// TIA Portal V17 export
// export: Created 2025-03-05T08:01:27.0836463Z, ExportSetting WithDefaults, DisplayName Totally Integrated Automation Portal, DisplayVersion V17 Update 8, DisplayName TIA Portal Openness, DisplayVersion V17 Update 8, DisplayName TIA Portal Version Control Interface, DisplayVersion V17, DisplayName SINAMICS Startdrive Advanced, DisplayVersion V17 SP2, DisplayName SINAMICS Startdrive G110M, G120, G120C, G120D, G120P, G115D, DisplayVersion V17 SP2, DisplayName SINAMICS Startdrive G130, G150, S120, S150, SINAMICS MV, S210, DisplayVersion V17 SP2, DisplayName STEP 7 Professional, DisplayVersion V17 Update 8, DisplayName SINUMERIK ONE STEP 7 Toolbox, DisplayVersion V17 Update 12, DisplayName SINUMERIK 840D sl STEP 7 Toolbox, DisplayVersion V17 Update 12, DisplayName STEP 7 Safety, DisplayVersion V17 Update 6, DisplayName WinCC Advanced, DisplayVersion V17 Update 8
FUNCTION "FC16011_METHOD_CALLS_U01_STA3_MEAS" : Void   // FC16011, LAD
{ S7_Optimized_Access := 'TRUE' }
VERSION : 0.1
// stored: AutoNumber false, IsIECCheckEnabled false, SetENOAutomatically false, UDAEnableTagReadback false
   VAR_TEMP
      AUX_WSTRING_PART_ID_STA3 : WString;
      AUX_WCHARS : Array[0..63] of WChar;
      index : Int;
      ALARM_AUX : Bool;
   END_VAR
   VAR_TEMP   // added for the SCL form of the ladder/FBD networks
      _w1 : Bool;
      _w2 : Bool;
      _w3 : Bool;
      _s5time1 : S5Time;
      _w4 : Bool;
   END_VAR
BEGIN

REGION Network 1 (SCL): TRANSFORM TO WCHARS
   FOR #index := 0 TO 63 DO
       #AUX_WCHARS[#index] := CHAR_TO_WCHAR("DB8000_PART_STATUS".UNIT_01.STATION_3.PART_A.PART_ID[#index]);
   END_FOR;
END_REGION

REGION Network 2: TRANSFORM TO WSTRING
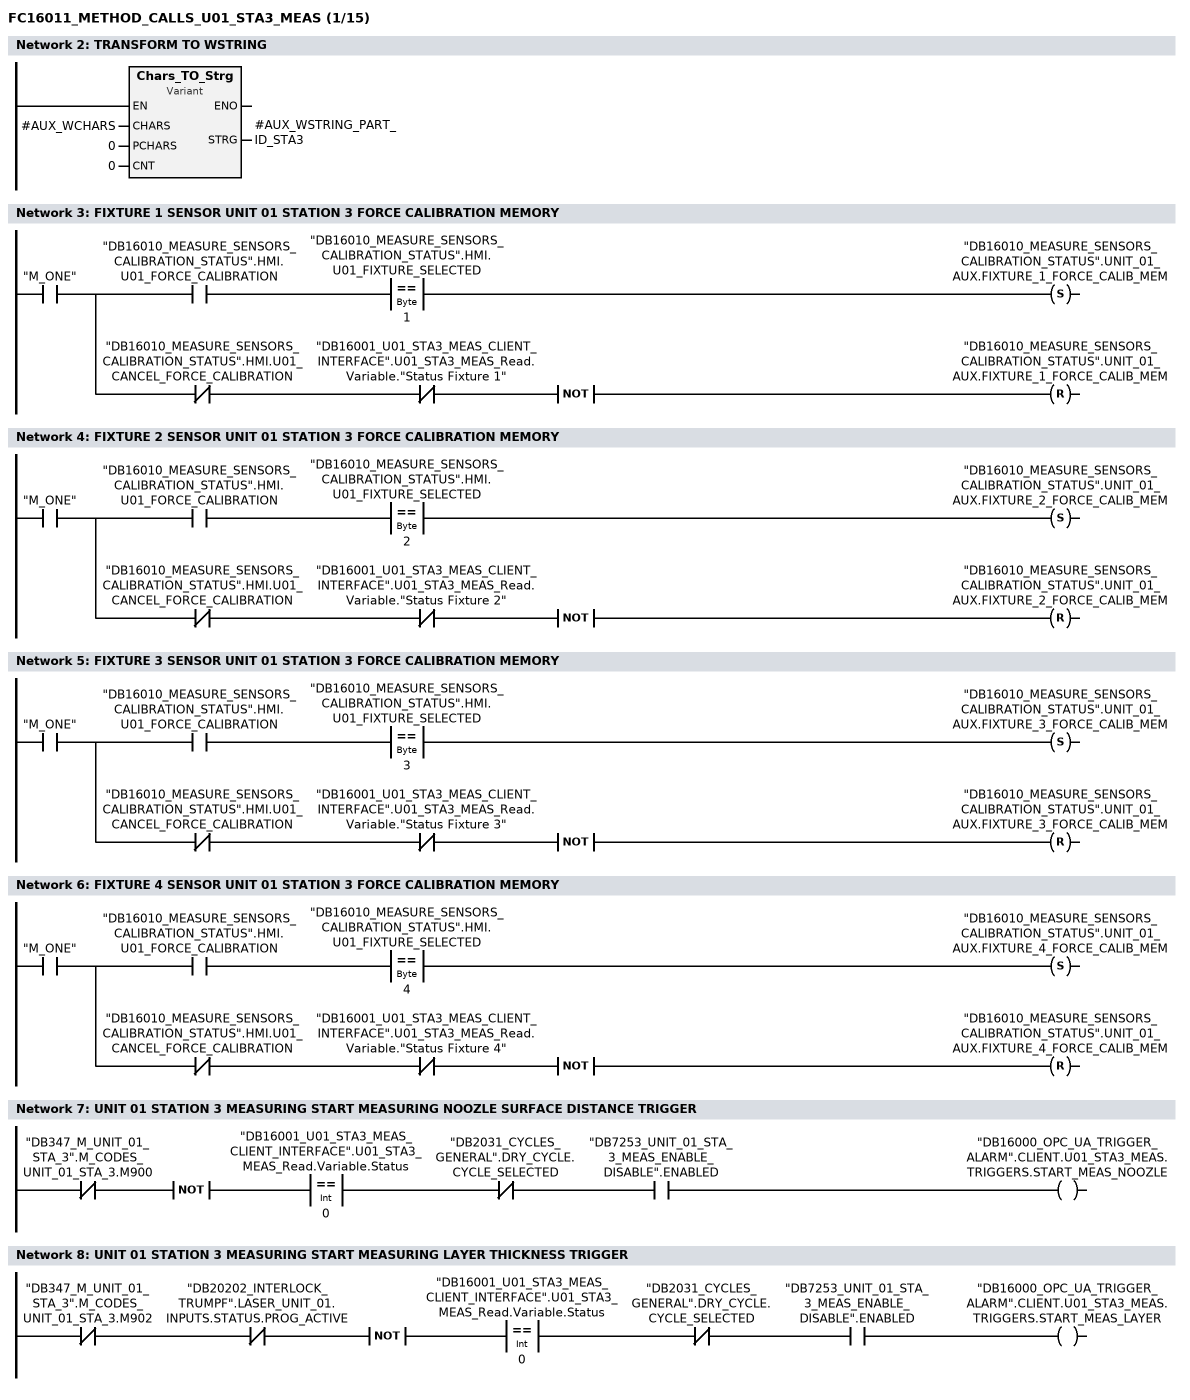
   RUNG wire#powerrail
      { S7_Templates := "[ptr_type := Variant, str_type := WString]" } Chars_TO_Strg(Chars := #AUX_WCHARS, pChars := 0, Cnt := 0, Strg => #AUX_WSTRING_PART_ID_STA3)
   END_RUNG
   // the same network as SCL:
   Chars_TO_Strg(Chars := #AUX_WCHARS, pChars := 0, Cnt := 0, Strg => #AUX_WSTRING_PART_ID_STA3);
END_REGION

REGION Network 3: FIXTURE 1 SENSOR UNIT 01 STATION 3 FORCE CALIBRATION MEMORY
   RUNG wire#powerrail
      Contact( "M_ONE" )
      wire#w1
      Contact( "DB16010_MEASURE_SENSORS_CALIBRATION_STATUS".HMI.U01_FORCE_CALIBRATION )
      { S7_Templates := "SrcType := Byte" } EQ_Contact(in1 := "DB16010_MEASURE_SENSORS_CALIBRATION_STATUS".HMI.U01_FIXTURE_SELECTED, in2 := 1)
      S_Coil( "DB16010_MEASURE_SENSORS_CALIBRATION_STATUS".UNIT_01_AUX.FIXTURE_1_FORCE_CALIB_MEM )
   END_RUNG
   RUNG wire#w1
      I_Contact( "DB16010_MEASURE_SENSORS_CALIBRATION_STATUS".HMI.U01_CANCEL_FORCE_CALIBRATION )
      I_Contact( "DB16001_U01_STA3_MEAS_CLIENT_INTERFACE".U01_STA3_MEAS_Read.Variable."Status Fixture 1" )
      Not()
      R_Coil( "DB16010_MEASURE_SENSORS_CALIBRATION_STATUS".UNIT_01_AUX.FIXTURE_1_FORCE_CALIB_MEM )
   END_RUNG
   // the same network as SCL:
   IF "M_ONE" AND "DB16010_MEASURE_SENSORS_CALIBRATION_STATUS".HMI.U01_FORCE_CALIBRATION AND ("DB16010_MEASURE_SENSORS_CALIBRATION_STATUS".HMI.U01_FIXTURE_SELECTED = 1) THEN
       "DB16010_MEASURE_SENSORS_CALIBRATION_STATUS".UNIT_01_AUX.FIXTURE_1_FORCE_CALIB_MEM := TRUE;
   END_IF;
   IF NOT ("M_ONE" AND NOT "DB16010_MEASURE_SENSORS_CALIBRATION_STATUS".HMI.U01_CANCEL_FORCE_CALIBRATION AND NOT "DB16001_U01_STA3_MEAS_CLIENT_INTERFACE".U01_STA3_MEAS_Read.Variable."Status Fixture 1") THEN
       "DB16010_MEASURE_SENSORS_CALIBRATION_STATUS".UNIT_01_AUX.FIXTURE_1_FORCE_CALIB_MEM := FALSE;
   END_IF;
END_REGION

REGION Network 4: FIXTURE 2 SENSOR UNIT 01 STATION 3 FORCE CALIBRATION MEMORY
   RUNG wire#powerrail
      Contact( "M_ONE" )
      wire#w1
      Contact( "DB16010_MEASURE_SENSORS_CALIBRATION_STATUS".HMI.U01_FORCE_CALIBRATION )
      { S7_Templates := "SrcType := Byte" } EQ_Contact(in1 := "DB16010_MEASURE_SENSORS_CALIBRATION_STATUS".HMI.U01_FIXTURE_SELECTED, in2 := 2)
      S_Coil( "DB16010_MEASURE_SENSORS_CALIBRATION_STATUS".UNIT_01_AUX.FIXTURE_2_FORCE_CALIB_MEM )
   END_RUNG
   RUNG wire#w1
      I_Contact( "DB16010_MEASURE_SENSORS_CALIBRATION_STATUS".HMI.U01_CANCEL_FORCE_CALIBRATION )
      I_Contact( "DB16001_U01_STA3_MEAS_CLIENT_INTERFACE".U01_STA3_MEAS_Read.Variable."Status Fixture 2" )
      Not()
      R_Coil( "DB16010_MEASURE_SENSORS_CALIBRATION_STATUS".UNIT_01_AUX.FIXTURE_2_FORCE_CALIB_MEM )
   END_RUNG
   // the same network as SCL:
   IF "M_ONE" AND "DB16010_MEASURE_SENSORS_CALIBRATION_STATUS".HMI.U01_FORCE_CALIBRATION AND ("DB16010_MEASURE_SENSORS_CALIBRATION_STATUS".HMI.U01_FIXTURE_SELECTED = 2) THEN
       "DB16010_MEASURE_SENSORS_CALIBRATION_STATUS".UNIT_01_AUX.FIXTURE_2_FORCE_CALIB_MEM := TRUE;
   END_IF;
   IF NOT ("M_ONE" AND NOT "DB16010_MEASURE_SENSORS_CALIBRATION_STATUS".HMI.U01_CANCEL_FORCE_CALIBRATION AND NOT "DB16001_U01_STA3_MEAS_CLIENT_INTERFACE".U01_STA3_MEAS_Read.Variable."Status Fixture 2") THEN
       "DB16010_MEASURE_SENSORS_CALIBRATION_STATUS".UNIT_01_AUX.FIXTURE_2_FORCE_CALIB_MEM := FALSE;
   END_IF;
END_REGION

REGION Network 5: FIXTURE 3 SENSOR UNIT 01 STATION 3 FORCE CALIBRATION MEMORY
   RUNG wire#powerrail
      Contact( "M_ONE" )
      wire#w1
      Contact( "DB16010_MEASURE_SENSORS_CALIBRATION_STATUS".HMI.U01_FORCE_CALIBRATION )
      { S7_Templates := "SrcType := Byte" } EQ_Contact(in1 := "DB16010_MEASURE_SENSORS_CALIBRATION_STATUS".HMI.U01_FIXTURE_SELECTED, in2 := 3)
      S_Coil( "DB16010_MEASURE_SENSORS_CALIBRATION_STATUS".UNIT_01_AUX.FIXTURE_3_FORCE_CALIB_MEM )
   END_RUNG
   RUNG wire#w1
      I_Contact( "DB16010_MEASURE_SENSORS_CALIBRATION_STATUS".HMI.U01_CANCEL_FORCE_CALIBRATION )
      I_Contact( "DB16001_U01_STA3_MEAS_CLIENT_INTERFACE".U01_STA3_MEAS_Read.Variable."Status Fixture 3" )
      Not()
      R_Coil( "DB16010_MEASURE_SENSORS_CALIBRATION_STATUS".UNIT_01_AUX.FIXTURE_3_FORCE_CALIB_MEM )
   END_RUNG
   // the same network as SCL:
   IF "M_ONE" AND "DB16010_MEASURE_SENSORS_CALIBRATION_STATUS".HMI.U01_FORCE_CALIBRATION AND ("DB16010_MEASURE_SENSORS_CALIBRATION_STATUS".HMI.U01_FIXTURE_SELECTED = 3) THEN
       "DB16010_MEASURE_SENSORS_CALIBRATION_STATUS".UNIT_01_AUX.FIXTURE_3_FORCE_CALIB_MEM := TRUE;
   END_IF;
   IF NOT ("M_ONE" AND NOT "DB16010_MEASURE_SENSORS_CALIBRATION_STATUS".HMI.U01_CANCEL_FORCE_CALIBRATION AND NOT "DB16001_U01_STA3_MEAS_CLIENT_INTERFACE".U01_STA3_MEAS_Read.Variable."Status Fixture 3") THEN
       "DB16010_MEASURE_SENSORS_CALIBRATION_STATUS".UNIT_01_AUX.FIXTURE_3_FORCE_CALIB_MEM := FALSE;
   END_IF;
END_REGION

REGION Network 6: FIXTURE 4 SENSOR UNIT 01 STATION 3 FORCE CALIBRATION MEMORY
   RUNG wire#powerrail
      Contact( "M_ONE" )
      wire#w1
      Contact( "DB16010_MEASURE_SENSORS_CALIBRATION_STATUS".HMI.U01_FORCE_CALIBRATION )
      { S7_Templates := "SrcType := Byte" } EQ_Contact(in1 := "DB16010_MEASURE_SENSORS_CALIBRATION_STATUS".HMI.U01_FIXTURE_SELECTED, in2 := 4)
      S_Coil( "DB16010_MEASURE_SENSORS_CALIBRATION_STATUS".UNIT_01_AUX.FIXTURE_4_FORCE_CALIB_MEM )
   END_RUNG
   RUNG wire#w1
      I_Contact( "DB16010_MEASURE_SENSORS_CALIBRATION_STATUS".HMI.U01_CANCEL_FORCE_CALIBRATION )
      I_Contact( "DB16001_U01_STA3_MEAS_CLIENT_INTERFACE".U01_STA3_MEAS_Read.Variable."Status Fixture 4" )
      Not()
      R_Coil( "DB16010_MEASURE_SENSORS_CALIBRATION_STATUS".UNIT_01_AUX.FIXTURE_4_FORCE_CALIB_MEM )
   END_RUNG
   // the same network as SCL:
   IF "M_ONE" AND "DB16010_MEASURE_SENSORS_CALIBRATION_STATUS".HMI.U01_FORCE_CALIBRATION AND ("DB16010_MEASURE_SENSORS_CALIBRATION_STATUS".HMI.U01_FIXTURE_SELECTED = 4) THEN
       "DB16010_MEASURE_SENSORS_CALIBRATION_STATUS".UNIT_01_AUX.FIXTURE_4_FORCE_CALIB_MEM := TRUE;
   END_IF;
   IF NOT ("M_ONE" AND NOT "DB16010_MEASURE_SENSORS_CALIBRATION_STATUS".HMI.U01_CANCEL_FORCE_CALIBRATION AND NOT "DB16001_U01_STA3_MEAS_CLIENT_INTERFACE".U01_STA3_MEAS_Read.Variable."Status Fixture 4") THEN
       "DB16010_MEASURE_SENSORS_CALIBRATION_STATUS".UNIT_01_AUX.FIXTURE_4_FORCE_CALIB_MEM := FALSE;
   END_IF;
END_REGION

REGION Network 7: UNIT 01 STATION 3 MEASURING START MEASURING NOOZLE SURFACE DISTANCE TRIGGER
   RUNG wire#powerrail
      I_Contact( "DB347_M_UNIT_01_STA_3".M_CODES_UNIT_01_STA_3.M900 )
      Not()
      { S7_Templates := "SrcType := Int" } EQ_Contact(in1 := "DB16001_U01_STA3_MEAS_CLIENT_INTERFACE".U01_STA3_MEAS_Read.Variable.Status, in2 := 0)
      I_Contact( "DB2031_CYCLES_GENERAL".DRY_CYCLE.CYCLE_SELECTED )
      Contact( "DB7253_UNIT_01_STA_3_MEAS_ENABLE_DISABLE".ENABLED )
      Coil( "DB16000_OPC_UA_TRIGGER_ALARM".CLIENT.U01_STA3_MEAS.TRIGGERS.START_MEAS_NOOZLE )
   END_RUNG
   // the same network as SCL:
   "DB16000_OPC_UA_TRIGGER_ALARM".CLIENT.U01_STA3_MEAS.TRIGGERS.START_MEAS_NOOZLE := NOT (NOT "DB347_M_UNIT_01_STA_3".M_CODES_UNIT_01_STA_3.M900) AND ("DB16001_U01_STA3_MEAS_CLIENT_INTERFACE".U01_STA3_MEAS_Read.Variable.Status = 0) AND NOT "DB2031_CYCLES_GENERAL".DRY_CYCLE.CYCLE_SELECTED AND "DB7253_UNIT_01_STA_3_MEAS_ENABLE_DISABLE".ENABLED;
END_REGION

REGION Network 8: UNIT 01 STATION 3 MEASURING START MEASURING LAYER THICKNESS TRIGGER
   RUNG wire#powerrail
      I_Contact( "DB347_M_UNIT_01_STA_3".M_CODES_UNIT_01_STA_3.M902 )
      I_Contact( "DB20202_INTERLOCK_TRUMPF".LASER_UNIT_01.INPUTS.STATUS.PROG_ACTIVE )
      Not()
      { S7_Templates := "SrcType := Int" } EQ_Contact(in1 := "DB16001_U01_STA3_MEAS_CLIENT_INTERFACE".U01_STA3_MEAS_Read.Variable.Status, in2 := 0)
      I_Contact( "DB2031_CYCLES_GENERAL".DRY_CYCLE.CYCLE_SELECTED )
      Contact( "DB7253_UNIT_01_STA_3_MEAS_ENABLE_DISABLE".ENABLED )
      Coil( "DB16000_OPC_UA_TRIGGER_ALARM".CLIENT.U01_STA3_MEAS.TRIGGERS.START_MEAS_LAYER )
   END_RUNG
   // the same network as SCL:
   "DB16000_OPC_UA_TRIGGER_ALARM".CLIENT.U01_STA3_MEAS.TRIGGERS.START_MEAS_LAYER := NOT (NOT "DB347_M_UNIT_01_STA_3".M_CODES_UNIT_01_STA_3.M902 AND NOT "DB20202_INTERLOCK_TRUMPF".LASER_UNIT_01.INPUTS.STATUS.PROG_ACTIVE) AND ("DB16001_U01_STA3_MEAS_CLIENT_INTERFACE".U01_STA3_MEAS_Read.Variable.Status = 0) AND NOT "DB2031_CYCLES_GENERAL".DRY_CYCLE.CYCLE_SELECTED AND "DB7253_UNIT_01_STA_3_MEAS_ENABLE_DISABLE".ENABLED;
END_REGION

REGION Network 9: UNIT 01 STATION 3 MEASURING STOP MEASURING LAYER THICKNESS TRIGGER
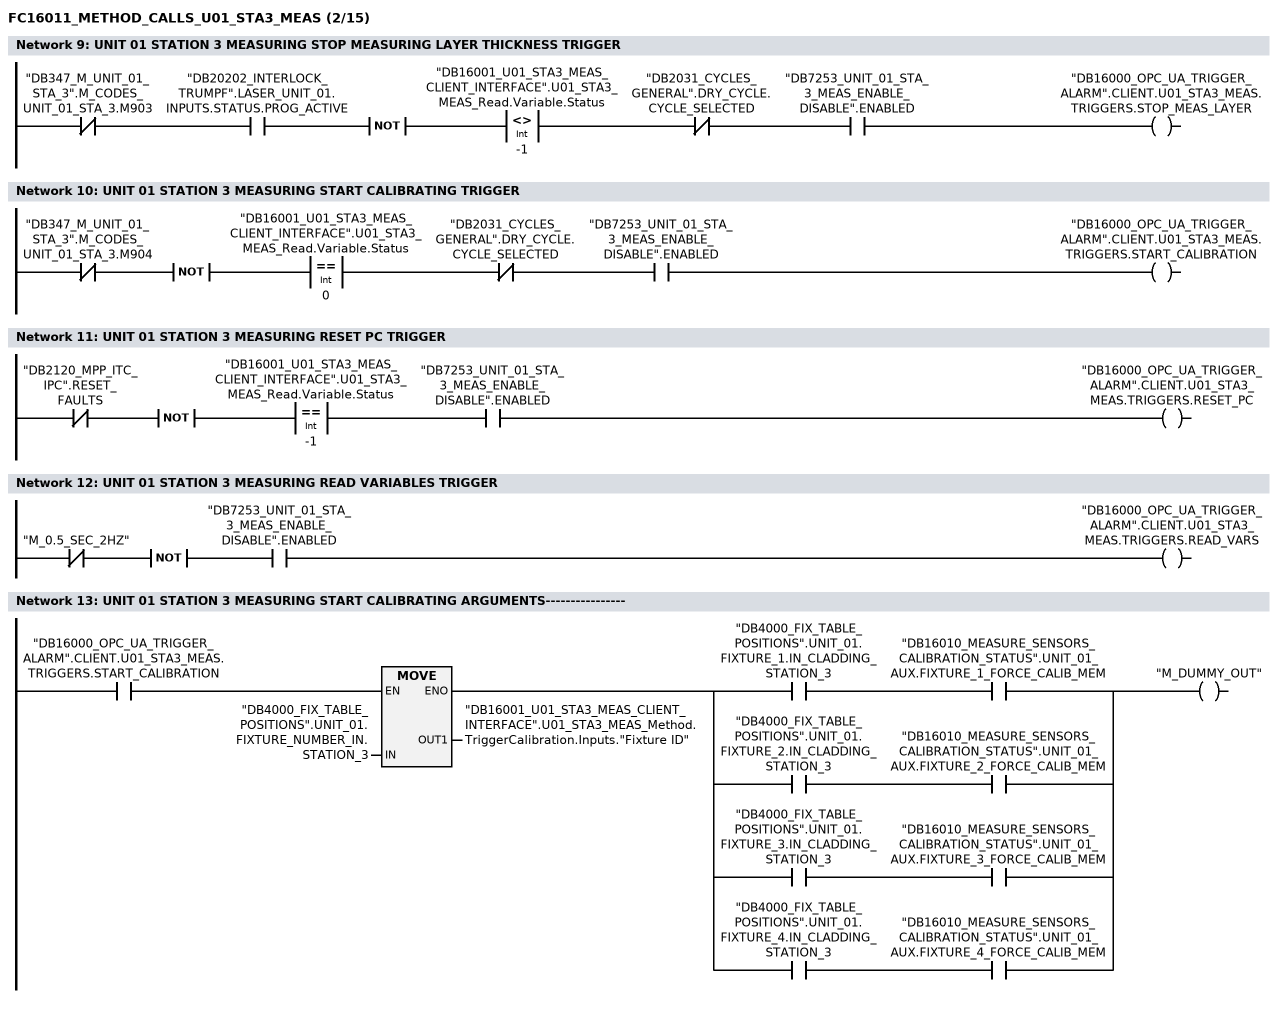
   RUNG wire#powerrail
      I_Contact( "DB347_M_UNIT_01_STA_3".M_CODES_UNIT_01_STA_3.M903 )
      Contact( "DB20202_INTERLOCK_TRUMPF".LASER_UNIT_01.INPUTS.STATUS.PROG_ACTIVE )
      Not()
      { S7_Templates := "SrcType := Int" } NE_Contact(in1 := "DB16001_U01_STA3_MEAS_CLIENT_INTERFACE".U01_STA3_MEAS_Read.Variable.Status, in2 := -1)
      I_Contact( "DB2031_CYCLES_GENERAL".DRY_CYCLE.CYCLE_SELECTED )
      Contact( "DB7253_UNIT_01_STA_3_MEAS_ENABLE_DISABLE".ENABLED )
      Coil( "DB16000_OPC_UA_TRIGGER_ALARM".CLIENT.U01_STA3_MEAS.TRIGGERS.STOP_MEAS_LAYER )
   END_RUNG
   // the same network as SCL:
   "DB16000_OPC_UA_TRIGGER_ALARM".CLIENT.U01_STA3_MEAS.TRIGGERS.STOP_MEAS_LAYER := NOT (NOT "DB347_M_UNIT_01_STA_3".M_CODES_UNIT_01_STA_3.M903 AND "DB20202_INTERLOCK_TRUMPF".LASER_UNIT_01.INPUTS.STATUS.PROG_ACTIVE) AND ("DB16001_U01_STA3_MEAS_CLIENT_INTERFACE".U01_STA3_MEAS_Read.Variable.Status <> (-1)) AND NOT "DB2031_CYCLES_GENERAL".DRY_CYCLE.CYCLE_SELECTED AND "DB7253_UNIT_01_STA_3_MEAS_ENABLE_DISABLE".ENABLED;
END_REGION

REGION Network 10: UNIT 01 STATION 3 MEASURING START CALIBRATING TRIGGER
   RUNG wire#powerrail
      I_Contact( "DB347_M_UNIT_01_STA_3".M_CODES_UNIT_01_STA_3.M904 )
      Not()
      { S7_Templates := "SrcType := Int" } EQ_Contact(in1 := "DB16001_U01_STA3_MEAS_CLIENT_INTERFACE".U01_STA3_MEAS_Read.Variable.Status, in2 := 0)
      I_Contact( "DB2031_CYCLES_GENERAL".DRY_CYCLE.CYCLE_SELECTED )
      Contact( "DB7253_UNIT_01_STA_3_MEAS_ENABLE_DISABLE".ENABLED )
      Coil( "DB16000_OPC_UA_TRIGGER_ALARM".CLIENT.U01_STA3_MEAS.TRIGGERS.START_CALIBRATION )
   END_RUNG
   // the same network as SCL:
   "DB16000_OPC_UA_TRIGGER_ALARM".CLIENT.U01_STA3_MEAS.TRIGGERS.START_CALIBRATION := NOT (NOT "DB347_M_UNIT_01_STA_3".M_CODES_UNIT_01_STA_3.M904) AND ("DB16001_U01_STA3_MEAS_CLIENT_INTERFACE".U01_STA3_MEAS_Read.Variable.Status = 0) AND NOT "DB2031_CYCLES_GENERAL".DRY_CYCLE.CYCLE_SELECTED AND "DB7253_UNIT_01_STA_3_MEAS_ENABLE_DISABLE".ENABLED;
END_REGION

REGION Network 11: UNIT 01 STATION 3 MEASURING RESET PC TRIGGER
   RUNG wire#powerrail
      I_Contact( "DB2120_MPP_ITC_IPC".RESET_FAULTS )
      Not()
      { S7_Templates := "SrcType := Int" } EQ_Contact(in1 := "DB16001_U01_STA3_MEAS_CLIENT_INTERFACE".U01_STA3_MEAS_Read.Variable.Status, in2 := -1)
      Contact( "DB7253_UNIT_01_STA_3_MEAS_ENABLE_DISABLE".ENABLED )
      Coil( "DB16000_OPC_UA_TRIGGER_ALARM".CLIENT.U01_STA3_MEAS.TRIGGERS.RESET_PC )
   END_RUNG
   // the same network as SCL:
   "DB16000_OPC_UA_TRIGGER_ALARM".CLIENT.U01_STA3_MEAS.TRIGGERS.RESET_PC := NOT (NOT "DB2120_MPP_ITC_IPC".RESET_FAULTS) AND ("DB16001_U01_STA3_MEAS_CLIENT_INTERFACE".U01_STA3_MEAS_Read.Variable.Status = (-1)) AND "DB7253_UNIT_01_STA_3_MEAS_ENABLE_DISABLE".ENABLED;
END_REGION

REGION Network 12: UNIT 01 STATION 3 MEASURING READ VARIABLES TRIGGER
   RUNG wire#powerrail
      I_Contact( "M_0.5_SEC_2HZ" )
      Not()
      Contact( "DB7253_UNIT_01_STA_3_MEAS_ENABLE_DISABLE".ENABLED )
      Coil( "DB16000_OPC_UA_TRIGGER_ALARM".CLIENT.U01_STA3_MEAS.TRIGGERS.READ_VARS )
   END_RUNG
   // the same network as SCL:
   "DB16000_OPC_UA_TRIGGER_ALARM".CLIENT.U01_STA3_MEAS.TRIGGERS.READ_VARS := NOT (NOT "M_0.5_SEC_2HZ") AND "DB7253_UNIT_01_STA_3_MEAS_ENABLE_DISABLE".ENABLED;
END_REGION

REGION Network 13: UNIT 01 STATION 3 MEASURING START CALIBRATING ARGUMENTS----------------
   RUNG wire#powerrail
      Contact( "DB16000_OPC_UA_TRIGGER_ALARM".CLIENT.U01_STA3_MEAS.TRIGGERS.START_CALIBRATION )
      Move(in := "DB4000_FIX_TABLE_POSITIONS".UNIT_01.FIXTURE_NUMBER_IN.STATION_3, out1 => "DB16001_U01_STA3_MEAS_CLIENT_INTERFACE".U01_STA3_MEAS_Method.TriggerCalibration.Inputs."Fixture ID")
      wire#w1
      Contact( "DB4000_FIX_TABLE_POSITIONS".UNIT_01.FIXTURE_1.IN_CLADDING_STATION_3 )
      Contact( "DB16010_MEASURE_SENSORS_CALIBRATION_STATUS".UNIT_01_AUX.FIXTURE_1_FORCE_CALIB_MEM )
      wire#w2
      Coil( "M_DUMMY_OUT" )
   END_RUNG
   RUNG wire#w1
      Contact( "DB4000_FIX_TABLE_POSITIONS".UNIT_01.FIXTURE_2.IN_CLADDING_STATION_3 )
      Contact( "DB16010_MEASURE_SENSORS_CALIBRATION_STATUS".UNIT_01_AUX.FIXTURE_2_FORCE_CALIB_MEM )
   END_RUNG wire#w2
   RUNG wire#w1
      Contact( "DB4000_FIX_TABLE_POSITIONS".UNIT_01.FIXTURE_3.IN_CLADDING_STATION_3 )
      Contact( "DB16010_MEASURE_SENSORS_CALIBRATION_STATUS".UNIT_01_AUX.FIXTURE_3_FORCE_CALIB_MEM )
   END_RUNG wire#w2
   RUNG wire#w1
      Contact( "DB4000_FIX_TABLE_POSITIONS".UNIT_01.FIXTURE_4.IN_CLADDING_STATION_3 )
      Contact( "DB16010_MEASURE_SENSORS_CALIBRATION_STATUS".UNIT_01_AUX.FIXTURE_4_FORCE_CALIB_MEM )
   END_RUNG wire#w2
   // the same network as SCL:
   IF "DB16000_OPC_UA_TRIGGER_ALARM".CLIENT.U01_STA3_MEAS.TRIGGERS.START_CALIBRATION THEN
       "DB16001_U01_STA3_MEAS_CLIENT_INTERFACE".U01_STA3_MEAS_Method.TriggerCalibration.Inputs."Fixture ID" := "DB4000_FIX_TABLE_POSITIONS".UNIT_01.FIXTURE_NUMBER_IN.STATION_3;
   END_IF;
   "M_DUMMY_OUT" := "DB16000_OPC_UA_TRIGGER_ALARM".CLIENT.U01_STA3_MEAS.TRIGGERS.START_CALIBRATION AND (("DB4000_FIX_TABLE_POSITIONS".UNIT_01.FIXTURE_1.IN_CLADDING_STATION_3 AND "DB16010_MEASURE_SENSORS_CALIBRATION_STATUS".UNIT_01_AUX.FIXTURE_1_FORCE_CALIB_MEM) OR ("DB4000_FIX_TABLE_POSITIONS".UNIT_01.FIXTURE_2.IN_CLADDING_STATION_3 AND "DB16010_MEASURE_SENSORS_CALIBRATION_STATUS".UNIT_01_AUX.FIXTURE_2_FORCE_CALIB_MEM) OR ("DB4000_FIX_TABLE_POSITIONS".UNIT_01.FIXTURE_3.IN_CLADDING_STATION_3 AND "DB16010_MEASURE_SENSORS_CALIBRATION_STATUS".UNIT_01_AUX.FIXTURE_3_FORCE_CALIB_MEM) OR ("DB4000_FIX_TABLE_POSITIONS".UNIT_01.FIXTURE_4.IN_CLADDING_STATION_3 AND "DB16010_MEASURE_SENSORS_CALIBRATION_STATUS".UNIT_01_AUX.FIXTURE_4_FORCE_CALIB_MEM));
END_REGION

REGION Network 14: UNIT 01 STATION 3 MEASURING START MEASURING NOOZLE SURFACE DISTANCE TRIGGER CALL
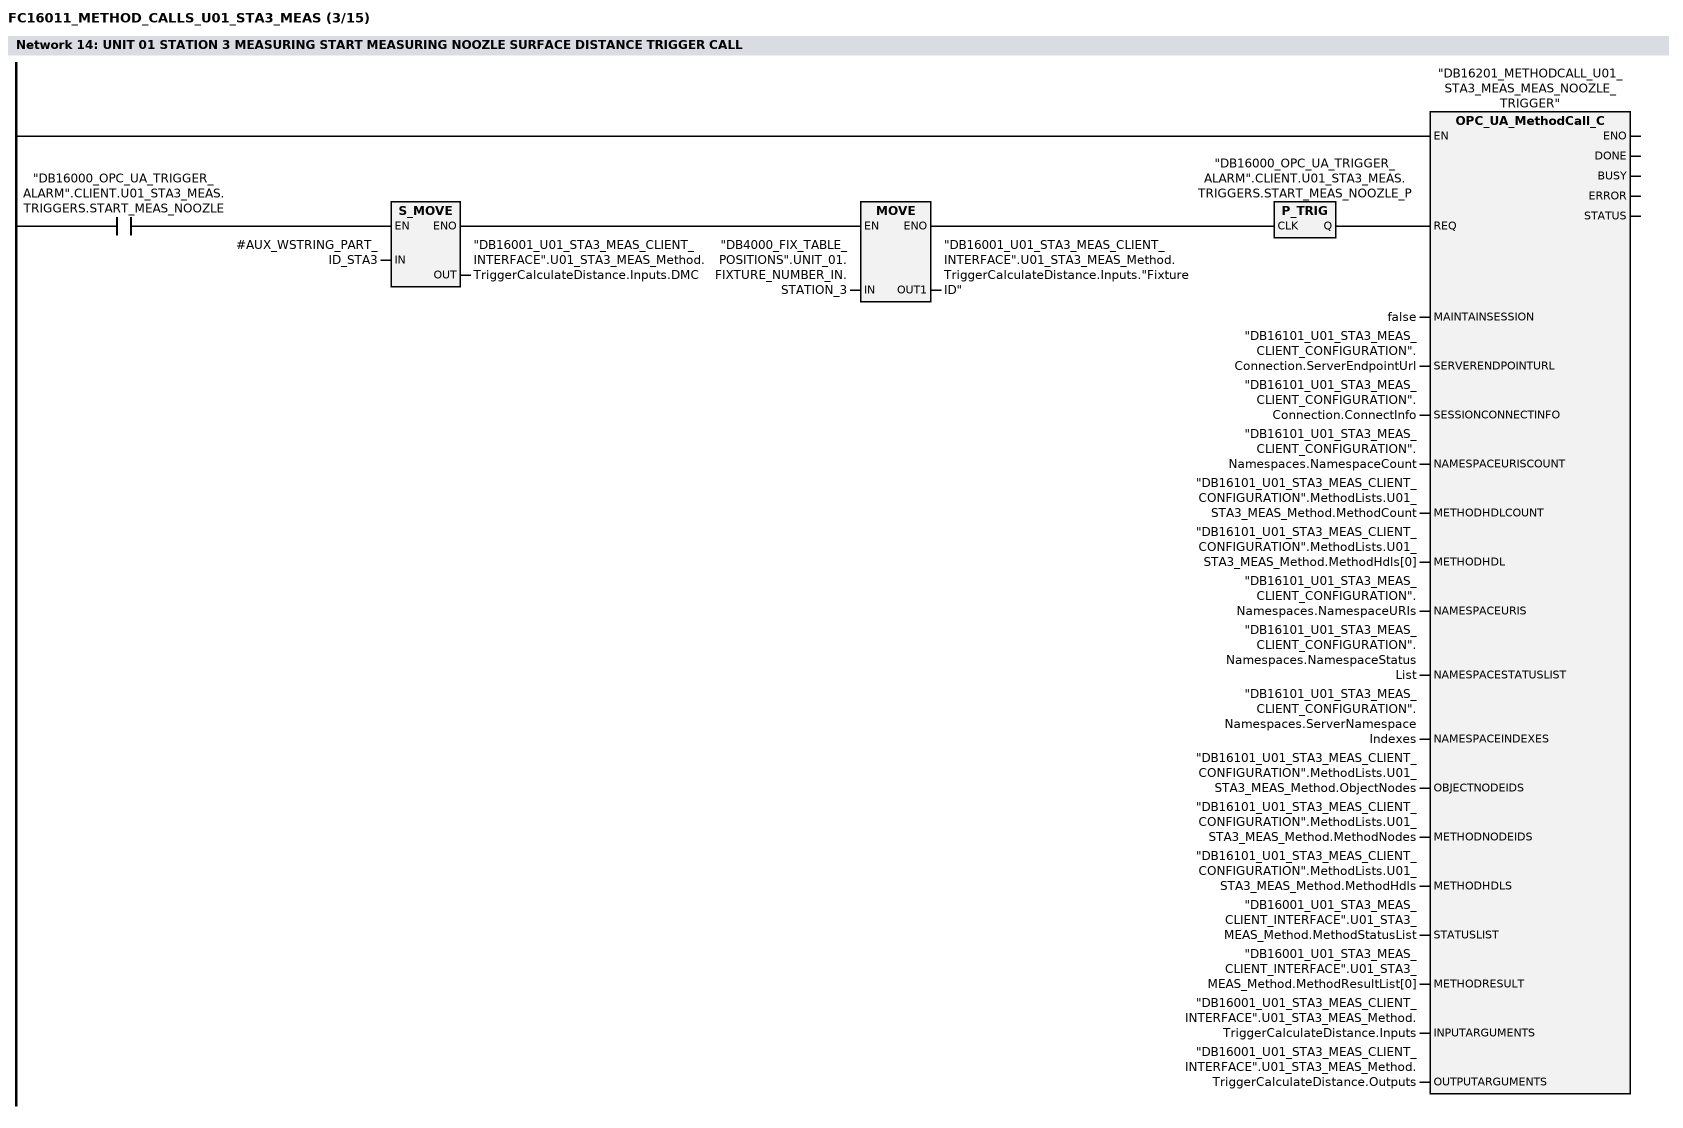
   RUNG wire#powerrail
      "DB16201_METHODCALL_U01_STA3_MEAS_MEAS_NOOZLE_TRIGGER".OPC_UA_MethodCall_C(REQ := wire#w1, MaintainSession := false, ServerEndpointUrl := "DB16101_U01_STA3_MEAS_CLIENT_CONFIGURATION".Connection.ServerEndpointUrl, SessionConnectInfo := "DB16101_U01_STA3_MEAS_CLIENT_CONFIGURATION".Connection.ConnectInfo, NamespaceUrisCount := "DB16101_U01_STA3_MEAS_CLIENT_CONFIGURATION".Namespaces.NamespaceCount, MethodHdlCount := "DB16101_U01_STA3_MEAS_CLIENT_CONFIGURATION".MethodLists.U01_STA3_MEAS_Method.MethodCount, MethodHdl := "DB16101_U01_STA3_MEAS_CLIENT_CONFIGURATION".MethodLists.U01_STA3_MEAS_Method.MethodHdls[0], NamespaceUris := "DB16101_U01_STA3_MEAS_CLIENT_CONFIGURATION".Namespaces.NamespaceURIs, NamespaceStatusList := "DB16101_U01_STA3_MEAS_CLIENT_CONFIGURATION".Namespaces.NamespaceStatusList, NamespaceIndexes := "DB16101_U01_STA3_MEAS_CLIENT_CONFIGURATION".Namespaces.ServerNamespaceIndexes, ObjectNodeIDs := "DB16101_U01_STA3_MEAS_CLIENT_CONFIGURATION".MethodLists.U01_STA3_MEAS_Method.ObjectNodes, MethodNodeIDs := "DB16101_U01_STA3_MEAS_CLIENT_CONFIGURATION".MethodLists.U01_STA3_MEAS_Method.MethodNodes, MethodHdls := "DB16101_U01_STA3_MEAS_CLIENT_CONFIGURATION".MethodLists.U01_STA3_MEAS_Method.MethodHdls, StatusList := "DB16001_U01_STA3_MEAS_CLIENT_INTERFACE".U01_STA3_MEAS_Method.MethodStatusList, MethodResult := "DB16001_U01_STA3_MEAS_CLIENT_INTERFACE".U01_STA3_MEAS_Method.MethodResultList[0], InputArguments := "DB16001_U01_STA3_MEAS_CLIENT_INTERFACE".U01_STA3_MEAS_Method.TriggerCalculateDistance.Inputs, OutputArguments := "DB16001_U01_STA3_MEAS_CLIENT_INTERFACE".U01_STA3_MEAS_Method.TriggerCalculateDistance.Outputs, Done =>, Busy =>, Error =>, Status =>)
   END_RUNG
   RUNG wire#powerrail
      Contact( "DB16000_OPC_UA_TRIGGER_ALARM".CLIENT.U01_STA3_MEAS.TRIGGERS.START_MEAS_NOOZLE )
      S_Move(in := #AUX_WSTRING_PART_ID_STA3, out => "DB16001_U01_STA3_MEAS_CLIENT_INTERFACE".U01_STA3_MEAS_Method.TriggerCalculateDistance.Inputs.DMC)
      Move(in := "DB4000_FIX_TABLE_POSITIONS".UNIT_01.FIXTURE_NUMBER_IN.STATION_3, out1 => "DB16001_U01_STA3_MEAS_CLIENT_INTERFACE".U01_STA3_MEAS_Method.TriggerCalculateDistance.Inputs."Fixture ID")
      P_Trig( "DB16000_OPC_UA_TRIGGER_ALARM".CLIENT.U01_STA3_MEAS.TRIGGERS.START_MEAS_NOOZLE_P )
   END_RUNG wire#w1
   // the same network as SCL:
   IF "DB16000_OPC_UA_TRIGGER_ALARM".CLIENT.U01_STA3_MEAS.TRIGGERS.START_MEAS_NOOZLE THEN
       "DB16001_U01_STA3_MEAS_CLIENT_INTERFACE".U01_STA3_MEAS_Method.TriggerCalculateDistance.Inputs.DMC := #AUX_WSTRING_PART_ID_STA3;
       "DB16001_U01_STA3_MEAS_CLIENT_INTERFACE".U01_STA3_MEAS_Method.TriggerCalculateDistance.Inputs."Fixture ID" := "DB4000_FIX_TABLE_POSITIONS".UNIT_01.FIXTURE_NUMBER_IN.STATION_3;
   END_IF;
   #_w1 := "DB16000_OPC_UA_TRIGGER_ALARM".CLIENT.U01_STA3_MEAS.TRIGGERS.START_MEAS_NOOZLE AND NOT "DB16000_OPC_UA_TRIGGER_ALARM".CLIENT.U01_STA3_MEAS.TRIGGERS.START_MEAS_NOOZLE_P;   // rising edge
   "DB16000_OPC_UA_TRIGGER_ALARM".CLIENT.U01_STA3_MEAS.TRIGGERS.START_MEAS_NOOZLE_P := "DB16000_OPC_UA_TRIGGER_ALARM".CLIENT.U01_STA3_MEAS.TRIGGERS.START_MEAS_NOOZLE;
   "DB16201_METHODCALL_U01_STA3_MEAS_MEAS_NOOZLE_TRIGGER"(REQ := #_w1,   // OPC_UA_MethodCall_C
                           MaintainSession := false,
                           ServerEndpointUrl := "DB16101_U01_STA3_MEAS_CLIENT_CONFIGURATION".Connection.ServerEndpointUrl,
                           SessionConnectInfo := "DB16101_U01_STA3_MEAS_CLIENT_CONFIGURATION".Connection.ConnectInfo,
                           NamespaceUrisCount := "DB16101_U01_STA3_MEAS_CLIENT_CONFIGURATION".Namespaces.NamespaceCount,
                           MethodHdlCount := "DB16101_U01_STA3_MEAS_CLIENT_CONFIGURATION".MethodLists.U01_STA3_MEAS_Method.MethodCount,
                           MethodHdl := "DB16101_U01_STA3_MEAS_CLIENT_CONFIGURATION".MethodLists.U01_STA3_MEAS_Method.MethodHdls[0],
                           NamespaceUris := "DB16101_U01_STA3_MEAS_CLIENT_CONFIGURATION".Namespaces.NamespaceURIs,
                           NamespaceStatusList := "DB16101_U01_STA3_MEAS_CLIENT_CONFIGURATION".Namespaces.NamespaceStatusList,
                           NamespaceIndexes := "DB16101_U01_STA3_MEAS_CLIENT_CONFIGURATION".Namespaces.ServerNamespaceIndexes,
                           ObjectNodeIDs := "DB16101_U01_STA3_MEAS_CLIENT_CONFIGURATION".MethodLists.U01_STA3_MEAS_Method.ObjectNodes,
                           MethodNodeIDs := "DB16101_U01_STA3_MEAS_CLIENT_CONFIGURATION".MethodLists.U01_STA3_MEAS_Method.MethodNodes,
                           MethodHdls := "DB16101_U01_STA3_MEAS_CLIENT_CONFIGURATION".MethodLists.U01_STA3_MEAS_Method.MethodHdls,
                           StatusList := "DB16001_U01_STA3_MEAS_CLIENT_INTERFACE".U01_STA3_MEAS_Method.MethodStatusList,
                           MethodResult := "DB16001_U01_STA3_MEAS_CLIENT_INTERFACE".U01_STA3_MEAS_Method.MethodResultList[0],
                           InputArguments := "DB16001_U01_STA3_MEAS_CLIENT_INTERFACE".U01_STA3_MEAS_Method.TriggerCalculateDistance.Inputs,
                           OutputArguments := "DB16001_U01_STA3_MEAS_CLIENT_INTERFACE".U01_STA3_MEAS_Method.TriggerCalculateDistance.Outputs);
END_REGION

REGION Network 15: UNIT 01 STATION 3 MEASURING START MEASURING LAYER THICKNESS TRIGGER CALL
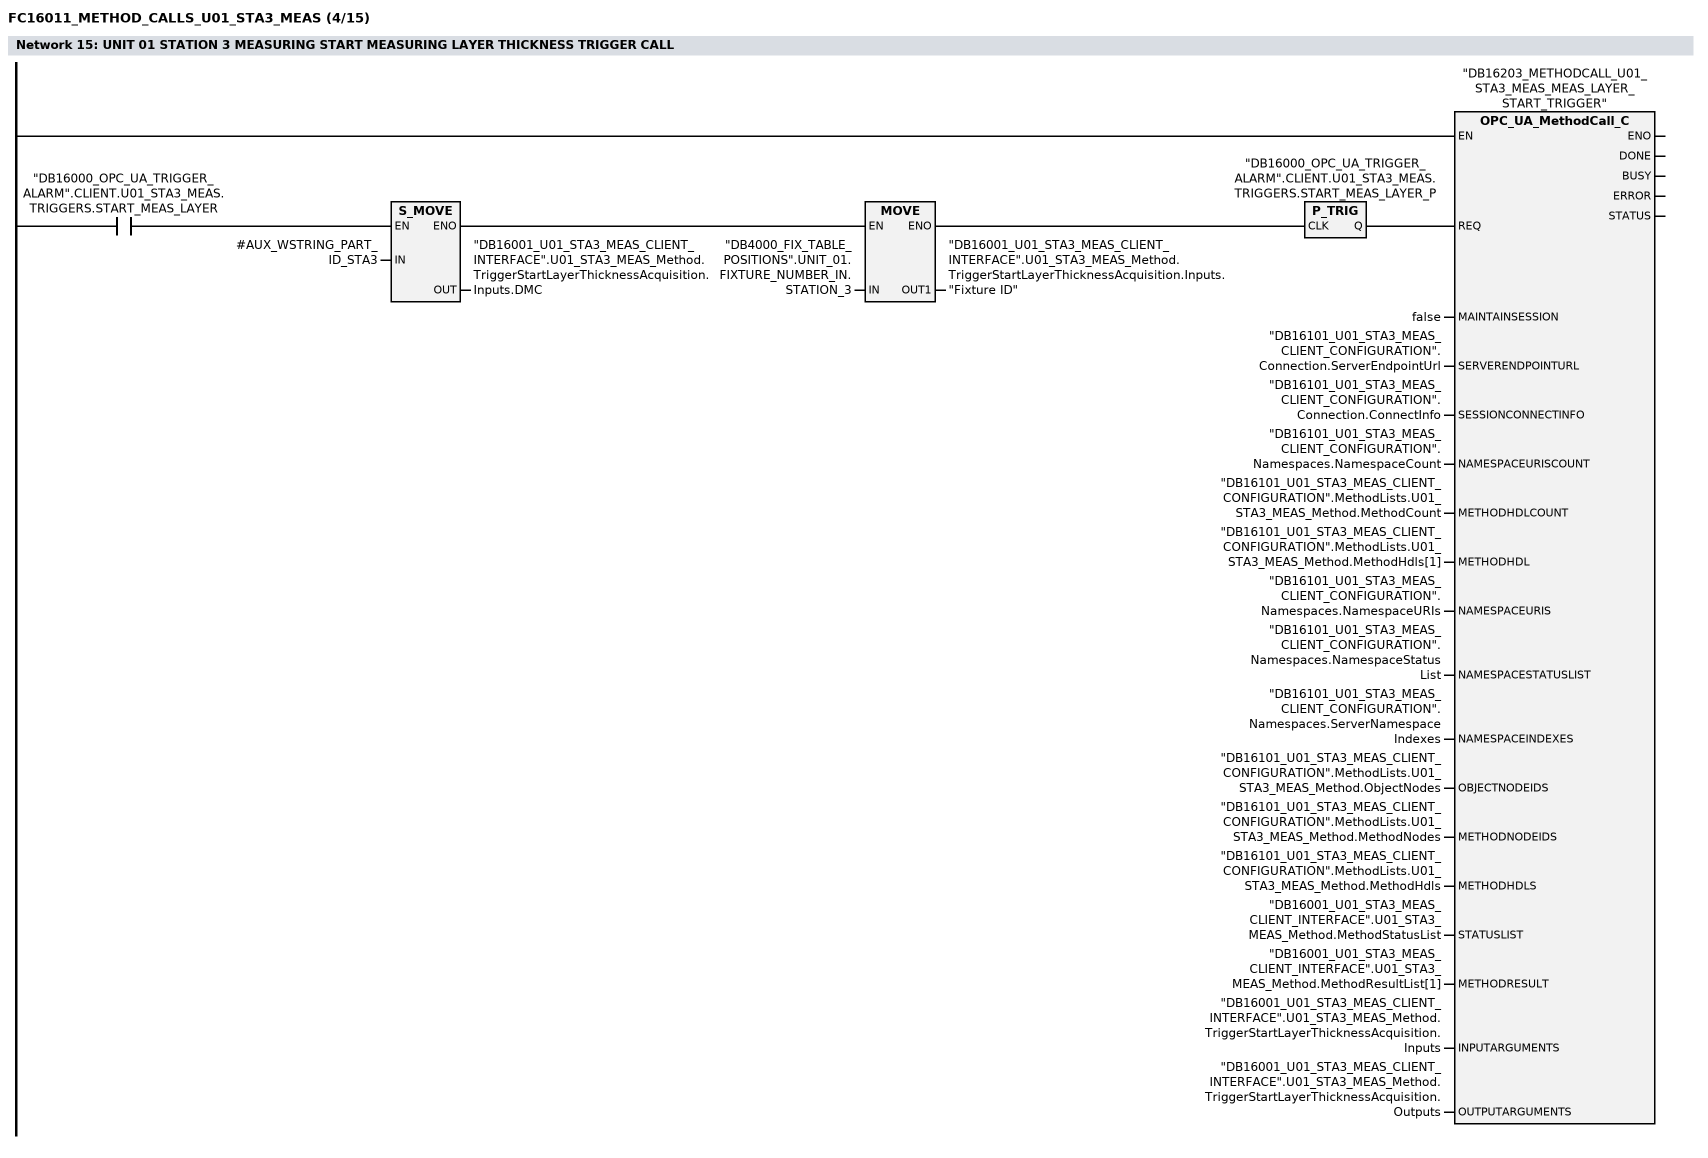
   RUNG wire#powerrail
      "DB16203_METHODCALL_U01_STA3_MEAS_MEAS_LAYER_START_TRIGGER".OPC_UA_MethodCall_C(REQ := wire#w1, MaintainSession := false, ServerEndpointUrl := "DB16101_U01_STA3_MEAS_CLIENT_CONFIGURATION".Connection.ServerEndpointUrl, SessionConnectInfo := "DB16101_U01_STA3_MEAS_CLIENT_CONFIGURATION".Connection.ConnectInfo, NamespaceUrisCount := "DB16101_U01_STA3_MEAS_CLIENT_CONFIGURATION".Namespaces.NamespaceCount, MethodHdlCount := "DB16101_U01_STA3_MEAS_CLIENT_CONFIGURATION".MethodLists.U01_STA3_MEAS_Method.MethodCount, MethodHdl := "DB16101_U01_STA3_MEAS_CLIENT_CONFIGURATION".MethodLists.U01_STA3_MEAS_Method.MethodHdls[1], NamespaceUris := "DB16101_U01_STA3_MEAS_CLIENT_CONFIGURATION".Namespaces.NamespaceURIs, NamespaceStatusList := "DB16101_U01_STA3_MEAS_CLIENT_CONFIGURATION".Namespaces.NamespaceStatusList, NamespaceIndexes := "DB16101_U01_STA3_MEAS_CLIENT_CONFIGURATION".Namespaces.ServerNamespaceIndexes, ObjectNodeIDs := "DB16101_U01_STA3_MEAS_CLIENT_CONFIGURATION".MethodLists.U01_STA3_MEAS_Method.ObjectNodes, MethodNodeIDs := "DB16101_U01_STA3_MEAS_CLIENT_CONFIGURATION".MethodLists.U01_STA3_MEAS_Method.MethodNodes, MethodHdls := "DB16101_U01_STA3_MEAS_CLIENT_CONFIGURATION".MethodLists.U01_STA3_MEAS_Method.MethodHdls, StatusList := "DB16001_U01_STA3_MEAS_CLIENT_INTERFACE".U01_STA3_MEAS_Method.MethodStatusList, MethodResult := "DB16001_U01_STA3_MEAS_CLIENT_INTERFACE".U01_STA3_MEAS_Method.MethodResultList[1], InputArguments := "DB16001_U01_STA3_MEAS_CLIENT_INTERFACE".U01_STA3_MEAS_Method.TriggerStartLayerThicknessAcquisition.Inputs, OutputArguments := "DB16001_U01_STA3_MEAS_CLIENT_INTERFACE".U01_STA3_MEAS_Method.TriggerStartLayerThicknessAcquisition.Outputs, Done =>, Busy =>, Error =>, Status =>)
   END_RUNG
   RUNG wire#powerrail
      Contact( "DB16000_OPC_UA_TRIGGER_ALARM".CLIENT.U01_STA3_MEAS.TRIGGERS.START_MEAS_LAYER )
      S_Move(in := #AUX_WSTRING_PART_ID_STA3, out => "DB16001_U01_STA3_MEAS_CLIENT_INTERFACE".U01_STA3_MEAS_Method.TriggerStartLayerThicknessAcquisition.Inputs.DMC)
      Move(in := "DB4000_FIX_TABLE_POSITIONS".UNIT_01.FIXTURE_NUMBER_IN.STATION_3, out1 => "DB16001_U01_STA3_MEAS_CLIENT_INTERFACE".U01_STA3_MEAS_Method.TriggerStartLayerThicknessAcquisition.Inputs."Fixture ID")
      P_Trig( "DB16000_OPC_UA_TRIGGER_ALARM".CLIENT.U01_STA3_MEAS.TRIGGERS.START_MEAS_LAYER_P )
   END_RUNG wire#w1
   // the same network as SCL:
   IF "DB16000_OPC_UA_TRIGGER_ALARM".CLIENT.U01_STA3_MEAS.TRIGGERS.START_MEAS_LAYER THEN
       "DB16001_U01_STA3_MEAS_CLIENT_INTERFACE".U01_STA3_MEAS_Method.TriggerStartLayerThicknessAcquisition.Inputs.DMC := #AUX_WSTRING_PART_ID_STA3;
       "DB16001_U01_STA3_MEAS_CLIENT_INTERFACE".U01_STA3_MEAS_Method.TriggerStartLayerThicknessAcquisition.Inputs."Fixture ID" := "DB4000_FIX_TABLE_POSITIONS".UNIT_01.FIXTURE_NUMBER_IN.STATION_3;
   END_IF;
   #_w1 := "DB16000_OPC_UA_TRIGGER_ALARM".CLIENT.U01_STA3_MEAS.TRIGGERS.START_MEAS_LAYER AND NOT "DB16000_OPC_UA_TRIGGER_ALARM".CLIENT.U01_STA3_MEAS.TRIGGERS.START_MEAS_LAYER_P;   // rising edge
   "DB16000_OPC_UA_TRIGGER_ALARM".CLIENT.U01_STA3_MEAS.TRIGGERS.START_MEAS_LAYER_P := "DB16000_OPC_UA_TRIGGER_ALARM".CLIENT.U01_STA3_MEAS.TRIGGERS.START_MEAS_LAYER;
   "DB16203_METHODCALL_U01_STA3_MEAS_MEAS_LAYER_START_TRIGGER"(REQ := #_w1,   // OPC_UA_MethodCall_C
                           MaintainSession := false,
                           ServerEndpointUrl := "DB16101_U01_STA3_MEAS_CLIENT_CONFIGURATION".Connection.ServerEndpointUrl,
                           SessionConnectInfo := "DB16101_U01_STA3_MEAS_CLIENT_CONFIGURATION".Connection.ConnectInfo,
                           NamespaceUrisCount := "DB16101_U01_STA3_MEAS_CLIENT_CONFIGURATION".Namespaces.NamespaceCount,
                           MethodHdlCount := "DB16101_U01_STA3_MEAS_CLIENT_CONFIGURATION".MethodLists.U01_STA3_MEAS_Method.MethodCount,
                           MethodHdl := "DB16101_U01_STA3_MEAS_CLIENT_CONFIGURATION".MethodLists.U01_STA3_MEAS_Method.MethodHdls[1],
                           NamespaceUris := "DB16101_U01_STA3_MEAS_CLIENT_CONFIGURATION".Namespaces.NamespaceURIs,
                           NamespaceStatusList := "DB16101_U01_STA3_MEAS_CLIENT_CONFIGURATION".Namespaces.NamespaceStatusList,
                           NamespaceIndexes := "DB16101_U01_STA3_MEAS_CLIENT_CONFIGURATION".Namespaces.ServerNamespaceIndexes,
                           ObjectNodeIDs := "DB16101_U01_STA3_MEAS_CLIENT_CONFIGURATION".MethodLists.U01_STA3_MEAS_Method.ObjectNodes,
                           MethodNodeIDs := "DB16101_U01_STA3_MEAS_CLIENT_CONFIGURATION".MethodLists.U01_STA3_MEAS_Method.MethodNodes,
                           MethodHdls := "DB16101_U01_STA3_MEAS_CLIENT_CONFIGURATION".MethodLists.U01_STA3_MEAS_Method.MethodHdls,
                           StatusList := "DB16001_U01_STA3_MEAS_CLIENT_INTERFACE".U01_STA3_MEAS_Method.MethodStatusList,
                           MethodResult := "DB16001_U01_STA3_MEAS_CLIENT_INTERFACE".U01_STA3_MEAS_Method.MethodResultList[1],
                           InputArguments := "DB16001_U01_STA3_MEAS_CLIENT_INTERFACE".U01_STA3_MEAS_Method.TriggerStartLayerThicknessAcquisition.Inputs,
                           OutputArguments := "DB16001_U01_STA3_MEAS_CLIENT_INTERFACE".U01_STA3_MEAS_Method.TriggerStartLayerThicknessAcquisition.Outputs);
END_REGION

REGION Network 16: UNIT 01 STATION 3 MEASURING STOP MEASURING LAYER THICKNESS TRIGGER CALL
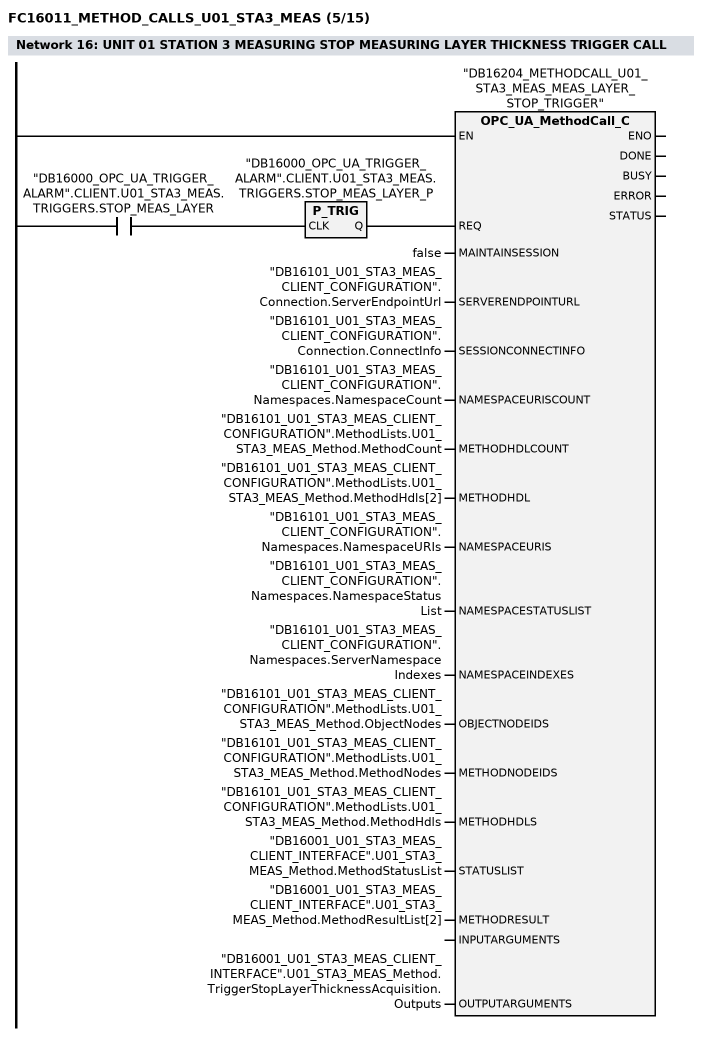
   RUNG wire#powerrail
      "DB16204_METHODCALL_U01_STA3_MEAS_MEAS_LAYER_STOP_TRIGGER".OPC_UA_MethodCall_C(REQ := wire#w1, MaintainSession := false, ServerEndpointUrl := "DB16101_U01_STA3_MEAS_CLIENT_CONFIGURATION".Connection.ServerEndpointUrl, SessionConnectInfo := "DB16101_U01_STA3_MEAS_CLIENT_CONFIGURATION".Connection.ConnectInfo, NamespaceUrisCount := "DB16101_U01_STA3_MEAS_CLIENT_CONFIGURATION".Namespaces.NamespaceCount, MethodHdlCount := "DB16101_U01_STA3_MEAS_CLIENT_CONFIGURATION".MethodLists.U01_STA3_MEAS_Method.MethodCount, MethodHdl := "DB16101_U01_STA3_MEAS_CLIENT_CONFIGURATION".MethodLists.U01_STA3_MEAS_Method.MethodHdls[2], NamespaceUris := "DB16101_U01_STA3_MEAS_CLIENT_CONFIGURATION".Namespaces.NamespaceURIs, NamespaceStatusList := "DB16101_U01_STA3_MEAS_CLIENT_CONFIGURATION".Namespaces.NamespaceStatusList, NamespaceIndexes := "DB16101_U01_STA3_MEAS_CLIENT_CONFIGURATION".Namespaces.ServerNamespaceIndexes, ObjectNodeIDs := "DB16101_U01_STA3_MEAS_CLIENT_CONFIGURATION".MethodLists.U01_STA3_MEAS_Method.ObjectNodes, MethodNodeIDs := "DB16101_U01_STA3_MEAS_CLIENT_CONFIGURATION".MethodLists.U01_STA3_MEAS_Method.MethodNodes, MethodHdls := "DB16101_U01_STA3_MEAS_CLIENT_CONFIGURATION".MethodLists.U01_STA3_MEAS_Method.MethodHdls, StatusList := "DB16001_U01_STA3_MEAS_CLIENT_INTERFACE".U01_STA3_MEAS_Method.MethodStatusList, MethodResult := "DB16001_U01_STA3_MEAS_CLIENT_INTERFACE".U01_STA3_MEAS_Method.MethodResultList[2], InputArguments :=, OutputArguments := "DB16001_U01_STA3_MEAS_CLIENT_INTERFACE".U01_STA3_MEAS_Method.TriggerStopLayerThicknessAcquisition.Outputs, Done =>, Busy =>, Error =>, Status =>)
   END_RUNG
   RUNG wire#powerrail
      Contact( "DB16000_OPC_UA_TRIGGER_ALARM".CLIENT.U01_STA3_MEAS.TRIGGERS.STOP_MEAS_LAYER )
      P_Trig( "DB16000_OPC_UA_TRIGGER_ALARM".CLIENT.U01_STA3_MEAS.TRIGGERS.STOP_MEAS_LAYER_P )
   END_RUNG wire#w1
   // the same network as SCL:
   #_w1 := "DB16000_OPC_UA_TRIGGER_ALARM".CLIENT.U01_STA3_MEAS.TRIGGERS.STOP_MEAS_LAYER AND NOT "DB16000_OPC_UA_TRIGGER_ALARM".CLIENT.U01_STA3_MEAS.TRIGGERS.STOP_MEAS_LAYER_P;   // rising edge
   "DB16000_OPC_UA_TRIGGER_ALARM".CLIENT.U01_STA3_MEAS.TRIGGERS.STOP_MEAS_LAYER_P := "DB16000_OPC_UA_TRIGGER_ALARM".CLIENT.U01_STA3_MEAS.TRIGGERS.STOP_MEAS_LAYER;
   "DB16204_METHODCALL_U01_STA3_MEAS_MEAS_LAYER_STOP_TRIGGER"(REQ := #_w1,   // OPC_UA_MethodCall_C
                           MaintainSession := false,
                           ServerEndpointUrl := "DB16101_U01_STA3_MEAS_CLIENT_CONFIGURATION".Connection.ServerEndpointUrl,
                           SessionConnectInfo := "DB16101_U01_STA3_MEAS_CLIENT_CONFIGURATION".Connection.ConnectInfo,
                           NamespaceUrisCount := "DB16101_U01_STA3_MEAS_CLIENT_CONFIGURATION".Namespaces.NamespaceCount,
                           MethodHdlCount := "DB16101_U01_STA3_MEAS_CLIENT_CONFIGURATION".MethodLists.U01_STA3_MEAS_Method.MethodCount,
                           MethodHdl := "DB16101_U01_STA3_MEAS_CLIENT_CONFIGURATION".MethodLists.U01_STA3_MEAS_Method.MethodHdls[2],
                           NamespaceUris := "DB16101_U01_STA3_MEAS_CLIENT_CONFIGURATION".Namespaces.NamespaceURIs,
                           NamespaceStatusList := "DB16101_U01_STA3_MEAS_CLIENT_CONFIGURATION".Namespaces.NamespaceStatusList,
                           NamespaceIndexes := "DB16101_U01_STA3_MEAS_CLIENT_CONFIGURATION".Namespaces.ServerNamespaceIndexes,
                           ObjectNodeIDs := "DB16101_U01_STA3_MEAS_CLIENT_CONFIGURATION".MethodLists.U01_STA3_MEAS_Method.ObjectNodes,
                           MethodNodeIDs := "DB16101_U01_STA3_MEAS_CLIENT_CONFIGURATION".MethodLists.U01_STA3_MEAS_Method.MethodNodes,
                           MethodHdls := "DB16101_U01_STA3_MEAS_CLIENT_CONFIGURATION".MethodLists.U01_STA3_MEAS_Method.MethodHdls,
                           StatusList := "DB16001_U01_STA3_MEAS_CLIENT_INTERFACE".U01_STA3_MEAS_Method.MethodStatusList,
                           MethodResult := "DB16001_U01_STA3_MEAS_CLIENT_INTERFACE".U01_STA3_MEAS_Method.MethodResultList[2],
                           OutputArguments := "DB16001_U01_STA3_MEAS_CLIENT_INTERFACE".U01_STA3_MEAS_Method.TriggerStopLayerThicknessAcquisition.Outputs);
END_REGION

REGION Network 17: UNIT 01 STATION 3 MEASURING START CALIBRATING TRIGGER CALL
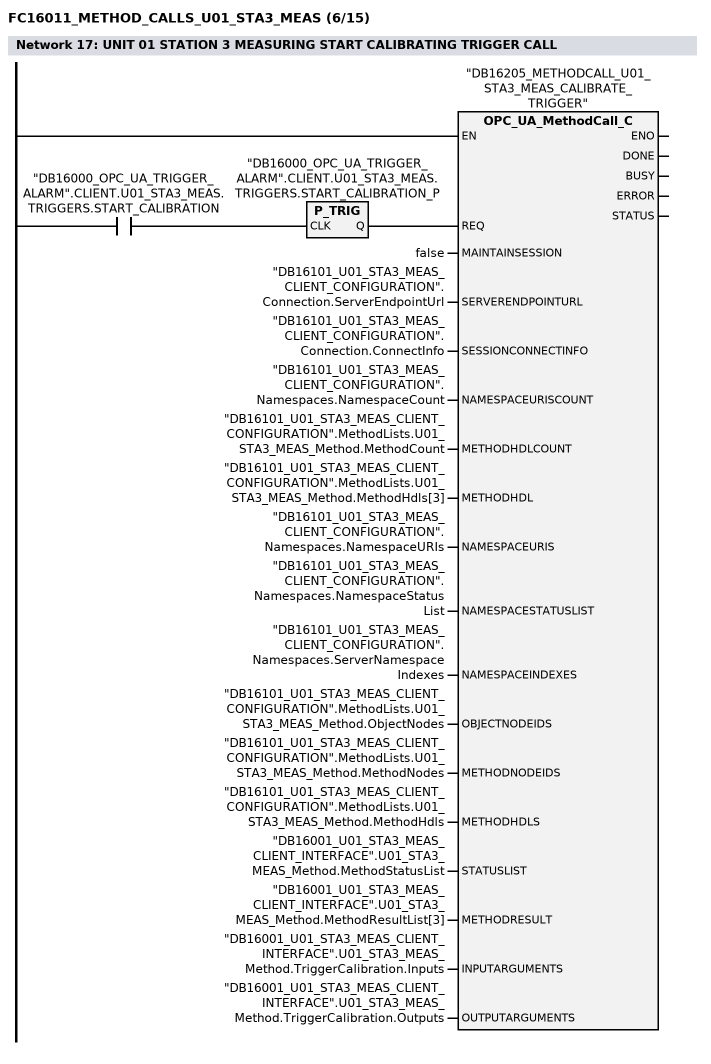
   RUNG wire#powerrail
      "DB16205_METHODCALL_U01_STA3_MEAS_CALIBRATE_TRIGGER".OPC_UA_MethodCall_C(REQ := wire#w1, MaintainSession := false, ServerEndpointUrl := "DB16101_U01_STA3_MEAS_CLIENT_CONFIGURATION".Connection.ServerEndpointUrl, SessionConnectInfo := "DB16101_U01_STA3_MEAS_CLIENT_CONFIGURATION".Connection.ConnectInfo, NamespaceUrisCount := "DB16101_U01_STA3_MEAS_CLIENT_CONFIGURATION".Namespaces.NamespaceCount, MethodHdlCount := "DB16101_U01_STA3_MEAS_CLIENT_CONFIGURATION".MethodLists.U01_STA3_MEAS_Method.MethodCount, MethodHdl := "DB16101_U01_STA3_MEAS_CLIENT_CONFIGURATION".MethodLists.U01_STA3_MEAS_Method.MethodHdls[3], NamespaceUris := "DB16101_U01_STA3_MEAS_CLIENT_CONFIGURATION".Namespaces.NamespaceURIs, NamespaceStatusList := "DB16101_U01_STA3_MEAS_CLIENT_CONFIGURATION".Namespaces.NamespaceStatusList, NamespaceIndexes := "DB16101_U01_STA3_MEAS_CLIENT_CONFIGURATION".Namespaces.ServerNamespaceIndexes, ObjectNodeIDs := "DB16101_U01_STA3_MEAS_CLIENT_CONFIGURATION".MethodLists.U01_STA3_MEAS_Method.ObjectNodes, MethodNodeIDs := "DB16101_U01_STA3_MEAS_CLIENT_CONFIGURATION".MethodLists.U01_STA3_MEAS_Method.MethodNodes, MethodHdls := "DB16101_U01_STA3_MEAS_CLIENT_CONFIGURATION".MethodLists.U01_STA3_MEAS_Method.MethodHdls, StatusList := "DB16001_U01_STA3_MEAS_CLIENT_INTERFACE".U01_STA3_MEAS_Method.MethodStatusList, MethodResult := "DB16001_U01_STA3_MEAS_CLIENT_INTERFACE".U01_STA3_MEAS_Method.MethodResultList[3], InputArguments := "DB16001_U01_STA3_MEAS_CLIENT_INTERFACE".U01_STA3_MEAS_Method.TriggerCalibration.Inputs, OutputArguments := "DB16001_U01_STA3_MEAS_CLIENT_INTERFACE".U01_STA3_MEAS_Method.TriggerCalibration.Outputs, Done =>, Busy =>, Error =>, Status =>)
   END_RUNG
   RUNG wire#powerrail
      Contact( "DB16000_OPC_UA_TRIGGER_ALARM".CLIENT.U01_STA3_MEAS.TRIGGERS.START_CALIBRATION )
      P_Trig( "DB16000_OPC_UA_TRIGGER_ALARM".CLIENT.U01_STA3_MEAS.TRIGGERS.START_CALIBRATION_P )
   END_RUNG wire#w1
   // the same network as SCL:
   #_w1 := "DB16000_OPC_UA_TRIGGER_ALARM".CLIENT.U01_STA3_MEAS.TRIGGERS.START_CALIBRATION AND NOT "DB16000_OPC_UA_TRIGGER_ALARM".CLIENT.U01_STA3_MEAS.TRIGGERS.START_CALIBRATION_P;   // rising edge
   "DB16000_OPC_UA_TRIGGER_ALARM".CLIENT.U01_STA3_MEAS.TRIGGERS.START_CALIBRATION_P := "DB16000_OPC_UA_TRIGGER_ALARM".CLIENT.U01_STA3_MEAS.TRIGGERS.START_CALIBRATION;
   "DB16205_METHODCALL_U01_STA3_MEAS_CALIBRATE_TRIGGER"(REQ := #_w1,   // OPC_UA_MethodCall_C
                           MaintainSession := false,
                           ServerEndpointUrl := "DB16101_U01_STA3_MEAS_CLIENT_CONFIGURATION".Connection.ServerEndpointUrl,
                           SessionConnectInfo := "DB16101_U01_STA3_MEAS_CLIENT_CONFIGURATION".Connection.ConnectInfo,
                           NamespaceUrisCount := "DB16101_U01_STA3_MEAS_CLIENT_CONFIGURATION".Namespaces.NamespaceCount,
                           MethodHdlCount := "DB16101_U01_STA3_MEAS_CLIENT_CONFIGURATION".MethodLists.U01_STA3_MEAS_Method.MethodCount,
                           MethodHdl := "DB16101_U01_STA3_MEAS_CLIENT_CONFIGURATION".MethodLists.U01_STA3_MEAS_Method.MethodHdls[3],
                           NamespaceUris := "DB16101_U01_STA3_MEAS_CLIENT_CONFIGURATION".Namespaces.NamespaceURIs,
                           NamespaceStatusList := "DB16101_U01_STA3_MEAS_CLIENT_CONFIGURATION".Namespaces.NamespaceStatusList,
                           NamespaceIndexes := "DB16101_U01_STA3_MEAS_CLIENT_CONFIGURATION".Namespaces.ServerNamespaceIndexes,
                           ObjectNodeIDs := "DB16101_U01_STA3_MEAS_CLIENT_CONFIGURATION".MethodLists.U01_STA3_MEAS_Method.ObjectNodes,
                           MethodNodeIDs := "DB16101_U01_STA3_MEAS_CLIENT_CONFIGURATION".MethodLists.U01_STA3_MEAS_Method.MethodNodes,
                           MethodHdls := "DB16101_U01_STA3_MEAS_CLIENT_CONFIGURATION".MethodLists.U01_STA3_MEAS_Method.MethodHdls,
                           StatusList := "DB16001_U01_STA3_MEAS_CLIENT_INTERFACE".U01_STA3_MEAS_Method.MethodStatusList,
                           MethodResult := "DB16001_U01_STA3_MEAS_CLIENT_INTERFACE".U01_STA3_MEAS_Method.MethodResultList[3],
                           InputArguments := "DB16001_U01_STA3_MEAS_CLIENT_INTERFACE".U01_STA3_MEAS_Method.TriggerCalibration.Inputs,
                           OutputArguments := "DB16001_U01_STA3_MEAS_CLIENT_INTERFACE".U01_STA3_MEAS_Method.TriggerCalibration.Outputs);
END_REGION

REGION Network 18: UNIT 01 STATION 3 MEASURING RESET PC TRIGGER CALL
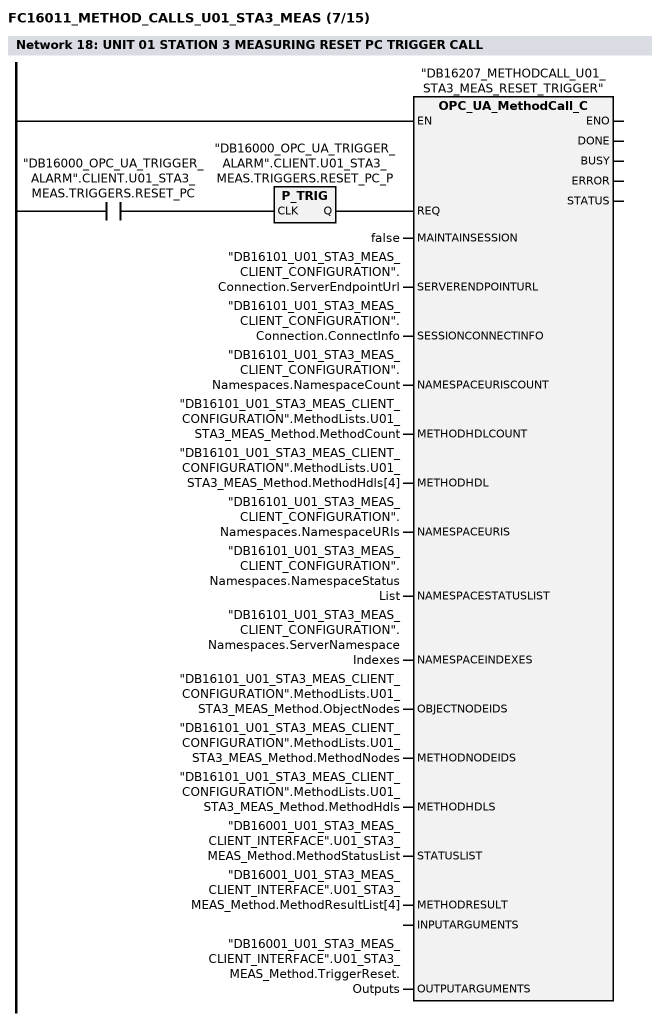
   RUNG wire#powerrail
      "DB16207_METHODCALL_U01_STA3_MEAS_RESET_TRIGGER".OPC_UA_MethodCall_C(REQ := wire#w1, MaintainSession := false, ServerEndpointUrl := "DB16101_U01_STA3_MEAS_CLIENT_CONFIGURATION".Connection.ServerEndpointUrl, SessionConnectInfo := "DB16101_U01_STA3_MEAS_CLIENT_CONFIGURATION".Connection.ConnectInfo, NamespaceUrisCount := "DB16101_U01_STA3_MEAS_CLIENT_CONFIGURATION".Namespaces.NamespaceCount, MethodHdlCount := "DB16101_U01_STA3_MEAS_CLIENT_CONFIGURATION".MethodLists.U01_STA3_MEAS_Method.MethodCount, MethodHdl := "DB16101_U01_STA3_MEAS_CLIENT_CONFIGURATION".MethodLists.U01_STA3_MEAS_Method.MethodHdls[4], NamespaceUris := "DB16101_U01_STA3_MEAS_CLIENT_CONFIGURATION".Namespaces.NamespaceURIs, NamespaceStatusList := "DB16101_U01_STA3_MEAS_CLIENT_CONFIGURATION".Namespaces.NamespaceStatusList, NamespaceIndexes := "DB16101_U01_STA3_MEAS_CLIENT_CONFIGURATION".Namespaces.ServerNamespaceIndexes, ObjectNodeIDs := "DB16101_U01_STA3_MEAS_CLIENT_CONFIGURATION".MethodLists.U01_STA3_MEAS_Method.ObjectNodes, MethodNodeIDs := "DB16101_U01_STA3_MEAS_CLIENT_CONFIGURATION".MethodLists.U01_STA3_MEAS_Method.MethodNodes, MethodHdls := "DB16101_U01_STA3_MEAS_CLIENT_CONFIGURATION".MethodLists.U01_STA3_MEAS_Method.MethodHdls, StatusList := "DB16001_U01_STA3_MEAS_CLIENT_INTERFACE".U01_STA3_MEAS_Method.MethodStatusList, MethodResult := "DB16001_U01_STA3_MEAS_CLIENT_INTERFACE".U01_STA3_MEAS_Method.MethodResultList[4], InputArguments :=, OutputArguments := "DB16001_U01_STA3_MEAS_CLIENT_INTERFACE".U01_STA3_MEAS_Method.TriggerReset.Outputs, Done =>, Busy =>, Error =>, Status =>)
   END_RUNG
   RUNG wire#powerrail
      Contact( "DB16000_OPC_UA_TRIGGER_ALARM".CLIENT.U01_STA3_MEAS.TRIGGERS.RESET_PC )
      P_Trig( "DB16000_OPC_UA_TRIGGER_ALARM".CLIENT.U01_STA3_MEAS.TRIGGERS.RESET_PC_P )
   END_RUNG wire#w1
   // the same network as SCL:
   #_w1 := "DB16000_OPC_UA_TRIGGER_ALARM".CLIENT.U01_STA3_MEAS.TRIGGERS.RESET_PC AND NOT "DB16000_OPC_UA_TRIGGER_ALARM".CLIENT.U01_STA3_MEAS.TRIGGERS.RESET_PC_P;   // rising edge
   "DB16000_OPC_UA_TRIGGER_ALARM".CLIENT.U01_STA3_MEAS.TRIGGERS.RESET_PC_P := "DB16000_OPC_UA_TRIGGER_ALARM".CLIENT.U01_STA3_MEAS.TRIGGERS.RESET_PC;
   "DB16207_METHODCALL_U01_STA3_MEAS_RESET_TRIGGER"(REQ := #_w1,   // OPC_UA_MethodCall_C
                           MaintainSession := false,
                           ServerEndpointUrl := "DB16101_U01_STA3_MEAS_CLIENT_CONFIGURATION".Connection.ServerEndpointUrl,
                           SessionConnectInfo := "DB16101_U01_STA3_MEAS_CLIENT_CONFIGURATION".Connection.ConnectInfo,
                           NamespaceUrisCount := "DB16101_U01_STA3_MEAS_CLIENT_CONFIGURATION".Namespaces.NamespaceCount,
                           MethodHdlCount := "DB16101_U01_STA3_MEAS_CLIENT_CONFIGURATION".MethodLists.U01_STA3_MEAS_Method.MethodCount,
                           MethodHdl := "DB16101_U01_STA3_MEAS_CLIENT_CONFIGURATION".MethodLists.U01_STA3_MEAS_Method.MethodHdls[4],
                           NamespaceUris := "DB16101_U01_STA3_MEAS_CLIENT_CONFIGURATION".Namespaces.NamespaceURIs,
                           NamespaceStatusList := "DB16101_U01_STA3_MEAS_CLIENT_CONFIGURATION".Namespaces.NamespaceStatusList,
                           NamespaceIndexes := "DB16101_U01_STA3_MEAS_CLIENT_CONFIGURATION".Namespaces.ServerNamespaceIndexes,
                           ObjectNodeIDs := "DB16101_U01_STA3_MEAS_CLIENT_CONFIGURATION".MethodLists.U01_STA3_MEAS_Method.ObjectNodes,
                           MethodNodeIDs := "DB16101_U01_STA3_MEAS_CLIENT_CONFIGURATION".MethodLists.U01_STA3_MEAS_Method.MethodNodes,
                           MethodHdls := "DB16101_U01_STA3_MEAS_CLIENT_CONFIGURATION".MethodLists.U01_STA3_MEAS_Method.MethodHdls,
                           StatusList := "DB16001_U01_STA3_MEAS_CLIENT_INTERFACE".U01_STA3_MEAS_Method.MethodStatusList,
                           MethodResult := "DB16001_U01_STA3_MEAS_CLIENT_INTERFACE".U01_STA3_MEAS_Method.MethodResultList[4],
                           OutputArguments := "DB16001_U01_STA3_MEAS_CLIENT_INTERFACE".U01_STA3_MEAS_Method.TriggerReset.Outputs);
END_REGION

REGION Network 19: UNIT 01 STATION 3 MEASURING READ VARIABLES TRIGGER CALL
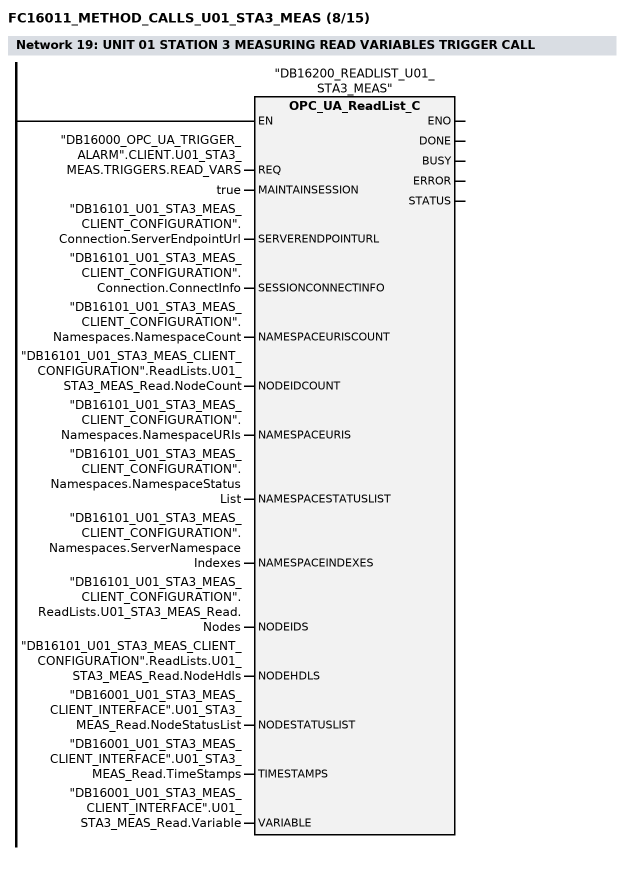
   RUNG wire#powerrail
      "DB16200_READLIST_U01_STA3_MEAS".OPC_UA_ReadList_C(REQ := "DB16000_OPC_UA_TRIGGER_ALARM".CLIENT.U01_STA3_MEAS.TRIGGERS.READ_VARS, MaintainSession := true, ServerEndpointUrl := "DB16101_U01_STA3_MEAS_CLIENT_CONFIGURATION".Connection.ServerEndpointUrl, SessionConnectInfo := "DB16101_U01_STA3_MEAS_CLIENT_CONFIGURATION".Connection.ConnectInfo, NamespaceUrisCount := "DB16101_U01_STA3_MEAS_CLIENT_CONFIGURATION".Namespaces.NamespaceCount, NodeIDCount := "DB16101_U01_STA3_MEAS_CLIENT_CONFIGURATION".ReadLists.U01_STA3_MEAS_Read.NodeCount, NamespaceUris := "DB16101_U01_STA3_MEAS_CLIENT_CONFIGURATION".Namespaces.NamespaceURIs, NamespaceStatusList := "DB16101_U01_STA3_MEAS_CLIENT_CONFIGURATION".Namespaces.NamespaceStatusList, NamespaceIndexes := "DB16101_U01_STA3_MEAS_CLIENT_CONFIGURATION".Namespaces.ServerNamespaceIndexes, NodeIDs := "DB16101_U01_STA3_MEAS_CLIENT_CONFIGURATION".ReadLists.U01_STA3_MEAS_Read.Nodes, NodeHdls := "DB16101_U01_STA3_MEAS_CLIENT_CONFIGURATION".ReadLists.U01_STA3_MEAS_Read.NodeHdls, NodeStatusList := "DB16001_U01_STA3_MEAS_CLIENT_INTERFACE".U01_STA3_MEAS_Read.NodeStatusList, Timestamps := "DB16001_U01_STA3_MEAS_CLIENT_INTERFACE".U01_STA3_MEAS_Read.TimeStamps, Variable := "DB16001_U01_STA3_MEAS_CLIENT_INTERFACE".U01_STA3_MEAS_Read.Variable, Done =>, Busy =>, Error =>, Status =>)
   END_RUNG
   // the same network as SCL:
   "DB16200_READLIST_U01_STA3_MEAS"(REQ := "DB16000_OPC_UA_TRIGGER_ALARM".CLIENT.U01_STA3_MEAS.TRIGGERS.READ_VARS,   // OPC_UA_ReadList_C
                           MaintainSession := true,
                           ServerEndpointUrl := "DB16101_U01_STA3_MEAS_CLIENT_CONFIGURATION".Connection.ServerEndpointUrl,
                           SessionConnectInfo := "DB16101_U01_STA3_MEAS_CLIENT_CONFIGURATION".Connection.ConnectInfo,
                           NamespaceUrisCount := "DB16101_U01_STA3_MEAS_CLIENT_CONFIGURATION".Namespaces.NamespaceCount,
                           NodeIDCount := "DB16101_U01_STA3_MEAS_CLIENT_CONFIGURATION".ReadLists.U01_STA3_MEAS_Read.NodeCount,
                           NamespaceUris := "DB16101_U01_STA3_MEAS_CLIENT_CONFIGURATION".Namespaces.NamespaceURIs,
                           NamespaceStatusList := "DB16101_U01_STA3_MEAS_CLIENT_CONFIGURATION".Namespaces.NamespaceStatusList,
                           NamespaceIndexes := "DB16101_U01_STA3_MEAS_CLIENT_CONFIGURATION".Namespaces.ServerNamespaceIndexes,
                           NodeIDs := "DB16101_U01_STA3_MEAS_CLIENT_CONFIGURATION".ReadLists.U01_STA3_MEAS_Read.Nodes,
                           NodeHdls := "DB16101_U01_STA3_MEAS_CLIENT_CONFIGURATION".ReadLists.U01_STA3_MEAS_Read.NodeHdls,
                           NodeStatusList := "DB16001_U01_STA3_MEAS_CLIENT_INTERFACE".U01_STA3_MEAS_Read.NodeStatusList,
                           Timestamps := "DB16001_U01_STA3_MEAS_CLIENT_INTERFACE".U01_STA3_MEAS_Read.TimeStamps,
                           Variable := "DB16001_U01_STA3_MEAS_CLIENT_INTERFACE".U01_STA3_MEAS_Read.Variable);
END_REGION

REGION Network 20: UNIT 01 NOOZLE SURFACE DISTANCE UPDATE
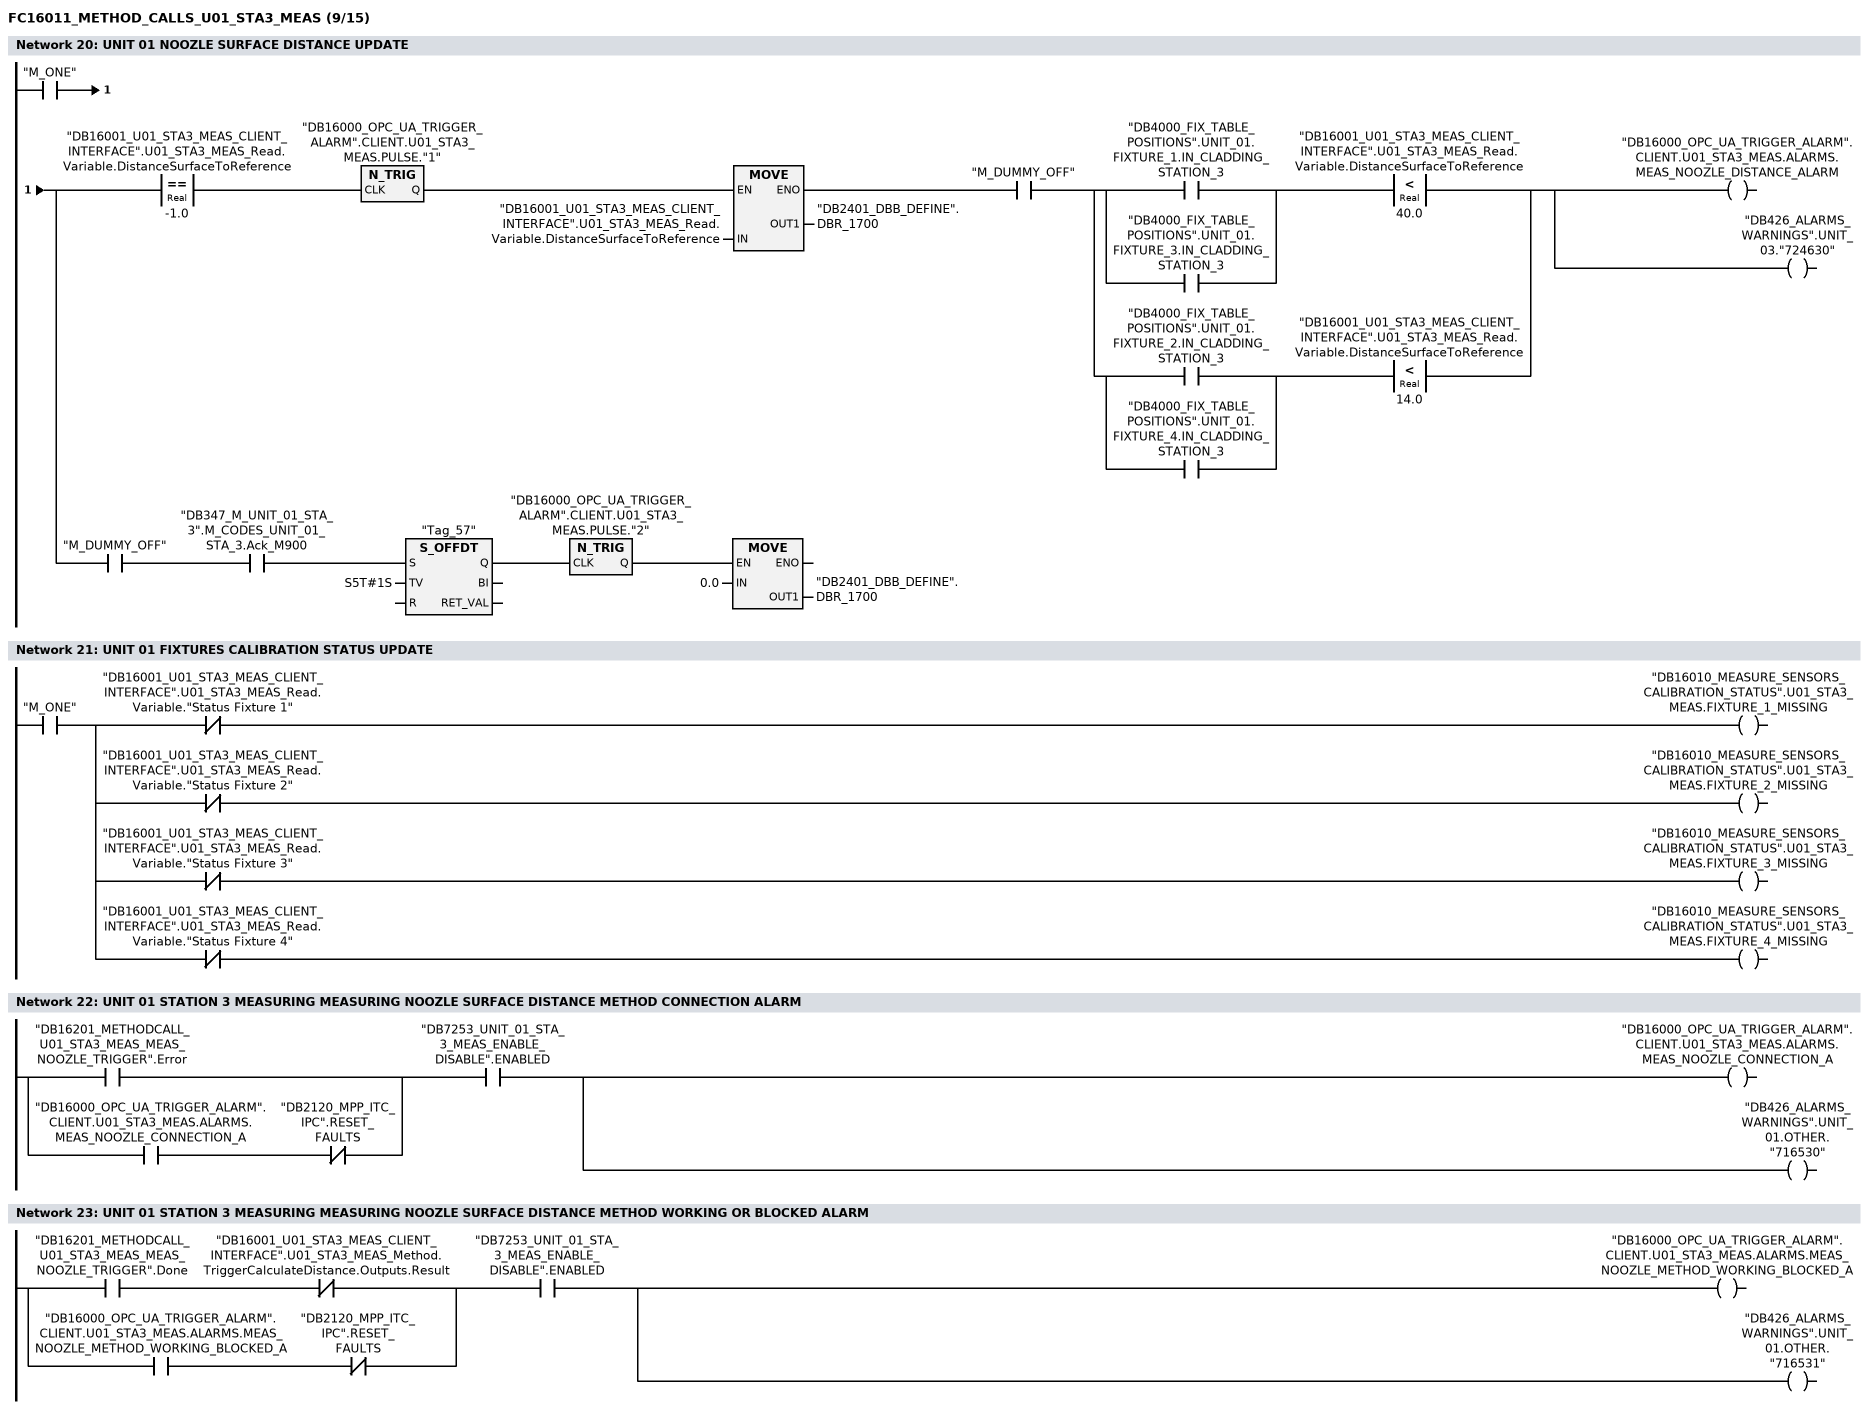
   RUNG wire#powerrail
      Contact( "M_ONE" )
      wire#w1
      { S7_Templates := "SrcType := Real" } EQ_Contact(in1 := "DB16001_U01_STA3_MEAS_CLIENT_INTERFACE".U01_STA3_MEAS_Read.Variable.DistanceSurfaceToReference, in2 := -1.0)
      N_Trig( "DB16000_OPC_UA_TRIGGER_ALARM".CLIENT.U01_STA3_MEAS.PULSE."1" )
      Move(in := "DB16001_U01_STA3_MEAS_CLIENT_INTERFACE".U01_STA3_MEAS_Read.Variable.DistanceSurfaceToReference, out1 => "DB2401_DBB_DEFINE".DBR_1700)
      Contact( "M_DUMMY_OFF" )
      wire#w2
      Contact( "DB4000_FIX_TABLE_POSITIONS".UNIT_01.FIXTURE_1.IN_CLADDING_STATION_3 )
      wire#w3
      { S7_Templates := "SrcType := Real" } LT_Contact(in1 := "DB16001_U01_STA3_MEAS_CLIENT_INTERFACE".U01_STA3_MEAS_Read.Variable.DistanceSurfaceToReference, in2 := 40.0)
      wire#w4
      Coil( "DB16000_OPC_UA_TRIGGER_ALARM".CLIENT.U01_STA3_MEAS.ALARMS.MEAS_NOOZLE_DISTANCE_ALARM )
   END_RUNG
   RUNG wire#w2
      Contact( "DB4000_FIX_TABLE_POSITIONS".UNIT_01.FIXTURE_3.IN_CLADDING_STATION_3 )
   END_RUNG wire#w3
   RUNG wire#w2
      Contact( "DB4000_FIX_TABLE_POSITIONS".UNIT_01.FIXTURE_2.IN_CLADDING_STATION_3 )
      wire#w5
      { S7_Templates := "SrcType := Real" } LT_Contact(in1 := "DB16001_U01_STA3_MEAS_CLIENT_INTERFACE".U01_STA3_MEAS_Read.Variable.DistanceSurfaceToReference, in2 := 14.0)
   END_RUNG wire#w4
   RUNG wire#w2
      Contact( "DB4000_FIX_TABLE_POSITIONS".UNIT_01.FIXTURE_4.IN_CLADDING_STATION_3 )
   END_RUNG wire#w5
   RUNG wire#w4
      Coil( "DB426_ALARMS_WARNINGS".UNIT_03."724630" )
   END_RUNG
   RUNG wire#w1
      Contact( "M_DUMMY_OFF" )
      Contact( "DB347_M_UNIT_01_STA_3".M_CODES_UNIT_01_STA_3.Ack_M900 )
      S_OFFDT(T_NO := "Tag_57", TV := S5T#1S, R :=, BI =>, RET_VAL =>)
      N_Trig( "DB16000_OPC_UA_TRIGGER_ALARM".CLIENT.U01_STA3_MEAS.PULSE."2" )
      Move(in := 0.0, out1 => "DB2401_DBB_DEFINE".DBR_1700)
   END_RUNG
   // the same network as SCL:
   #_w1 := "M_ONE" AND ("DB16001_U01_STA3_MEAS_CLIENT_INTERFACE".U01_STA3_MEAS_Read.Variable.DistanceSurfaceToReference = (-1.0));
   #_w2 := NOT #_w1 AND "DB16000_OPC_UA_TRIGGER_ALARM".CLIENT.U01_STA3_MEAS.PULSE."1";   // falling edge
   "DB16000_OPC_UA_TRIGGER_ALARM".CLIENT.U01_STA3_MEAS.PULSE."1" := #_w1;
   IF #_w2 THEN
       "DB2401_DBB_DEFINE".DBR_1700 := "DB16001_U01_STA3_MEAS_CLIENT_INTERFACE".U01_STA3_MEAS_Read.Variable.DistanceSurfaceToReference;
   END_IF;
   "DB16000_OPC_UA_TRIGGER_ALARM".CLIENT.U01_STA3_MEAS.ALARMS.MEAS_NOOZLE_DISTANCE_ALARM := #_w2 AND "M_DUMMY_OFF" AND ((("DB4000_FIX_TABLE_POSITIONS".UNIT_01.FIXTURE_1.IN_CLADDING_STATION_3 OR "DB4000_FIX_TABLE_POSITIONS".UNIT_01.FIXTURE_3.IN_CLADDING_STATION_3) AND ("DB16001_U01_STA3_MEAS_CLIENT_INTERFACE".U01_STA3_MEAS_Read.Variable.DistanceSurfaceToReference < 40.0)) OR (("DB4000_FIX_TABLE_POSITIONS".UNIT_01.FIXTURE_2.IN_CLADDING_STATION_3 OR "DB4000_FIX_TABLE_POSITIONS".UNIT_01.FIXTURE_4.IN_CLADDING_STATION_3) AND ("DB16001_U01_STA3_MEAS_CLIENT_INTERFACE".U01_STA3_MEAS_Read.Variable.DistanceSurfaceToReference < 14.0)));
   "DB426_ALARMS_WARNINGS".UNIT_03."724630" := "DB16000_OPC_UA_TRIGGER_ALARM".CLIENT.U01_STA3_MEAS.ALARMS.MEAS_NOOZLE_DISTANCE_ALARM;
   #_s5time1 := S_OFFDT(T_NO := "Tag_57",
                        S := "M_ONE" AND "M_DUMMY_OFF" AND "DB347_M_UNIT_01_STA_3".M_CODES_UNIT_01_STA_3.Ack_M900,
                        TV := S5T#1S,
                        Q => #_w3);
   #_w4 := NOT #_w3 AND "DB16000_OPC_UA_TRIGGER_ALARM".CLIENT.U01_STA3_MEAS.PULSE."2";   // falling edge
   "DB16000_OPC_UA_TRIGGER_ALARM".CLIENT.U01_STA3_MEAS.PULSE."2" := #_w3;
   IF #_w4 THEN "DB2401_DBB_DEFINE".DBR_1700 := 0.0; END_IF;
END_REGION

REGION Network 21: UNIT 01 FIXTURES CALIBRATION STATUS UPDATE
   RUNG wire#powerrail
      Contact( "M_ONE" )
      wire#w1
      I_Contact( "DB16001_U01_STA3_MEAS_CLIENT_INTERFACE".U01_STA3_MEAS_Read.Variable."Status Fixture 1" )
      Coil( "DB16010_MEASURE_SENSORS_CALIBRATION_STATUS".U01_STA3_MEAS.FIXTURE_1_MISSING )
   END_RUNG
   RUNG wire#w1
      I_Contact( "DB16001_U01_STA3_MEAS_CLIENT_INTERFACE".U01_STA3_MEAS_Read.Variable."Status Fixture 2" )
      Coil( "DB16010_MEASURE_SENSORS_CALIBRATION_STATUS".U01_STA3_MEAS.FIXTURE_2_MISSING )
   END_RUNG
   RUNG wire#w1
      I_Contact( "DB16001_U01_STA3_MEAS_CLIENT_INTERFACE".U01_STA3_MEAS_Read.Variable."Status Fixture 3" )
      Coil( "DB16010_MEASURE_SENSORS_CALIBRATION_STATUS".U01_STA3_MEAS.FIXTURE_3_MISSING )
   END_RUNG
   RUNG wire#w1
      I_Contact( "DB16001_U01_STA3_MEAS_CLIENT_INTERFACE".U01_STA3_MEAS_Read.Variable."Status Fixture 4" )
      Coil( "DB16010_MEASURE_SENSORS_CALIBRATION_STATUS".U01_STA3_MEAS.FIXTURE_4_MISSING )
   END_RUNG
   // the same network as SCL:
   "DB16010_MEASURE_SENSORS_CALIBRATION_STATUS".U01_STA3_MEAS.FIXTURE_1_MISSING := "M_ONE" AND NOT "DB16001_U01_STA3_MEAS_CLIENT_INTERFACE".U01_STA3_MEAS_Read.Variable."Status Fixture 1";
   "DB16010_MEASURE_SENSORS_CALIBRATION_STATUS".U01_STA3_MEAS.FIXTURE_2_MISSING := "M_ONE" AND NOT "DB16001_U01_STA3_MEAS_CLIENT_INTERFACE".U01_STA3_MEAS_Read.Variable."Status Fixture 2";
   "DB16010_MEASURE_SENSORS_CALIBRATION_STATUS".U01_STA3_MEAS.FIXTURE_3_MISSING := "M_ONE" AND NOT "DB16001_U01_STA3_MEAS_CLIENT_INTERFACE".U01_STA3_MEAS_Read.Variable."Status Fixture 3";
   "DB16010_MEASURE_SENSORS_CALIBRATION_STATUS".U01_STA3_MEAS.FIXTURE_4_MISSING := "M_ONE" AND NOT "DB16001_U01_STA3_MEAS_CLIENT_INTERFACE".U01_STA3_MEAS_Read.Variable."Status Fixture 4";
END_REGION

REGION Network 22: UNIT 01 STATION 3 MEASURING MEASURING NOOZLE SURFACE DISTANCE METHOD CONNECTION ALARM
   RUNG wire#powerrail
      Contact( "DB16201_METHODCALL_U01_STA3_MEAS_MEAS_NOOZLE_TRIGGER".Error )
      wire#w1
      Contact( "DB7253_UNIT_01_STA_3_MEAS_ENABLE_DISABLE".ENABLED )
      wire#w2
      Coil( "DB16000_OPC_UA_TRIGGER_ALARM".CLIENT.U01_STA3_MEAS.ALARMS.MEAS_NOOZLE_CONNECTION_A )
   END_RUNG
   RUNG wire#powerrail
      Contact( "DB16000_OPC_UA_TRIGGER_ALARM".CLIENT.U01_STA3_MEAS.ALARMS.MEAS_NOOZLE_CONNECTION_A )
      I_Contact( "DB2120_MPP_ITC_IPC".RESET_FAULTS )
   END_RUNG wire#w1
   RUNG wire#w2
      Coil( "DB426_ALARMS_WARNINGS".UNIT_01.OTHER."716530" )
   END_RUNG
   // the same network as SCL:
   "DB16000_OPC_UA_TRIGGER_ALARM".CLIENT.U01_STA3_MEAS.ALARMS.MEAS_NOOZLE_CONNECTION_A := ("DB16201_METHODCALL_U01_STA3_MEAS_MEAS_NOOZLE_TRIGGER".Error OR ("DB16000_OPC_UA_TRIGGER_ALARM".CLIENT.U01_STA3_MEAS.ALARMS.MEAS_NOOZLE_CONNECTION_A AND NOT "DB2120_MPP_ITC_IPC".RESET_FAULTS)) AND "DB7253_UNIT_01_STA_3_MEAS_ENABLE_DISABLE".ENABLED;
   "DB426_ALARMS_WARNINGS".UNIT_01.OTHER."716530" := "DB16000_OPC_UA_TRIGGER_ALARM".CLIENT.U01_STA3_MEAS.ALARMS.MEAS_NOOZLE_CONNECTION_A;
END_REGION

REGION Network 23: UNIT 01 STATION 3 MEASURING MEASURING NOOZLE SURFACE DISTANCE METHOD WORKING OR BLOCKED ALARM
   RUNG wire#powerrail
      Contact( "DB16201_METHODCALL_U01_STA3_MEAS_MEAS_NOOZLE_TRIGGER".Done )
      I_Contact( "DB16001_U01_STA3_MEAS_CLIENT_INTERFACE".U01_STA3_MEAS_Method.TriggerCalculateDistance.Outputs.Result )
      wire#w1
      Contact( "DB7253_UNIT_01_STA_3_MEAS_ENABLE_DISABLE".ENABLED )
      wire#w2
      Coil( "DB16000_OPC_UA_TRIGGER_ALARM".CLIENT.U01_STA3_MEAS.ALARMS.MEAS_NOOZLE_METHOD_WORKING_BLOCKED_A )
   END_RUNG
   RUNG wire#powerrail
      Contact( "DB16000_OPC_UA_TRIGGER_ALARM".CLIENT.U01_STA3_MEAS.ALARMS.MEAS_NOOZLE_METHOD_WORKING_BLOCKED_A )
      I_Contact( "DB2120_MPP_ITC_IPC".RESET_FAULTS )
   END_RUNG wire#w1
   RUNG wire#w2
      Coil( "DB426_ALARMS_WARNINGS".UNIT_01.OTHER."716531" )
   END_RUNG
   // the same network as SCL:
   "DB16000_OPC_UA_TRIGGER_ALARM".CLIENT.U01_STA3_MEAS.ALARMS.MEAS_NOOZLE_METHOD_WORKING_BLOCKED_A := (("DB16201_METHODCALL_U01_STA3_MEAS_MEAS_NOOZLE_TRIGGER".Done AND NOT "DB16001_U01_STA3_MEAS_CLIENT_INTERFACE".U01_STA3_MEAS_Method.TriggerCalculateDistance.Outputs.Result) OR ("DB16000_OPC_UA_TRIGGER_ALARM".CLIENT.U01_STA3_MEAS.ALARMS.MEAS_NOOZLE_METHOD_WORKING_BLOCKED_A AND NOT "DB2120_MPP_ITC_IPC".RESET_FAULTS)) AND "DB7253_UNIT_01_STA_3_MEAS_ENABLE_DISABLE".ENABLED;
   "DB426_ALARMS_WARNINGS".UNIT_01.OTHER."716531" := "DB16000_OPC_UA_TRIGGER_ALARM".CLIENT.U01_STA3_MEAS.ALARMS.MEAS_NOOZLE_METHOD_WORKING_BLOCKED_A;
END_REGION

REGION Network 24: UNIT 01 STATION 3 MEASURING START MEASURING LAYER THICKNESS METHOD CONNECTION ALARM
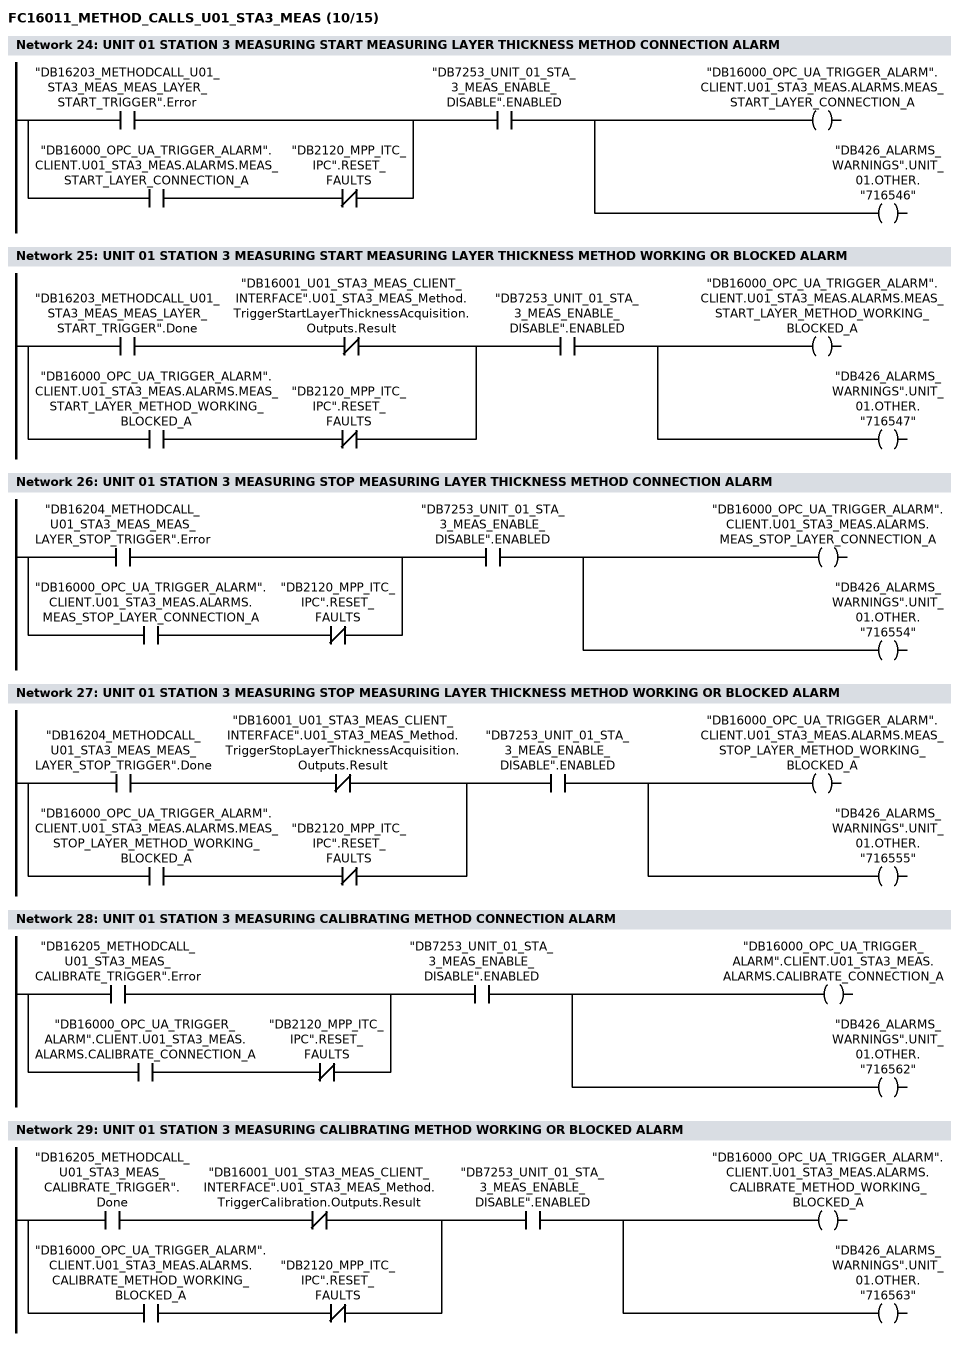
   RUNG wire#powerrail
      Contact( "DB16203_METHODCALL_U01_STA3_MEAS_MEAS_LAYER_START_TRIGGER".Error )
      wire#w1
      Contact( "DB7253_UNIT_01_STA_3_MEAS_ENABLE_DISABLE".ENABLED )
      wire#w2
      Coil( "DB16000_OPC_UA_TRIGGER_ALARM".CLIENT.U01_STA3_MEAS.ALARMS.MEAS_START_LAYER_CONNECTION_A )
   END_RUNG
   RUNG wire#powerrail
      Contact( "DB16000_OPC_UA_TRIGGER_ALARM".CLIENT.U01_STA3_MEAS.ALARMS.MEAS_START_LAYER_CONNECTION_A )
      I_Contact( "DB2120_MPP_ITC_IPC".RESET_FAULTS )
   END_RUNG wire#w1
   RUNG wire#w2
      Coil( "DB426_ALARMS_WARNINGS".UNIT_01.OTHER."716546" )
   END_RUNG
   // the same network as SCL:
   "DB16000_OPC_UA_TRIGGER_ALARM".CLIENT.U01_STA3_MEAS.ALARMS.MEAS_START_LAYER_CONNECTION_A := ("DB16203_METHODCALL_U01_STA3_MEAS_MEAS_LAYER_START_TRIGGER".Error OR ("DB16000_OPC_UA_TRIGGER_ALARM".CLIENT.U01_STA3_MEAS.ALARMS.MEAS_START_LAYER_CONNECTION_A AND NOT "DB2120_MPP_ITC_IPC".RESET_FAULTS)) AND "DB7253_UNIT_01_STA_3_MEAS_ENABLE_DISABLE".ENABLED;
   "DB426_ALARMS_WARNINGS".UNIT_01.OTHER."716546" := "DB16000_OPC_UA_TRIGGER_ALARM".CLIENT.U01_STA3_MEAS.ALARMS.MEAS_START_LAYER_CONNECTION_A;
END_REGION

REGION Network 25: UNIT 01 STATION 3 MEASURING START MEASURING LAYER THICKNESS METHOD WORKING OR BLOCKED ALARM
   RUNG wire#powerrail
      Contact( "DB16203_METHODCALL_U01_STA3_MEAS_MEAS_LAYER_START_TRIGGER".Done )
      I_Contact( "DB16001_U01_STA3_MEAS_CLIENT_INTERFACE".U01_STA3_MEAS_Method.TriggerStartLayerThicknessAcquisition.Outputs.Result )
      wire#w1
      Contact( "DB7253_UNIT_01_STA_3_MEAS_ENABLE_DISABLE".ENABLED )
      wire#w2
      Coil( "DB16000_OPC_UA_TRIGGER_ALARM".CLIENT.U01_STA3_MEAS.ALARMS.MEAS_START_LAYER_METHOD_WORKING_BLOCKED_A )
   END_RUNG
   RUNG wire#powerrail
      Contact( "DB16000_OPC_UA_TRIGGER_ALARM".CLIENT.U01_STA3_MEAS.ALARMS.MEAS_START_LAYER_METHOD_WORKING_BLOCKED_A )
      I_Contact( "DB2120_MPP_ITC_IPC".RESET_FAULTS )
   END_RUNG wire#w1
   RUNG wire#w2
      Coil( "DB426_ALARMS_WARNINGS".UNIT_01.OTHER."716547" )
   END_RUNG
   // the same network as SCL:
   "DB16000_OPC_UA_TRIGGER_ALARM".CLIENT.U01_STA3_MEAS.ALARMS.MEAS_START_LAYER_METHOD_WORKING_BLOCKED_A := (("DB16203_METHODCALL_U01_STA3_MEAS_MEAS_LAYER_START_TRIGGER".Done AND NOT "DB16001_U01_STA3_MEAS_CLIENT_INTERFACE".U01_STA3_MEAS_Method.TriggerStartLayerThicknessAcquisition.Outputs.Result) OR ("DB16000_OPC_UA_TRIGGER_ALARM".CLIENT.U01_STA3_MEAS.ALARMS.MEAS_START_LAYER_METHOD_WORKING_BLOCKED_A AND NOT "DB2120_MPP_ITC_IPC".RESET_FAULTS)) AND "DB7253_UNIT_01_STA_3_MEAS_ENABLE_DISABLE".ENABLED;
   "DB426_ALARMS_WARNINGS".UNIT_01.OTHER."716547" := "DB16000_OPC_UA_TRIGGER_ALARM".CLIENT.U01_STA3_MEAS.ALARMS.MEAS_START_LAYER_METHOD_WORKING_BLOCKED_A;
END_REGION

REGION Network 26: UNIT 01 STATION 3 MEASURING STOP MEASURING LAYER THICKNESS METHOD CONNECTION ALARM
   RUNG wire#powerrail
      Contact( "DB16204_METHODCALL_U01_STA3_MEAS_MEAS_LAYER_STOP_TRIGGER".Error )
      wire#w1
      Contact( "DB7253_UNIT_01_STA_3_MEAS_ENABLE_DISABLE".ENABLED )
      wire#w2
      Coil( "DB16000_OPC_UA_TRIGGER_ALARM".CLIENT.U01_STA3_MEAS.ALARMS.MEAS_STOP_LAYER_CONNECTION_A )
   END_RUNG
   RUNG wire#powerrail
      Contact( "DB16000_OPC_UA_TRIGGER_ALARM".CLIENT.U01_STA3_MEAS.ALARMS.MEAS_STOP_LAYER_CONNECTION_A )
      I_Contact( "DB2120_MPP_ITC_IPC".RESET_FAULTS )
   END_RUNG wire#w1
   RUNG wire#w2
      Coil( "DB426_ALARMS_WARNINGS".UNIT_01.OTHER."716554" )
   END_RUNG
   // the same network as SCL:
   "DB16000_OPC_UA_TRIGGER_ALARM".CLIENT.U01_STA3_MEAS.ALARMS.MEAS_STOP_LAYER_CONNECTION_A := ("DB16204_METHODCALL_U01_STA3_MEAS_MEAS_LAYER_STOP_TRIGGER".Error OR ("DB16000_OPC_UA_TRIGGER_ALARM".CLIENT.U01_STA3_MEAS.ALARMS.MEAS_STOP_LAYER_CONNECTION_A AND NOT "DB2120_MPP_ITC_IPC".RESET_FAULTS)) AND "DB7253_UNIT_01_STA_3_MEAS_ENABLE_DISABLE".ENABLED;
   "DB426_ALARMS_WARNINGS".UNIT_01.OTHER."716554" := "DB16000_OPC_UA_TRIGGER_ALARM".CLIENT.U01_STA3_MEAS.ALARMS.MEAS_STOP_LAYER_CONNECTION_A;
END_REGION

REGION Network 27: UNIT 01 STATION 3 MEASURING STOP MEASURING LAYER THICKNESS METHOD WORKING OR BLOCKED ALARM
   RUNG wire#powerrail
      Contact( "DB16204_METHODCALL_U01_STA3_MEAS_MEAS_LAYER_STOP_TRIGGER".Done )
      I_Contact( "DB16001_U01_STA3_MEAS_CLIENT_INTERFACE".U01_STA3_MEAS_Method.TriggerStopLayerThicknessAcquisition.Outputs.Result )
      wire#w1
      Contact( "DB7253_UNIT_01_STA_3_MEAS_ENABLE_DISABLE".ENABLED )
      wire#w2
      Coil( "DB16000_OPC_UA_TRIGGER_ALARM".CLIENT.U01_STA3_MEAS.ALARMS.MEAS_STOP_LAYER_METHOD_WORKING_BLOCKED_A )
   END_RUNG
   RUNG wire#powerrail
      Contact( "DB16000_OPC_UA_TRIGGER_ALARM".CLIENT.U01_STA3_MEAS.ALARMS.MEAS_STOP_LAYER_METHOD_WORKING_BLOCKED_A )
      I_Contact( "DB2120_MPP_ITC_IPC".RESET_FAULTS )
   END_RUNG wire#w1
   RUNG wire#w2
      Coil( "DB426_ALARMS_WARNINGS".UNIT_01.OTHER."716555" )
   END_RUNG
   // the same network as SCL:
   "DB16000_OPC_UA_TRIGGER_ALARM".CLIENT.U01_STA3_MEAS.ALARMS.MEAS_STOP_LAYER_METHOD_WORKING_BLOCKED_A := (("DB16204_METHODCALL_U01_STA3_MEAS_MEAS_LAYER_STOP_TRIGGER".Done AND NOT "DB16001_U01_STA3_MEAS_CLIENT_INTERFACE".U01_STA3_MEAS_Method.TriggerStopLayerThicknessAcquisition.Outputs.Result) OR ("DB16000_OPC_UA_TRIGGER_ALARM".CLIENT.U01_STA3_MEAS.ALARMS.MEAS_STOP_LAYER_METHOD_WORKING_BLOCKED_A AND NOT "DB2120_MPP_ITC_IPC".RESET_FAULTS)) AND "DB7253_UNIT_01_STA_3_MEAS_ENABLE_DISABLE".ENABLED;
   "DB426_ALARMS_WARNINGS".UNIT_01.OTHER."716555" := "DB16000_OPC_UA_TRIGGER_ALARM".CLIENT.U01_STA3_MEAS.ALARMS.MEAS_STOP_LAYER_METHOD_WORKING_BLOCKED_A;
END_REGION

REGION Network 28: UNIT 01 STATION 3 MEASURING CALIBRATING METHOD CONNECTION ALARM
   RUNG wire#powerrail
      Contact( "DB16205_METHODCALL_U01_STA3_MEAS_CALIBRATE_TRIGGER".Error )
      wire#w1
      Contact( "DB7253_UNIT_01_STA_3_MEAS_ENABLE_DISABLE".ENABLED )
      wire#w2
      Coil( "DB16000_OPC_UA_TRIGGER_ALARM".CLIENT.U01_STA3_MEAS.ALARMS.CALIBRATE_CONNECTION_A )
   END_RUNG
   RUNG wire#powerrail
      Contact( "DB16000_OPC_UA_TRIGGER_ALARM".CLIENT.U01_STA3_MEAS.ALARMS.CALIBRATE_CONNECTION_A )
      I_Contact( "DB2120_MPP_ITC_IPC".RESET_FAULTS )
   END_RUNG wire#w1
   RUNG wire#w2
      Coil( "DB426_ALARMS_WARNINGS".UNIT_01.OTHER."716562" )
   END_RUNG
   // the same network as SCL:
   "DB16000_OPC_UA_TRIGGER_ALARM".CLIENT.U01_STA3_MEAS.ALARMS.CALIBRATE_CONNECTION_A := ("DB16205_METHODCALL_U01_STA3_MEAS_CALIBRATE_TRIGGER".Error OR ("DB16000_OPC_UA_TRIGGER_ALARM".CLIENT.U01_STA3_MEAS.ALARMS.CALIBRATE_CONNECTION_A AND NOT "DB2120_MPP_ITC_IPC".RESET_FAULTS)) AND "DB7253_UNIT_01_STA_3_MEAS_ENABLE_DISABLE".ENABLED;
   "DB426_ALARMS_WARNINGS".UNIT_01.OTHER."716562" := "DB16000_OPC_UA_TRIGGER_ALARM".CLIENT.U01_STA3_MEAS.ALARMS.CALIBRATE_CONNECTION_A;
END_REGION

REGION Network 29: UNIT 01 STATION 3 MEASURING CALIBRATING METHOD WORKING OR BLOCKED ALARM
   RUNG wire#powerrail
      Contact( "DB16205_METHODCALL_U01_STA3_MEAS_CALIBRATE_TRIGGER".Done )
      I_Contact( "DB16001_U01_STA3_MEAS_CLIENT_INTERFACE".U01_STA3_MEAS_Method.TriggerCalibration.Outputs.Result )
      wire#w1
      Contact( "DB7253_UNIT_01_STA_3_MEAS_ENABLE_DISABLE".ENABLED )
      wire#w2
      Coil( "DB16000_OPC_UA_TRIGGER_ALARM".CLIENT.U01_STA3_MEAS.ALARMS.CALIBRATE_METHOD_WORKING_BLOCKED_A )
   END_RUNG
   RUNG wire#powerrail
      Contact( "DB16000_OPC_UA_TRIGGER_ALARM".CLIENT.U01_STA3_MEAS.ALARMS.CALIBRATE_METHOD_WORKING_BLOCKED_A )
      I_Contact( "DB2120_MPP_ITC_IPC".RESET_FAULTS )
   END_RUNG wire#w1
   RUNG wire#w2
      Coil( "DB426_ALARMS_WARNINGS".UNIT_01.OTHER."716563" )
   END_RUNG
   // the same network as SCL:
   "DB16000_OPC_UA_TRIGGER_ALARM".CLIENT.U01_STA3_MEAS.ALARMS.CALIBRATE_METHOD_WORKING_BLOCKED_A := (("DB16205_METHODCALL_U01_STA3_MEAS_CALIBRATE_TRIGGER".Done AND NOT "DB16001_U01_STA3_MEAS_CLIENT_INTERFACE".U01_STA3_MEAS_Method.TriggerCalibration.Outputs.Result) OR ("DB16000_OPC_UA_TRIGGER_ALARM".CLIENT.U01_STA3_MEAS.ALARMS.CALIBRATE_METHOD_WORKING_BLOCKED_A AND NOT "DB2120_MPP_ITC_IPC".RESET_FAULTS)) AND "DB7253_UNIT_01_STA_3_MEAS_ENABLE_DISABLE".ENABLED;
   "DB426_ALARMS_WARNINGS".UNIT_01.OTHER."716563" := "DB16000_OPC_UA_TRIGGER_ALARM".CLIENT.U01_STA3_MEAS.ALARMS.CALIBRATE_METHOD_WORKING_BLOCKED_A;
END_REGION

REGION Network 30: UNIT 01 STATION 3 MEASURING RESET METHOD CONNECTION ALARM
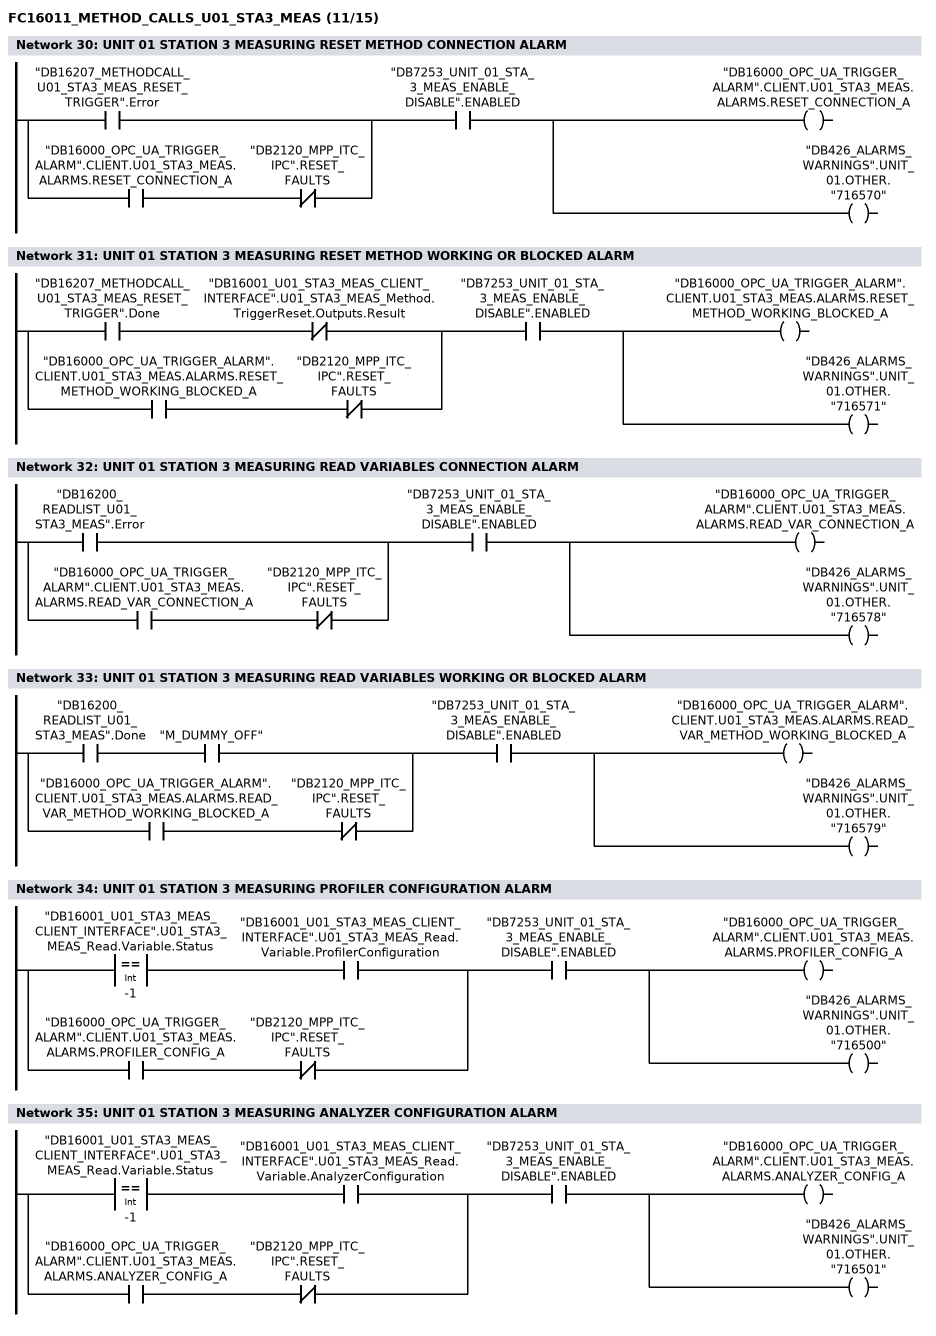
   RUNG wire#powerrail
      Contact( "DB16207_METHODCALL_U01_STA3_MEAS_RESET_TRIGGER".Error )
      wire#w1
      Contact( "DB7253_UNIT_01_STA_3_MEAS_ENABLE_DISABLE".ENABLED )
      wire#w2
      Coil( "DB16000_OPC_UA_TRIGGER_ALARM".CLIENT.U01_STA3_MEAS.ALARMS.RESET_CONNECTION_A )
   END_RUNG
   RUNG wire#powerrail
      Contact( "DB16000_OPC_UA_TRIGGER_ALARM".CLIENT.U01_STA3_MEAS.ALARMS.RESET_CONNECTION_A )
      I_Contact( "DB2120_MPP_ITC_IPC".RESET_FAULTS )
   END_RUNG wire#w1
   RUNG wire#w2
      Coil( "DB426_ALARMS_WARNINGS".UNIT_01.OTHER."716570" )
   END_RUNG
   // the same network as SCL:
   "DB16000_OPC_UA_TRIGGER_ALARM".CLIENT.U01_STA3_MEAS.ALARMS.RESET_CONNECTION_A := ("DB16207_METHODCALL_U01_STA3_MEAS_RESET_TRIGGER".Error OR ("DB16000_OPC_UA_TRIGGER_ALARM".CLIENT.U01_STA3_MEAS.ALARMS.RESET_CONNECTION_A AND NOT "DB2120_MPP_ITC_IPC".RESET_FAULTS)) AND "DB7253_UNIT_01_STA_3_MEAS_ENABLE_DISABLE".ENABLED;
   "DB426_ALARMS_WARNINGS".UNIT_01.OTHER."716570" := "DB16000_OPC_UA_TRIGGER_ALARM".CLIENT.U01_STA3_MEAS.ALARMS.RESET_CONNECTION_A;
END_REGION

REGION Network 31: UNIT 01 STATION 3 MEASURING RESET METHOD WORKING OR BLOCKED ALARM
   RUNG wire#powerrail
      Contact( "DB16207_METHODCALL_U01_STA3_MEAS_RESET_TRIGGER".Done )
      I_Contact( "DB16001_U01_STA3_MEAS_CLIENT_INTERFACE".U01_STA3_MEAS_Method.TriggerReset.Outputs.Result )
      wire#w1
      Contact( "DB7253_UNIT_01_STA_3_MEAS_ENABLE_DISABLE".ENABLED )
      wire#w2
      Coil( "DB16000_OPC_UA_TRIGGER_ALARM".CLIENT.U01_STA3_MEAS.ALARMS.RESET_METHOD_WORKING_BLOCKED_A )
   END_RUNG
   RUNG wire#powerrail
      Contact( "DB16000_OPC_UA_TRIGGER_ALARM".CLIENT.U01_STA3_MEAS.ALARMS.RESET_METHOD_WORKING_BLOCKED_A )
      I_Contact( "DB2120_MPP_ITC_IPC".RESET_FAULTS )
   END_RUNG wire#w1
   RUNG wire#w2
      Coil( "DB426_ALARMS_WARNINGS".UNIT_01.OTHER."716571" )
   END_RUNG
   // the same network as SCL:
   "DB16000_OPC_UA_TRIGGER_ALARM".CLIENT.U01_STA3_MEAS.ALARMS.RESET_METHOD_WORKING_BLOCKED_A := (("DB16207_METHODCALL_U01_STA3_MEAS_RESET_TRIGGER".Done AND NOT "DB16001_U01_STA3_MEAS_CLIENT_INTERFACE".U01_STA3_MEAS_Method.TriggerReset.Outputs.Result) OR ("DB16000_OPC_UA_TRIGGER_ALARM".CLIENT.U01_STA3_MEAS.ALARMS.RESET_METHOD_WORKING_BLOCKED_A AND NOT "DB2120_MPP_ITC_IPC".RESET_FAULTS)) AND "DB7253_UNIT_01_STA_3_MEAS_ENABLE_DISABLE".ENABLED;
   "DB426_ALARMS_WARNINGS".UNIT_01.OTHER."716571" := "DB16000_OPC_UA_TRIGGER_ALARM".CLIENT.U01_STA3_MEAS.ALARMS.RESET_METHOD_WORKING_BLOCKED_A;
END_REGION

REGION Network 32: UNIT 01 STATION 3 MEASURING READ VARIABLES CONNECTION ALARM
   RUNG wire#powerrail
      Contact( "DB16200_READLIST_U01_STA3_MEAS".Error )
      wire#w1
      Contact( "DB7253_UNIT_01_STA_3_MEAS_ENABLE_DISABLE".ENABLED )
      wire#w2
      Coil( "DB16000_OPC_UA_TRIGGER_ALARM".CLIENT.U01_STA3_MEAS.ALARMS.READ_VAR_CONNECTION_A )
   END_RUNG
   RUNG wire#powerrail
      Contact( "DB16000_OPC_UA_TRIGGER_ALARM".CLIENT.U01_STA3_MEAS.ALARMS.READ_VAR_CONNECTION_A )
      I_Contact( "DB2120_MPP_ITC_IPC".RESET_FAULTS )
   END_RUNG wire#w1
   RUNG wire#w2
      Coil( "DB426_ALARMS_WARNINGS".UNIT_01.OTHER."716578" )
   END_RUNG
   // the same network as SCL:
   "DB16000_OPC_UA_TRIGGER_ALARM".CLIENT.U01_STA3_MEAS.ALARMS.READ_VAR_CONNECTION_A := ("DB16200_READLIST_U01_STA3_MEAS".Error OR ("DB16000_OPC_UA_TRIGGER_ALARM".CLIENT.U01_STA3_MEAS.ALARMS.READ_VAR_CONNECTION_A AND NOT "DB2120_MPP_ITC_IPC".RESET_FAULTS)) AND "DB7253_UNIT_01_STA_3_MEAS_ENABLE_DISABLE".ENABLED;
   "DB426_ALARMS_WARNINGS".UNIT_01.OTHER."716578" := "DB16000_OPC_UA_TRIGGER_ALARM".CLIENT.U01_STA3_MEAS.ALARMS.READ_VAR_CONNECTION_A;
END_REGION

REGION Network 33: UNIT 01 STATION 3 MEASURING READ VARIABLES WORKING OR BLOCKED ALARM
   RUNG wire#powerrail
      Contact( "DB16200_READLIST_U01_STA3_MEAS".Done )
      Contact( "M_DUMMY_OFF" )
      wire#w1
      Contact( "DB7253_UNIT_01_STA_3_MEAS_ENABLE_DISABLE".ENABLED )
      wire#w2
      Coil( "DB16000_OPC_UA_TRIGGER_ALARM".CLIENT.U01_STA3_MEAS.ALARMS.READ_VAR_METHOD_WORKING_BLOCKED_A )
   END_RUNG
   RUNG wire#powerrail
      Contact( "DB16000_OPC_UA_TRIGGER_ALARM".CLIENT.U01_STA3_MEAS.ALARMS.READ_VAR_METHOD_WORKING_BLOCKED_A )
      I_Contact( "DB2120_MPP_ITC_IPC".RESET_FAULTS )
   END_RUNG wire#w1
   RUNG wire#w2
      Coil( "DB426_ALARMS_WARNINGS".UNIT_01.OTHER."716579" )
   END_RUNG
   // the same network as SCL:
   "DB16000_OPC_UA_TRIGGER_ALARM".CLIENT.U01_STA3_MEAS.ALARMS.READ_VAR_METHOD_WORKING_BLOCKED_A := (("DB16200_READLIST_U01_STA3_MEAS".Done AND "M_DUMMY_OFF") OR ("DB16000_OPC_UA_TRIGGER_ALARM".CLIENT.U01_STA3_MEAS.ALARMS.READ_VAR_METHOD_WORKING_BLOCKED_A AND NOT "DB2120_MPP_ITC_IPC".RESET_FAULTS)) AND "DB7253_UNIT_01_STA_3_MEAS_ENABLE_DISABLE".ENABLED;
   "DB426_ALARMS_WARNINGS".UNIT_01.OTHER."716579" := "DB16000_OPC_UA_TRIGGER_ALARM".CLIENT.U01_STA3_MEAS.ALARMS.READ_VAR_METHOD_WORKING_BLOCKED_A;
END_REGION

REGION Network 34: UNIT 01 STATION 3 MEASURING PROFILER CONFIGURATION ALARM
   RUNG wire#powerrail
      { S7_Templates := "SrcType := Int" } EQ_Contact(in1 := "DB16001_U01_STA3_MEAS_CLIENT_INTERFACE".U01_STA3_MEAS_Read.Variable.Status, in2 := -1)
      Contact( "DB16001_U01_STA3_MEAS_CLIENT_INTERFACE".U01_STA3_MEAS_Read.Variable.ProfilerConfiguration )
      wire#w1
      Contact( "DB7253_UNIT_01_STA_3_MEAS_ENABLE_DISABLE".ENABLED )
      wire#w2
      Coil( "DB16000_OPC_UA_TRIGGER_ALARM".CLIENT.U01_STA3_MEAS.ALARMS.PROFILER_CONFIG_A )
   END_RUNG
   RUNG wire#powerrail
      Contact( "DB16000_OPC_UA_TRIGGER_ALARM".CLIENT.U01_STA3_MEAS.ALARMS.PROFILER_CONFIG_A )
      I_Contact( "DB2120_MPP_ITC_IPC".RESET_FAULTS )
   END_RUNG wire#w1
   RUNG wire#w2
      Coil( "DB426_ALARMS_WARNINGS".UNIT_01.OTHER."716500" )
   END_RUNG
   // the same network as SCL:
   "DB16000_OPC_UA_TRIGGER_ALARM".CLIENT.U01_STA3_MEAS.ALARMS.PROFILER_CONFIG_A := ((("DB16001_U01_STA3_MEAS_CLIENT_INTERFACE".U01_STA3_MEAS_Read.Variable.Status = (-1)) AND "DB16001_U01_STA3_MEAS_CLIENT_INTERFACE".U01_STA3_MEAS_Read.Variable.ProfilerConfiguration) OR ("DB16000_OPC_UA_TRIGGER_ALARM".CLIENT.U01_STA3_MEAS.ALARMS.PROFILER_CONFIG_A AND NOT "DB2120_MPP_ITC_IPC".RESET_FAULTS)) AND "DB7253_UNIT_01_STA_3_MEAS_ENABLE_DISABLE".ENABLED;
   "DB426_ALARMS_WARNINGS".UNIT_01.OTHER."716500" := "DB16000_OPC_UA_TRIGGER_ALARM".CLIENT.U01_STA3_MEAS.ALARMS.PROFILER_CONFIG_A;
END_REGION

REGION Network 35: UNIT 01 STATION 3 MEASURING ANALYZER CONFIGURATION ALARM
   RUNG wire#powerrail
      { S7_Templates := "SrcType := Int" } EQ_Contact(in1 := "DB16001_U01_STA3_MEAS_CLIENT_INTERFACE".U01_STA3_MEAS_Read.Variable.Status, in2 := -1)
      Contact( "DB16001_U01_STA3_MEAS_CLIENT_INTERFACE".U01_STA3_MEAS_Read.Variable.AnalyzerConfiguration )
      wire#w1
      Contact( "DB7253_UNIT_01_STA_3_MEAS_ENABLE_DISABLE".ENABLED )
      wire#w2
      Coil( "DB16000_OPC_UA_TRIGGER_ALARM".CLIENT.U01_STA3_MEAS.ALARMS.ANALYZER_CONFIG_A )
   END_RUNG
   RUNG wire#powerrail
      Contact( "DB16000_OPC_UA_TRIGGER_ALARM".CLIENT.U01_STA3_MEAS.ALARMS.ANALYZER_CONFIG_A )
      I_Contact( "DB2120_MPP_ITC_IPC".RESET_FAULTS )
   END_RUNG wire#w1
   RUNG wire#w2
      Coil( "DB426_ALARMS_WARNINGS".UNIT_01.OTHER."716501" )
   END_RUNG
   // the same network as SCL:
   "DB16000_OPC_UA_TRIGGER_ALARM".CLIENT.U01_STA3_MEAS.ALARMS.ANALYZER_CONFIG_A := ((("DB16001_U01_STA3_MEAS_CLIENT_INTERFACE".U01_STA3_MEAS_Read.Variable.Status = (-1)) AND "DB16001_U01_STA3_MEAS_CLIENT_INTERFACE".U01_STA3_MEAS_Read.Variable.AnalyzerConfiguration) OR ("DB16000_OPC_UA_TRIGGER_ALARM".CLIENT.U01_STA3_MEAS.ALARMS.ANALYZER_CONFIG_A AND NOT "DB2120_MPP_ITC_IPC".RESET_FAULTS)) AND "DB7253_UNIT_01_STA_3_MEAS_ENABLE_DISABLE".ENABLED;
   "DB426_ALARMS_WARNINGS".UNIT_01.OTHER."716501" := "DB16000_OPC_UA_TRIGGER_ALARM".CLIENT.U01_STA3_MEAS.ALARMS.ANALYZER_CONFIG_A;
END_REGION

REGION Network 36: UNIT 01 STATION 3 MEASURING DMC STRUCTURE ALARM
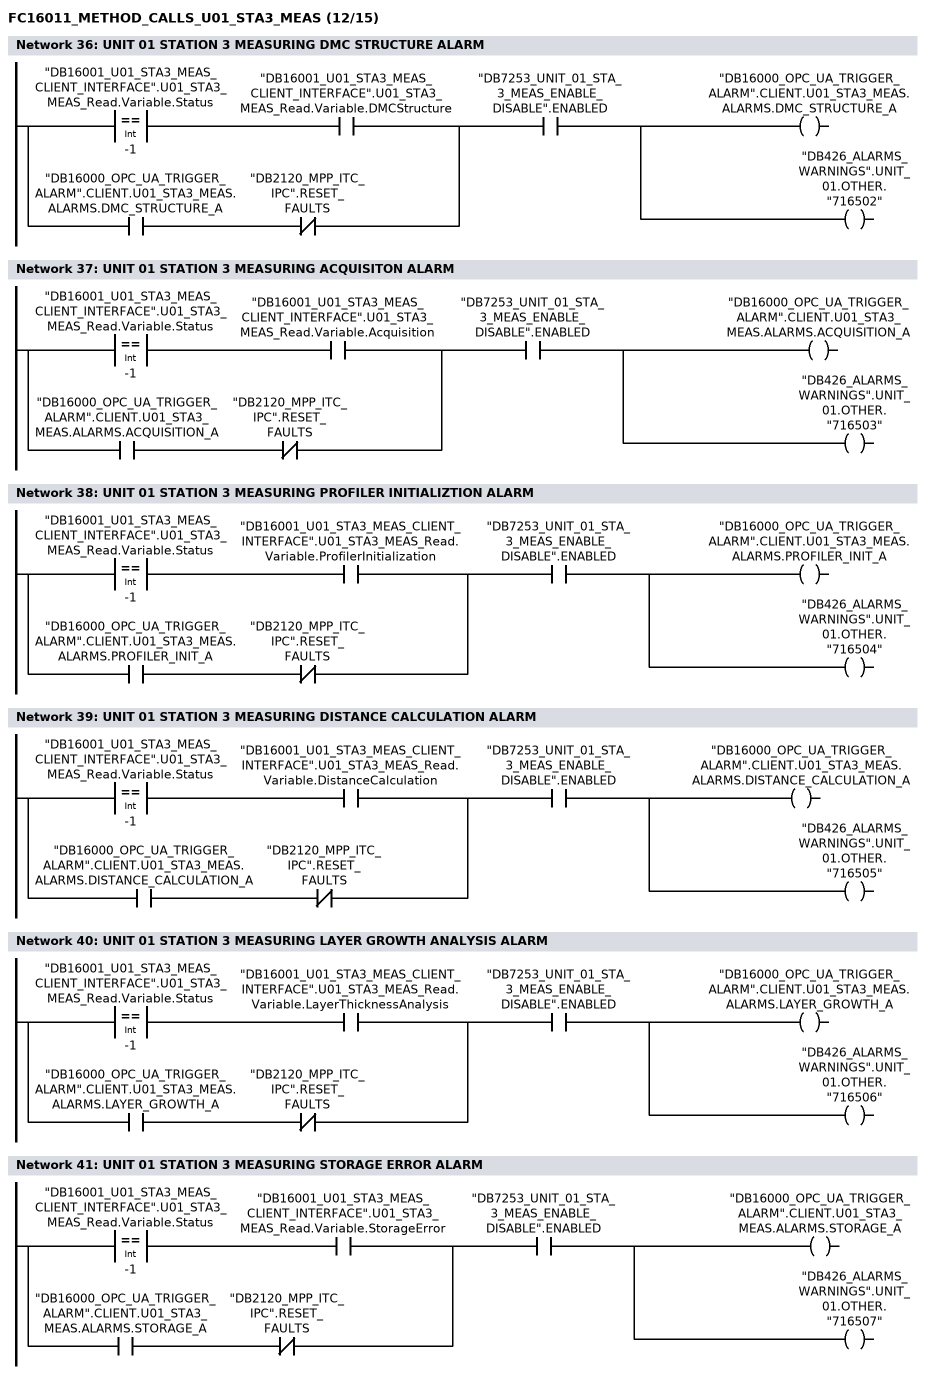
   RUNG wire#powerrail
      { S7_Templates := "SrcType := Int" } EQ_Contact(in1 := "DB16001_U01_STA3_MEAS_CLIENT_INTERFACE".U01_STA3_MEAS_Read.Variable.Status, in2 := -1)
      Contact( "DB16001_U01_STA3_MEAS_CLIENT_INTERFACE".U01_STA3_MEAS_Read.Variable.DMCStructure )
      wire#w1
      Contact( "DB7253_UNIT_01_STA_3_MEAS_ENABLE_DISABLE".ENABLED )
      wire#w2
      Coil( "DB16000_OPC_UA_TRIGGER_ALARM".CLIENT.U01_STA3_MEAS.ALARMS.DMC_STRUCTURE_A )
   END_RUNG
   RUNG wire#powerrail
      Contact( "DB16000_OPC_UA_TRIGGER_ALARM".CLIENT.U01_STA3_MEAS.ALARMS.DMC_STRUCTURE_A )
      I_Contact( "DB2120_MPP_ITC_IPC".RESET_FAULTS )
   END_RUNG wire#w1
   RUNG wire#w2
      Coil( "DB426_ALARMS_WARNINGS".UNIT_01.OTHER."716502" )
   END_RUNG
   // the same network as SCL:
   "DB16000_OPC_UA_TRIGGER_ALARM".CLIENT.U01_STA3_MEAS.ALARMS.DMC_STRUCTURE_A := ((("DB16001_U01_STA3_MEAS_CLIENT_INTERFACE".U01_STA3_MEAS_Read.Variable.Status = (-1)) AND "DB16001_U01_STA3_MEAS_CLIENT_INTERFACE".U01_STA3_MEAS_Read.Variable.DMCStructure) OR ("DB16000_OPC_UA_TRIGGER_ALARM".CLIENT.U01_STA3_MEAS.ALARMS.DMC_STRUCTURE_A AND NOT "DB2120_MPP_ITC_IPC".RESET_FAULTS)) AND "DB7253_UNIT_01_STA_3_MEAS_ENABLE_DISABLE".ENABLED;
   "DB426_ALARMS_WARNINGS".UNIT_01.OTHER."716502" := "DB16000_OPC_UA_TRIGGER_ALARM".CLIENT.U01_STA3_MEAS.ALARMS.DMC_STRUCTURE_A;
END_REGION

REGION Network 37: UNIT 01 STATION 3 MEASURING ACQUISITON ALARM
   RUNG wire#powerrail
      { S7_Templates := "SrcType := Int" } EQ_Contact(in1 := "DB16001_U01_STA3_MEAS_CLIENT_INTERFACE".U01_STA3_MEAS_Read.Variable.Status, in2 := -1)
      Contact( "DB16001_U01_STA3_MEAS_CLIENT_INTERFACE".U01_STA3_MEAS_Read.Variable.Acquisition )
      wire#w1
      Contact( "DB7253_UNIT_01_STA_3_MEAS_ENABLE_DISABLE".ENABLED )
      wire#w2
      Coil( "DB16000_OPC_UA_TRIGGER_ALARM".CLIENT.U01_STA3_MEAS.ALARMS.ACQUISITION_A )
   END_RUNG
   RUNG wire#powerrail
      Contact( "DB16000_OPC_UA_TRIGGER_ALARM".CLIENT.U01_STA3_MEAS.ALARMS.ACQUISITION_A )
      I_Contact( "DB2120_MPP_ITC_IPC".RESET_FAULTS )
   END_RUNG wire#w1
   RUNG wire#w2
      Coil( "DB426_ALARMS_WARNINGS".UNIT_01.OTHER."716503" )
   END_RUNG
   // the same network as SCL:
   "DB16000_OPC_UA_TRIGGER_ALARM".CLIENT.U01_STA3_MEAS.ALARMS.ACQUISITION_A := ((("DB16001_U01_STA3_MEAS_CLIENT_INTERFACE".U01_STA3_MEAS_Read.Variable.Status = (-1)) AND "DB16001_U01_STA3_MEAS_CLIENT_INTERFACE".U01_STA3_MEAS_Read.Variable.Acquisition) OR ("DB16000_OPC_UA_TRIGGER_ALARM".CLIENT.U01_STA3_MEAS.ALARMS.ACQUISITION_A AND NOT "DB2120_MPP_ITC_IPC".RESET_FAULTS)) AND "DB7253_UNIT_01_STA_3_MEAS_ENABLE_DISABLE".ENABLED;
   "DB426_ALARMS_WARNINGS".UNIT_01.OTHER."716503" := "DB16000_OPC_UA_TRIGGER_ALARM".CLIENT.U01_STA3_MEAS.ALARMS.ACQUISITION_A;
END_REGION

REGION Network 38: UNIT 01 STATION 3 MEASURING PROFILER INITIALIZTION ALARM
   RUNG wire#powerrail
      { S7_Templates := "SrcType := Int" } EQ_Contact(in1 := "DB16001_U01_STA3_MEAS_CLIENT_INTERFACE".U01_STA3_MEAS_Read.Variable.Status, in2 := -1)
      Contact( "DB16001_U01_STA3_MEAS_CLIENT_INTERFACE".U01_STA3_MEAS_Read.Variable.ProfilerInitialization )
      wire#w1
      Contact( "DB7253_UNIT_01_STA_3_MEAS_ENABLE_DISABLE".ENABLED )
      wire#w2
      Coil( "DB16000_OPC_UA_TRIGGER_ALARM".CLIENT.U01_STA3_MEAS.ALARMS.PROFILER_INIT_A )
   END_RUNG
   RUNG wire#powerrail
      Contact( "DB16000_OPC_UA_TRIGGER_ALARM".CLIENT.U01_STA3_MEAS.ALARMS.PROFILER_INIT_A )
      I_Contact( "DB2120_MPP_ITC_IPC".RESET_FAULTS )
   END_RUNG wire#w1
   RUNG wire#w2
      Coil( "DB426_ALARMS_WARNINGS".UNIT_01.OTHER."716504" )
   END_RUNG
   // the same network as SCL:
   "DB16000_OPC_UA_TRIGGER_ALARM".CLIENT.U01_STA3_MEAS.ALARMS.PROFILER_INIT_A := ((("DB16001_U01_STA3_MEAS_CLIENT_INTERFACE".U01_STA3_MEAS_Read.Variable.Status = (-1)) AND "DB16001_U01_STA3_MEAS_CLIENT_INTERFACE".U01_STA3_MEAS_Read.Variable.ProfilerInitialization) OR ("DB16000_OPC_UA_TRIGGER_ALARM".CLIENT.U01_STA3_MEAS.ALARMS.PROFILER_INIT_A AND NOT "DB2120_MPP_ITC_IPC".RESET_FAULTS)) AND "DB7253_UNIT_01_STA_3_MEAS_ENABLE_DISABLE".ENABLED;
   "DB426_ALARMS_WARNINGS".UNIT_01.OTHER."716504" := "DB16000_OPC_UA_TRIGGER_ALARM".CLIENT.U01_STA3_MEAS.ALARMS.PROFILER_INIT_A;
END_REGION

REGION Network 39: UNIT 01 STATION 3 MEASURING DISTANCE CALCULATION ALARM
   RUNG wire#powerrail
      { S7_Templates := "SrcType := Int" } EQ_Contact(in1 := "DB16001_U01_STA3_MEAS_CLIENT_INTERFACE".U01_STA3_MEAS_Read.Variable.Status, in2 := -1)
      Contact( "DB16001_U01_STA3_MEAS_CLIENT_INTERFACE".U01_STA3_MEAS_Read.Variable.DistanceCalculation )
      wire#w1
      Contact( "DB7253_UNIT_01_STA_3_MEAS_ENABLE_DISABLE".ENABLED )
      wire#w2
      Coil( "DB16000_OPC_UA_TRIGGER_ALARM".CLIENT.U01_STA3_MEAS.ALARMS.DISTANCE_CALCULATION_A )
   END_RUNG
   RUNG wire#powerrail
      Contact( "DB16000_OPC_UA_TRIGGER_ALARM".CLIENT.U01_STA3_MEAS.ALARMS.DISTANCE_CALCULATION_A )
      I_Contact( "DB2120_MPP_ITC_IPC".RESET_FAULTS )
   END_RUNG wire#w1
   RUNG wire#w2
      Coil( "DB426_ALARMS_WARNINGS".UNIT_01.OTHER."716505" )
   END_RUNG
   // the same network as SCL:
   "DB16000_OPC_UA_TRIGGER_ALARM".CLIENT.U01_STA3_MEAS.ALARMS.DISTANCE_CALCULATION_A := ((("DB16001_U01_STA3_MEAS_CLIENT_INTERFACE".U01_STA3_MEAS_Read.Variable.Status = (-1)) AND "DB16001_U01_STA3_MEAS_CLIENT_INTERFACE".U01_STA3_MEAS_Read.Variable.DistanceCalculation) OR ("DB16000_OPC_UA_TRIGGER_ALARM".CLIENT.U01_STA3_MEAS.ALARMS.DISTANCE_CALCULATION_A AND NOT "DB2120_MPP_ITC_IPC".RESET_FAULTS)) AND "DB7253_UNIT_01_STA_3_MEAS_ENABLE_DISABLE".ENABLED;
   "DB426_ALARMS_WARNINGS".UNIT_01.OTHER."716505" := "DB16000_OPC_UA_TRIGGER_ALARM".CLIENT.U01_STA3_MEAS.ALARMS.DISTANCE_CALCULATION_A;
END_REGION

REGION Network 40: UNIT 01 STATION 3 MEASURING LAYER GROWTH ANALYSIS ALARM
   RUNG wire#powerrail
      { S7_Templates := "SrcType := Int" } EQ_Contact(in1 := "DB16001_U01_STA3_MEAS_CLIENT_INTERFACE".U01_STA3_MEAS_Read.Variable.Status, in2 := -1)
      Contact( "DB16001_U01_STA3_MEAS_CLIENT_INTERFACE".U01_STA3_MEAS_Read.Variable.LayerThicknessAnalysis )
      wire#w1
      Contact( "DB7253_UNIT_01_STA_3_MEAS_ENABLE_DISABLE".ENABLED )
      wire#w2
      Coil( "DB16000_OPC_UA_TRIGGER_ALARM".CLIENT.U01_STA3_MEAS.ALARMS.LAYER_GROWTH_A )
   END_RUNG
   RUNG wire#powerrail
      Contact( "DB16000_OPC_UA_TRIGGER_ALARM".CLIENT.U01_STA3_MEAS.ALARMS.LAYER_GROWTH_A )
      I_Contact( "DB2120_MPP_ITC_IPC".RESET_FAULTS )
   END_RUNG wire#w1
   RUNG wire#w2
      Coil( "DB426_ALARMS_WARNINGS".UNIT_01.OTHER."716506" )
   END_RUNG
   // the same network as SCL:
   "DB16000_OPC_UA_TRIGGER_ALARM".CLIENT.U01_STA3_MEAS.ALARMS.LAYER_GROWTH_A := ((("DB16001_U01_STA3_MEAS_CLIENT_INTERFACE".U01_STA3_MEAS_Read.Variable.Status = (-1)) AND "DB16001_U01_STA3_MEAS_CLIENT_INTERFACE".U01_STA3_MEAS_Read.Variable.LayerThicknessAnalysis) OR ("DB16000_OPC_UA_TRIGGER_ALARM".CLIENT.U01_STA3_MEAS.ALARMS.LAYER_GROWTH_A AND NOT "DB2120_MPP_ITC_IPC".RESET_FAULTS)) AND "DB7253_UNIT_01_STA_3_MEAS_ENABLE_DISABLE".ENABLED;
   "DB426_ALARMS_WARNINGS".UNIT_01.OTHER."716506" := "DB16000_OPC_UA_TRIGGER_ALARM".CLIENT.U01_STA3_MEAS.ALARMS.LAYER_GROWTH_A;
END_REGION

REGION Network 41: UNIT 01 STATION 3 MEASURING STORAGE ERROR ALARM
   RUNG wire#powerrail
      { S7_Templates := "SrcType := Int" } EQ_Contact(in1 := "DB16001_U01_STA3_MEAS_CLIENT_INTERFACE".U01_STA3_MEAS_Read.Variable.Status, in2 := -1)
      Contact( "DB16001_U01_STA3_MEAS_CLIENT_INTERFACE".U01_STA3_MEAS_Read.Variable.StorageError )
      wire#w1
      Contact( "DB7253_UNIT_01_STA_3_MEAS_ENABLE_DISABLE".ENABLED )
      wire#w2
      Coil( "DB16000_OPC_UA_TRIGGER_ALARM".CLIENT.U01_STA3_MEAS.ALARMS.STORAGE_A )
   END_RUNG
   RUNG wire#powerrail
      Contact( "DB16000_OPC_UA_TRIGGER_ALARM".CLIENT.U01_STA3_MEAS.ALARMS.STORAGE_A )
      I_Contact( "DB2120_MPP_ITC_IPC".RESET_FAULTS )
   END_RUNG wire#w1
   RUNG wire#w2
      Coil( "DB426_ALARMS_WARNINGS".UNIT_01.OTHER."716507" )
   END_RUNG
   // the same network as SCL:
   "DB16000_OPC_UA_TRIGGER_ALARM".CLIENT.U01_STA3_MEAS.ALARMS.STORAGE_A := ((("DB16001_U01_STA3_MEAS_CLIENT_INTERFACE".U01_STA3_MEAS_Read.Variable.Status = (-1)) AND "DB16001_U01_STA3_MEAS_CLIENT_INTERFACE".U01_STA3_MEAS_Read.Variable.StorageError) OR ("DB16000_OPC_UA_TRIGGER_ALARM".CLIENT.U01_STA3_MEAS.ALARMS.STORAGE_A AND NOT "DB2120_MPP_ITC_IPC".RESET_FAULTS)) AND "DB7253_UNIT_01_STA_3_MEAS_ENABLE_DISABLE".ENABLED;
   "DB426_ALARMS_WARNINGS".UNIT_01.OTHER."716507" := "DB16000_OPC_UA_TRIGGER_ALARM".CLIENT.U01_STA3_MEAS.ALARMS.STORAGE_A;
END_REGION

REGION Network 42: UNIT 01 STATION 3 MEASURING DATABASE CONNECTION ALARM
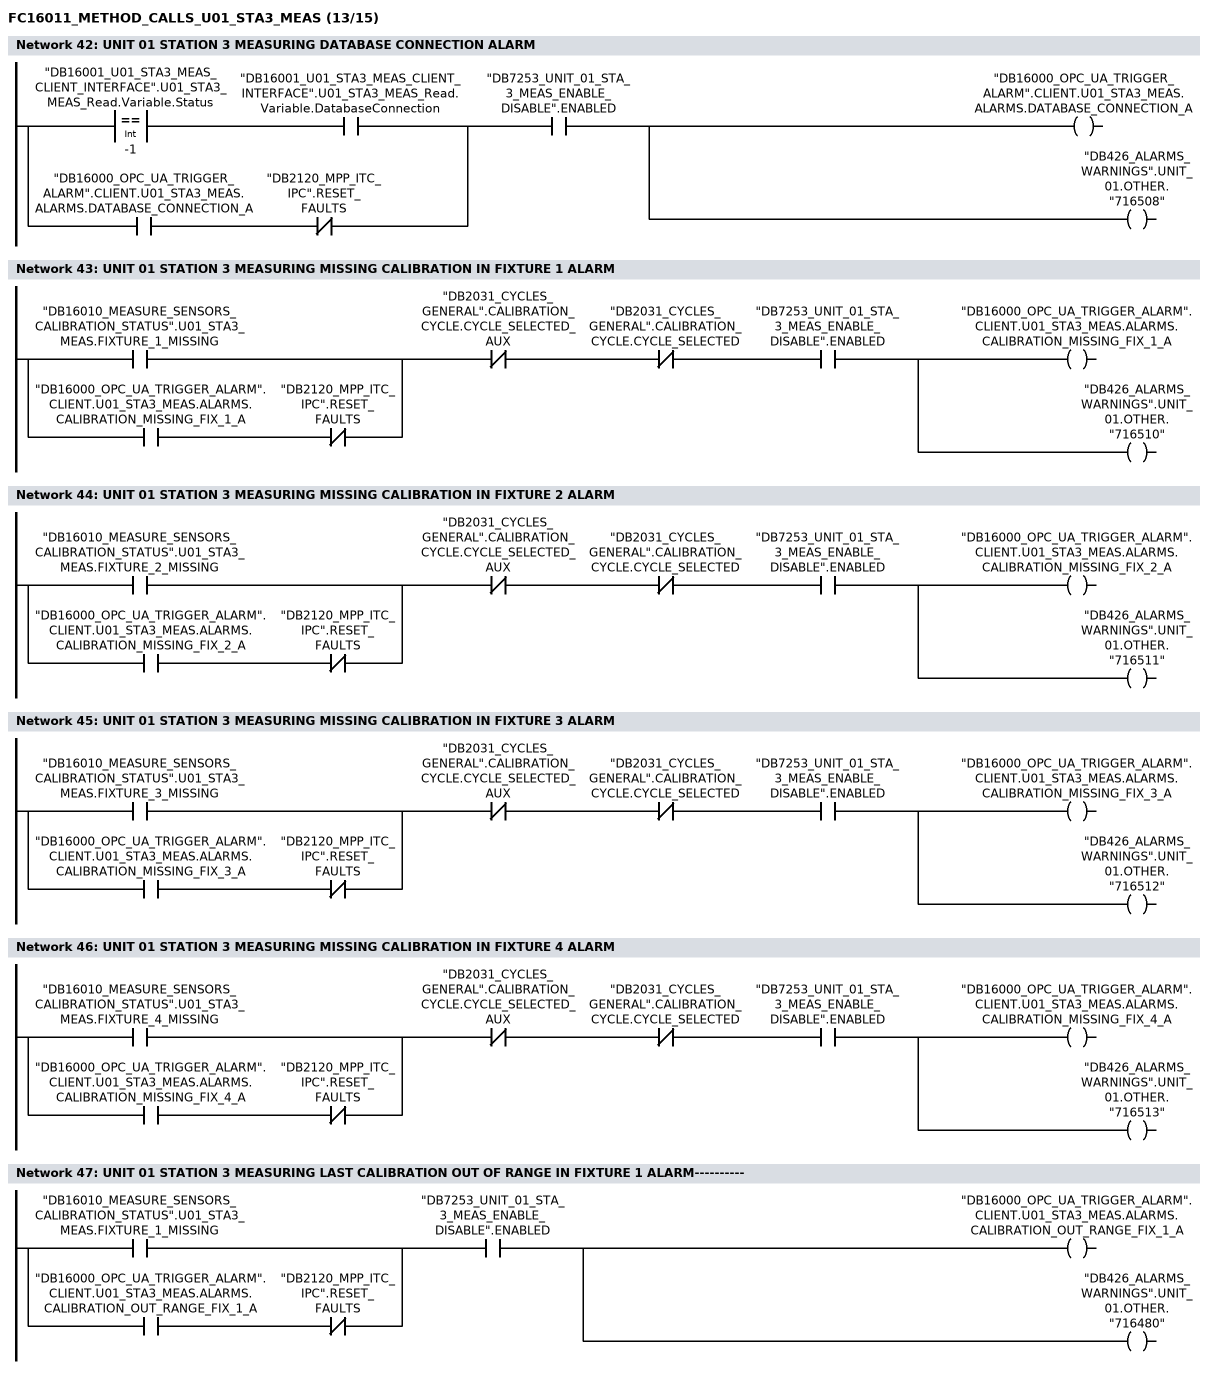
   RUNG wire#powerrail
      { S7_Templates := "SrcType := Int" } EQ_Contact(in1 := "DB16001_U01_STA3_MEAS_CLIENT_INTERFACE".U01_STA3_MEAS_Read.Variable.Status, in2 := -1)
      Contact( "DB16001_U01_STA3_MEAS_CLIENT_INTERFACE".U01_STA3_MEAS_Read.Variable.DatabaseConnection )
      wire#w1
      Contact( "DB7253_UNIT_01_STA_3_MEAS_ENABLE_DISABLE".ENABLED )
      wire#w2
      Coil( "DB16000_OPC_UA_TRIGGER_ALARM".CLIENT.U01_STA3_MEAS.ALARMS.DATABASE_CONNECTION_A )
   END_RUNG
   RUNG wire#powerrail
      Contact( "DB16000_OPC_UA_TRIGGER_ALARM".CLIENT.U01_STA3_MEAS.ALARMS.DATABASE_CONNECTION_A )
      I_Contact( "DB2120_MPP_ITC_IPC".RESET_FAULTS )
   END_RUNG wire#w1
   RUNG wire#w2
      Coil( "DB426_ALARMS_WARNINGS".UNIT_01.OTHER."716508" )
   END_RUNG
   // the same network as SCL:
   "DB16000_OPC_UA_TRIGGER_ALARM".CLIENT.U01_STA3_MEAS.ALARMS.DATABASE_CONNECTION_A := ((("DB16001_U01_STA3_MEAS_CLIENT_INTERFACE".U01_STA3_MEAS_Read.Variable.Status = (-1)) AND "DB16001_U01_STA3_MEAS_CLIENT_INTERFACE".U01_STA3_MEAS_Read.Variable.DatabaseConnection) OR ("DB16000_OPC_UA_TRIGGER_ALARM".CLIENT.U01_STA3_MEAS.ALARMS.DATABASE_CONNECTION_A AND NOT "DB2120_MPP_ITC_IPC".RESET_FAULTS)) AND "DB7253_UNIT_01_STA_3_MEAS_ENABLE_DISABLE".ENABLED;
   "DB426_ALARMS_WARNINGS".UNIT_01.OTHER."716508" := "DB16000_OPC_UA_TRIGGER_ALARM".CLIENT.U01_STA3_MEAS.ALARMS.DATABASE_CONNECTION_A;
END_REGION

REGION Network 43: UNIT 01 STATION 3 MEASURING MISSING CALIBRATION IN FIXTURE 1 ALARM
   RUNG wire#powerrail
      Contact( "DB16010_MEASURE_SENSORS_CALIBRATION_STATUS".U01_STA3_MEAS.FIXTURE_1_MISSING )
      wire#w1
      I_Contact( "DB2031_CYCLES_GENERAL".CALIBRATION_CYCLE.CYCLE_SELECTED_AUX )
      I_Contact( "DB2031_CYCLES_GENERAL".CALIBRATION_CYCLE.CYCLE_SELECTED )
      Contact( "DB7253_UNIT_01_STA_3_MEAS_ENABLE_DISABLE".ENABLED )
      wire#w2
      Coil( "DB16000_OPC_UA_TRIGGER_ALARM".CLIENT.U01_STA3_MEAS.ALARMS.CALIBRATION_MISSING_FIX_1_A )
   END_RUNG
   RUNG wire#powerrail
      Contact( "DB16000_OPC_UA_TRIGGER_ALARM".CLIENT.U01_STA3_MEAS.ALARMS.CALIBRATION_MISSING_FIX_1_A )
      I_Contact( "DB2120_MPP_ITC_IPC".RESET_FAULTS )
   END_RUNG wire#w1
   RUNG wire#w2
      Coil( "DB426_ALARMS_WARNINGS".UNIT_01.OTHER."716510" )
   END_RUNG
   // the same network as SCL:
   "DB16000_OPC_UA_TRIGGER_ALARM".CLIENT.U01_STA3_MEAS.ALARMS.CALIBRATION_MISSING_FIX_1_A := ("DB16010_MEASURE_SENSORS_CALIBRATION_STATUS".U01_STA3_MEAS.FIXTURE_1_MISSING OR ("DB16000_OPC_UA_TRIGGER_ALARM".CLIENT.U01_STA3_MEAS.ALARMS.CALIBRATION_MISSING_FIX_1_A AND NOT "DB2120_MPP_ITC_IPC".RESET_FAULTS)) AND NOT "DB2031_CYCLES_GENERAL".CALIBRATION_CYCLE.CYCLE_SELECTED_AUX AND NOT "DB2031_CYCLES_GENERAL".CALIBRATION_CYCLE.CYCLE_SELECTED AND "DB7253_UNIT_01_STA_3_MEAS_ENABLE_DISABLE".ENABLED;
   "DB426_ALARMS_WARNINGS".UNIT_01.OTHER."716510" := "DB16000_OPC_UA_TRIGGER_ALARM".CLIENT.U01_STA3_MEAS.ALARMS.CALIBRATION_MISSING_FIX_1_A;
END_REGION

REGION Network 44: UNIT 01 STATION 3 MEASURING MISSING CALIBRATION IN FIXTURE 2 ALARM
   RUNG wire#powerrail
      Contact( "DB16010_MEASURE_SENSORS_CALIBRATION_STATUS".U01_STA3_MEAS.FIXTURE_2_MISSING )
      wire#w1
      I_Contact( "DB2031_CYCLES_GENERAL".CALIBRATION_CYCLE.CYCLE_SELECTED_AUX )
      I_Contact( "DB2031_CYCLES_GENERAL".CALIBRATION_CYCLE.CYCLE_SELECTED )
      Contact( "DB7253_UNIT_01_STA_3_MEAS_ENABLE_DISABLE".ENABLED )
      wire#w2
      Coil( "DB16000_OPC_UA_TRIGGER_ALARM".CLIENT.U01_STA3_MEAS.ALARMS.CALIBRATION_MISSING_FIX_2_A )
   END_RUNG
   RUNG wire#powerrail
      Contact( "DB16000_OPC_UA_TRIGGER_ALARM".CLIENT.U01_STA3_MEAS.ALARMS.CALIBRATION_MISSING_FIX_2_A )
      I_Contact( "DB2120_MPP_ITC_IPC".RESET_FAULTS )
   END_RUNG wire#w1
   RUNG wire#w2
      Coil( "DB426_ALARMS_WARNINGS".UNIT_01.OTHER."716511" )
   END_RUNG
   // the same network as SCL:
   "DB16000_OPC_UA_TRIGGER_ALARM".CLIENT.U01_STA3_MEAS.ALARMS.CALIBRATION_MISSING_FIX_2_A := ("DB16010_MEASURE_SENSORS_CALIBRATION_STATUS".U01_STA3_MEAS.FIXTURE_2_MISSING OR ("DB16000_OPC_UA_TRIGGER_ALARM".CLIENT.U01_STA3_MEAS.ALARMS.CALIBRATION_MISSING_FIX_2_A AND NOT "DB2120_MPP_ITC_IPC".RESET_FAULTS)) AND NOT "DB2031_CYCLES_GENERAL".CALIBRATION_CYCLE.CYCLE_SELECTED_AUX AND NOT "DB2031_CYCLES_GENERAL".CALIBRATION_CYCLE.CYCLE_SELECTED AND "DB7253_UNIT_01_STA_3_MEAS_ENABLE_DISABLE".ENABLED;
   "DB426_ALARMS_WARNINGS".UNIT_01.OTHER."716511" := "DB16000_OPC_UA_TRIGGER_ALARM".CLIENT.U01_STA3_MEAS.ALARMS.CALIBRATION_MISSING_FIX_2_A;
END_REGION

REGION Network 45: UNIT 01 STATION 3 MEASURING MISSING CALIBRATION IN FIXTURE 3 ALARM
   RUNG wire#powerrail
      Contact( "DB16010_MEASURE_SENSORS_CALIBRATION_STATUS".U01_STA3_MEAS.FIXTURE_3_MISSING )
      wire#w1
      I_Contact( "DB2031_CYCLES_GENERAL".CALIBRATION_CYCLE.CYCLE_SELECTED_AUX )
      I_Contact( "DB2031_CYCLES_GENERAL".CALIBRATION_CYCLE.CYCLE_SELECTED )
      Contact( "DB7253_UNIT_01_STA_3_MEAS_ENABLE_DISABLE".ENABLED )
      wire#w2
      Coil( "DB16000_OPC_UA_TRIGGER_ALARM".CLIENT.U01_STA3_MEAS.ALARMS.CALIBRATION_MISSING_FIX_3_A )
   END_RUNG
   RUNG wire#powerrail
      Contact( "DB16000_OPC_UA_TRIGGER_ALARM".CLIENT.U01_STA3_MEAS.ALARMS.CALIBRATION_MISSING_FIX_3_A )
      I_Contact( "DB2120_MPP_ITC_IPC".RESET_FAULTS )
   END_RUNG wire#w1
   RUNG wire#w2
      Coil( "DB426_ALARMS_WARNINGS".UNIT_01.OTHER."716512" )
   END_RUNG
   // the same network as SCL:
   "DB16000_OPC_UA_TRIGGER_ALARM".CLIENT.U01_STA3_MEAS.ALARMS.CALIBRATION_MISSING_FIX_3_A := ("DB16010_MEASURE_SENSORS_CALIBRATION_STATUS".U01_STA3_MEAS.FIXTURE_3_MISSING OR ("DB16000_OPC_UA_TRIGGER_ALARM".CLIENT.U01_STA3_MEAS.ALARMS.CALIBRATION_MISSING_FIX_3_A AND NOT "DB2120_MPP_ITC_IPC".RESET_FAULTS)) AND NOT "DB2031_CYCLES_GENERAL".CALIBRATION_CYCLE.CYCLE_SELECTED_AUX AND NOT "DB2031_CYCLES_GENERAL".CALIBRATION_CYCLE.CYCLE_SELECTED AND "DB7253_UNIT_01_STA_3_MEAS_ENABLE_DISABLE".ENABLED;
   "DB426_ALARMS_WARNINGS".UNIT_01.OTHER."716512" := "DB16000_OPC_UA_TRIGGER_ALARM".CLIENT.U01_STA3_MEAS.ALARMS.CALIBRATION_MISSING_FIX_3_A;
END_REGION

REGION Network 46: UNIT 01 STATION 3 MEASURING MISSING CALIBRATION IN FIXTURE 4 ALARM
   RUNG wire#powerrail
      Contact( "DB16010_MEASURE_SENSORS_CALIBRATION_STATUS".U01_STA3_MEAS.FIXTURE_4_MISSING )
      wire#w1
      I_Contact( "DB2031_CYCLES_GENERAL".CALIBRATION_CYCLE.CYCLE_SELECTED_AUX )
      I_Contact( "DB2031_CYCLES_GENERAL".CALIBRATION_CYCLE.CYCLE_SELECTED )
      Contact( "DB7253_UNIT_01_STA_3_MEAS_ENABLE_DISABLE".ENABLED )
      wire#w2
      Coil( "DB16000_OPC_UA_TRIGGER_ALARM".CLIENT.U01_STA3_MEAS.ALARMS.CALIBRATION_MISSING_FIX_4_A )
   END_RUNG
   RUNG wire#powerrail
      Contact( "DB16000_OPC_UA_TRIGGER_ALARM".CLIENT.U01_STA3_MEAS.ALARMS.CALIBRATION_MISSING_FIX_4_A )
      I_Contact( "DB2120_MPP_ITC_IPC".RESET_FAULTS )
   END_RUNG wire#w1
   RUNG wire#w2
      Coil( "DB426_ALARMS_WARNINGS".UNIT_01.OTHER."716513" )
   END_RUNG
   // the same network as SCL:
   "DB16000_OPC_UA_TRIGGER_ALARM".CLIENT.U01_STA3_MEAS.ALARMS.CALIBRATION_MISSING_FIX_4_A := ("DB16010_MEASURE_SENSORS_CALIBRATION_STATUS".U01_STA3_MEAS.FIXTURE_4_MISSING OR ("DB16000_OPC_UA_TRIGGER_ALARM".CLIENT.U01_STA3_MEAS.ALARMS.CALIBRATION_MISSING_FIX_4_A AND NOT "DB2120_MPP_ITC_IPC".RESET_FAULTS)) AND NOT "DB2031_CYCLES_GENERAL".CALIBRATION_CYCLE.CYCLE_SELECTED_AUX AND NOT "DB2031_CYCLES_GENERAL".CALIBRATION_CYCLE.CYCLE_SELECTED AND "DB7253_UNIT_01_STA_3_MEAS_ENABLE_DISABLE".ENABLED;
   "DB426_ALARMS_WARNINGS".UNIT_01.OTHER."716513" := "DB16000_OPC_UA_TRIGGER_ALARM".CLIENT.U01_STA3_MEAS.ALARMS.CALIBRATION_MISSING_FIX_4_A;
END_REGION

REGION Network 47: UNIT 01 STATION 3 MEASURING LAST CALIBRATION OUT OF RANGE IN FIXTURE 1 ALARM----------
   RUNG wire#powerrail
      Contact( "DB16010_MEASURE_SENSORS_CALIBRATION_STATUS".U01_STA3_MEAS.FIXTURE_1_MISSING )
      wire#w1
      Contact( "DB7253_UNIT_01_STA_3_MEAS_ENABLE_DISABLE".ENABLED )
      wire#w2
      Coil( "DB16000_OPC_UA_TRIGGER_ALARM".CLIENT.U01_STA3_MEAS.ALARMS.CALIBRATION_OUT_RANGE_FIX_1_A )
   END_RUNG
   RUNG wire#powerrail
      Contact( "DB16000_OPC_UA_TRIGGER_ALARM".CLIENT.U01_STA3_MEAS.ALARMS.CALIBRATION_OUT_RANGE_FIX_1_A )
      I_Contact( "DB2120_MPP_ITC_IPC".RESET_FAULTS )
   END_RUNG wire#w1
   RUNG wire#w2
      Coil( "DB426_ALARMS_WARNINGS".UNIT_01.OTHER."716480" )
   END_RUNG
   // the same network as SCL:
   "DB16000_OPC_UA_TRIGGER_ALARM".CLIENT.U01_STA3_MEAS.ALARMS.CALIBRATION_OUT_RANGE_FIX_1_A := ("DB16010_MEASURE_SENSORS_CALIBRATION_STATUS".U01_STA3_MEAS.FIXTURE_1_MISSING OR ("DB16000_OPC_UA_TRIGGER_ALARM".CLIENT.U01_STA3_MEAS.ALARMS.CALIBRATION_OUT_RANGE_FIX_1_A AND NOT "DB2120_MPP_ITC_IPC".RESET_FAULTS)) AND "DB7253_UNIT_01_STA_3_MEAS_ENABLE_DISABLE".ENABLED;
   "DB426_ALARMS_WARNINGS".UNIT_01.OTHER."716480" := "DB16000_OPC_UA_TRIGGER_ALARM".CLIENT.U01_STA3_MEAS.ALARMS.CALIBRATION_OUT_RANGE_FIX_1_A;
END_REGION

REGION Network 48: UNIT 01 STATION 3 MEASURING LAST CALIBRATION OUT OF RANGE IN FIXTURE 2 ALARM----------
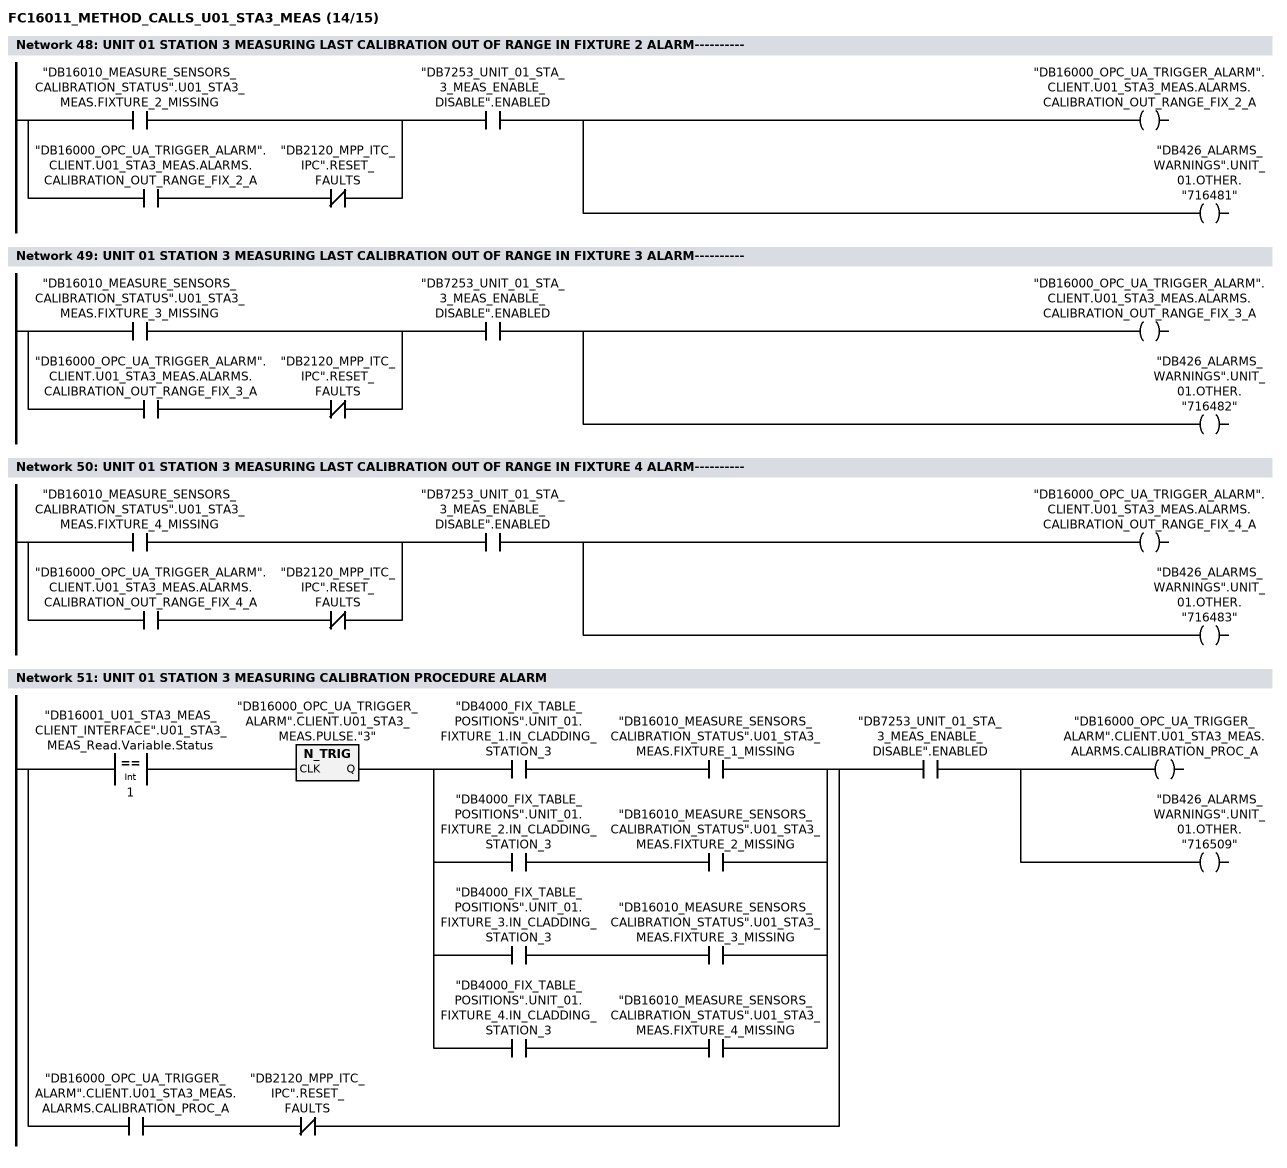
   RUNG wire#powerrail
      Contact( "DB16010_MEASURE_SENSORS_CALIBRATION_STATUS".U01_STA3_MEAS.FIXTURE_2_MISSING )
      wire#w1
      Contact( "DB7253_UNIT_01_STA_3_MEAS_ENABLE_DISABLE".ENABLED )
      wire#w2
      Coil( "DB16000_OPC_UA_TRIGGER_ALARM".CLIENT.U01_STA3_MEAS.ALARMS.CALIBRATION_OUT_RANGE_FIX_2_A )
   END_RUNG
   RUNG wire#powerrail
      Contact( "DB16000_OPC_UA_TRIGGER_ALARM".CLIENT.U01_STA3_MEAS.ALARMS.CALIBRATION_OUT_RANGE_FIX_2_A )
      I_Contact( "DB2120_MPP_ITC_IPC".RESET_FAULTS )
   END_RUNG wire#w1
   RUNG wire#w2
      Coil( "DB426_ALARMS_WARNINGS".UNIT_01.OTHER."716481" )
   END_RUNG
   // the same network as SCL:
   "DB16000_OPC_UA_TRIGGER_ALARM".CLIENT.U01_STA3_MEAS.ALARMS.CALIBRATION_OUT_RANGE_FIX_2_A := ("DB16010_MEASURE_SENSORS_CALIBRATION_STATUS".U01_STA3_MEAS.FIXTURE_2_MISSING OR ("DB16000_OPC_UA_TRIGGER_ALARM".CLIENT.U01_STA3_MEAS.ALARMS.CALIBRATION_OUT_RANGE_FIX_2_A AND NOT "DB2120_MPP_ITC_IPC".RESET_FAULTS)) AND "DB7253_UNIT_01_STA_3_MEAS_ENABLE_DISABLE".ENABLED;
   "DB426_ALARMS_WARNINGS".UNIT_01.OTHER."716481" := "DB16000_OPC_UA_TRIGGER_ALARM".CLIENT.U01_STA3_MEAS.ALARMS.CALIBRATION_OUT_RANGE_FIX_2_A;
END_REGION

REGION Network 49: UNIT 01 STATION 3 MEASURING LAST CALIBRATION OUT OF RANGE IN FIXTURE 3 ALARM----------
   RUNG wire#powerrail
      Contact( "DB16010_MEASURE_SENSORS_CALIBRATION_STATUS".U01_STA3_MEAS.FIXTURE_3_MISSING )
      wire#w1
      Contact( "DB7253_UNIT_01_STA_3_MEAS_ENABLE_DISABLE".ENABLED )
      wire#w2
      Coil( "DB16000_OPC_UA_TRIGGER_ALARM".CLIENT.U01_STA3_MEAS.ALARMS.CALIBRATION_OUT_RANGE_FIX_3_A )
   END_RUNG
   RUNG wire#powerrail
      Contact( "DB16000_OPC_UA_TRIGGER_ALARM".CLIENT.U01_STA3_MEAS.ALARMS.CALIBRATION_OUT_RANGE_FIX_3_A )
      I_Contact( "DB2120_MPP_ITC_IPC".RESET_FAULTS )
   END_RUNG wire#w1
   RUNG wire#w2
      Coil( "DB426_ALARMS_WARNINGS".UNIT_01.OTHER."716482" )
   END_RUNG
   // the same network as SCL:
   "DB16000_OPC_UA_TRIGGER_ALARM".CLIENT.U01_STA3_MEAS.ALARMS.CALIBRATION_OUT_RANGE_FIX_3_A := ("DB16010_MEASURE_SENSORS_CALIBRATION_STATUS".U01_STA3_MEAS.FIXTURE_3_MISSING OR ("DB16000_OPC_UA_TRIGGER_ALARM".CLIENT.U01_STA3_MEAS.ALARMS.CALIBRATION_OUT_RANGE_FIX_3_A AND NOT "DB2120_MPP_ITC_IPC".RESET_FAULTS)) AND "DB7253_UNIT_01_STA_3_MEAS_ENABLE_DISABLE".ENABLED;
   "DB426_ALARMS_WARNINGS".UNIT_01.OTHER."716482" := "DB16000_OPC_UA_TRIGGER_ALARM".CLIENT.U01_STA3_MEAS.ALARMS.CALIBRATION_OUT_RANGE_FIX_3_A;
END_REGION

REGION Network 50: UNIT 01 STATION 3 MEASURING LAST CALIBRATION OUT OF RANGE IN FIXTURE 4 ALARM----------
   RUNG wire#powerrail
      Contact( "DB16010_MEASURE_SENSORS_CALIBRATION_STATUS".U01_STA3_MEAS.FIXTURE_4_MISSING )
      wire#w1
      Contact( "DB7253_UNIT_01_STA_3_MEAS_ENABLE_DISABLE".ENABLED )
      wire#w2
      Coil( "DB16000_OPC_UA_TRIGGER_ALARM".CLIENT.U01_STA3_MEAS.ALARMS.CALIBRATION_OUT_RANGE_FIX_4_A )
   END_RUNG
   RUNG wire#powerrail
      Contact( "DB16000_OPC_UA_TRIGGER_ALARM".CLIENT.U01_STA3_MEAS.ALARMS.CALIBRATION_OUT_RANGE_FIX_4_A )
      I_Contact( "DB2120_MPP_ITC_IPC".RESET_FAULTS )
   END_RUNG wire#w1
   RUNG wire#w2
      Coil( "DB426_ALARMS_WARNINGS".UNIT_01.OTHER."716483" )
   END_RUNG
   // the same network as SCL:
   "DB16000_OPC_UA_TRIGGER_ALARM".CLIENT.U01_STA3_MEAS.ALARMS.CALIBRATION_OUT_RANGE_FIX_4_A := ("DB16010_MEASURE_SENSORS_CALIBRATION_STATUS".U01_STA3_MEAS.FIXTURE_4_MISSING OR ("DB16000_OPC_UA_TRIGGER_ALARM".CLIENT.U01_STA3_MEAS.ALARMS.CALIBRATION_OUT_RANGE_FIX_4_A AND NOT "DB2120_MPP_ITC_IPC".RESET_FAULTS)) AND "DB7253_UNIT_01_STA_3_MEAS_ENABLE_DISABLE".ENABLED;
   "DB426_ALARMS_WARNINGS".UNIT_01.OTHER."716483" := "DB16000_OPC_UA_TRIGGER_ALARM".CLIENT.U01_STA3_MEAS.ALARMS.CALIBRATION_OUT_RANGE_FIX_4_A;
END_REGION

REGION Network 51: UNIT 01 STATION 3 MEASURING CALIBRATION PROCEDURE ALARM
   RUNG wire#powerrail
      { S7_Templates := "SrcType := Int" } EQ_Contact(in1 := "DB16001_U01_STA3_MEAS_CLIENT_INTERFACE".U01_STA3_MEAS_Read.Variable.Status, in2 := 1)
      N_Trig( "DB16000_OPC_UA_TRIGGER_ALARM".CLIENT.U01_STA3_MEAS.PULSE."3" )
      wire#w1
      Contact( "DB4000_FIX_TABLE_POSITIONS".UNIT_01.FIXTURE_1.IN_CLADDING_STATION_3 )
      Contact( "DB16010_MEASURE_SENSORS_CALIBRATION_STATUS".U01_STA3_MEAS.FIXTURE_1_MISSING )
      wire#w2
      Contact( "DB7253_UNIT_01_STA_3_MEAS_ENABLE_DISABLE".ENABLED )
      wire#w3
      Coil( "DB16000_OPC_UA_TRIGGER_ALARM".CLIENT.U01_STA3_MEAS.ALARMS.CALIBRATION_PROC_A )
   END_RUNG
   RUNG wire#w1
      Contact( "DB4000_FIX_TABLE_POSITIONS".UNIT_01.FIXTURE_2.IN_CLADDING_STATION_3 )
      Contact( "DB16010_MEASURE_SENSORS_CALIBRATION_STATUS".U01_STA3_MEAS.FIXTURE_2_MISSING )
   END_RUNG wire#w2
   RUNG wire#w1
      Contact( "DB4000_FIX_TABLE_POSITIONS".UNIT_01.FIXTURE_3.IN_CLADDING_STATION_3 )
      Contact( "DB16010_MEASURE_SENSORS_CALIBRATION_STATUS".U01_STA3_MEAS.FIXTURE_3_MISSING )
   END_RUNG wire#w2
   RUNG wire#w1
      Contact( "DB4000_FIX_TABLE_POSITIONS".UNIT_01.FIXTURE_4.IN_CLADDING_STATION_3 )
      Contact( "DB16010_MEASURE_SENSORS_CALIBRATION_STATUS".U01_STA3_MEAS.FIXTURE_4_MISSING )
   END_RUNG wire#w2
   RUNG wire#powerrail
      Contact( "DB16000_OPC_UA_TRIGGER_ALARM".CLIENT.U01_STA3_MEAS.ALARMS.CALIBRATION_PROC_A )
      I_Contact( "DB2120_MPP_ITC_IPC".RESET_FAULTS )
   END_RUNG wire#w2
   RUNG wire#w3
      Coil( "DB426_ALARMS_WARNINGS".UNIT_01.OTHER."716509" )
   END_RUNG
   // the same network as SCL:
   #_w1 := "DB16001_U01_STA3_MEAS_CLIENT_INTERFACE".U01_STA3_MEAS_Read.Variable.Status = 1;
   #_w2 := NOT #_w1 AND "DB16000_OPC_UA_TRIGGER_ALARM".CLIENT.U01_STA3_MEAS.PULSE."3";   // falling edge
   "DB16000_OPC_UA_TRIGGER_ALARM".CLIENT.U01_STA3_MEAS.PULSE."3" := #_w1;
   "DB16000_OPC_UA_TRIGGER_ALARM".CLIENT.U01_STA3_MEAS.ALARMS.CALIBRATION_PROC_A := ((#_w2 AND (("DB4000_FIX_TABLE_POSITIONS".UNIT_01.FIXTURE_1.IN_CLADDING_STATION_3 AND "DB16010_MEASURE_SENSORS_CALIBRATION_STATUS".U01_STA3_MEAS.FIXTURE_1_MISSING) OR ("DB4000_FIX_TABLE_POSITIONS".UNIT_01.FIXTURE_2.IN_CLADDING_STATION_3 AND "DB16010_MEASURE_SENSORS_CALIBRATION_STATUS".U01_STA3_MEAS.FIXTURE_2_MISSING) OR ("DB4000_FIX_TABLE_POSITIONS".UNIT_01.FIXTURE_3.IN_CLADDING_STATION_3 AND "DB16010_MEASURE_SENSORS_CALIBRATION_STATUS".U01_STA3_MEAS.FIXTURE_3_MISSING) OR ("DB4000_FIX_TABLE_POSITIONS".UNIT_01.FIXTURE_4.IN_CLADDING_STATION_3 AND "DB16010_MEASURE_SENSORS_CALIBRATION_STATUS".U01_STA3_MEAS.FIXTURE_4_MISSING))) OR ("DB16000_OPC_UA_TRIGGER_ALARM".CLIENT.U01_STA3_MEAS.ALARMS.CALIBRATION_PROC_A AND NOT "DB2120_MPP_ITC_IPC".RESET_FAULTS)) AND "DB7253_UNIT_01_STA_3_MEAS_ENABLE_DISABLE".ENABLED;
   "DB426_ALARMS_WARNINGS".UNIT_01.OTHER."716509" := "DB16000_OPC_UA_TRIGGER_ALARM".CLIENT.U01_STA3_MEAS.ALARMS.CALIBRATION_PROC_A;
END_REGION

REGION Network 52: IS_SEOC ALARMS
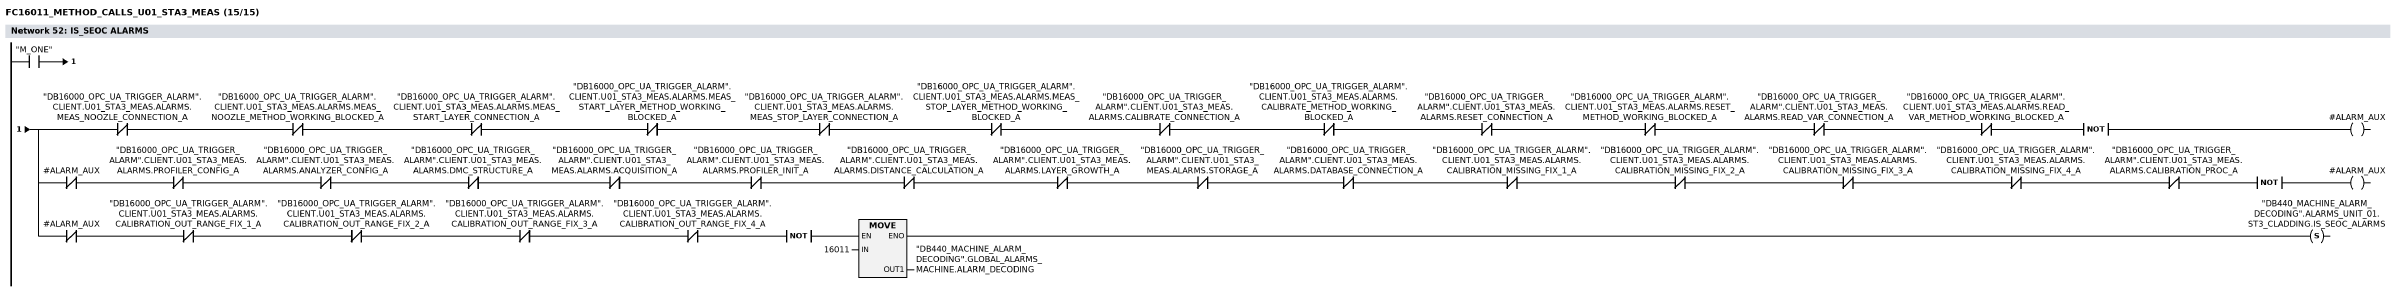
   RUNG wire#powerrail
      Contact( "M_ONE" )
      wire#w1
      I_Contact( "DB16000_OPC_UA_TRIGGER_ALARM".CLIENT.U01_STA3_MEAS.ALARMS.MEAS_NOOZLE_CONNECTION_A )
      I_Contact( "DB16000_OPC_UA_TRIGGER_ALARM".CLIENT.U01_STA3_MEAS.ALARMS.MEAS_NOOZLE_METHOD_WORKING_BLOCKED_A )
      I_Contact( "DB16000_OPC_UA_TRIGGER_ALARM".CLIENT.U01_STA3_MEAS.ALARMS.MEAS_START_LAYER_CONNECTION_A )
      I_Contact( "DB16000_OPC_UA_TRIGGER_ALARM".CLIENT.U01_STA3_MEAS.ALARMS.MEAS_START_LAYER_METHOD_WORKING_BLOCKED_A )
      I_Contact( "DB16000_OPC_UA_TRIGGER_ALARM".CLIENT.U01_STA3_MEAS.ALARMS.MEAS_STOP_LAYER_CONNECTION_A )
      I_Contact( "DB16000_OPC_UA_TRIGGER_ALARM".CLIENT.U01_STA3_MEAS.ALARMS.MEAS_STOP_LAYER_METHOD_WORKING_BLOCKED_A )
      I_Contact( "DB16000_OPC_UA_TRIGGER_ALARM".CLIENT.U01_STA3_MEAS.ALARMS.CALIBRATE_CONNECTION_A )
      I_Contact( "DB16000_OPC_UA_TRIGGER_ALARM".CLIENT.U01_STA3_MEAS.ALARMS.CALIBRATE_METHOD_WORKING_BLOCKED_A )
      I_Contact( "DB16000_OPC_UA_TRIGGER_ALARM".CLIENT.U01_STA3_MEAS.ALARMS.RESET_CONNECTION_A )
      I_Contact( "DB16000_OPC_UA_TRIGGER_ALARM".CLIENT.U01_STA3_MEAS.ALARMS.RESET_METHOD_WORKING_BLOCKED_A )
      I_Contact( "DB16000_OPC_UA_TRIGGER_ALARM".CLIENT.U01_STA3_MEAS.ALARMS.READ_VAR_CONNECTION_A )
      I_Contact( "DB16000_OPC_UA_TRIGGER_ALARM".CLIENT.U01_STA3_MEAS.ALARMS.READ_VAR_METHOD_WORKING_BLOCKED_A )
      Not()
      Coil( #ALARM_AUX )
   END_RUNG
   RUNG wire#w1
      I_Contact( #ALARM_AUX )
      I_Contact( "DB16000_OPC_UA_TRIGGER_ALARM".CLIENT.U01_STA3_MEAS.ALARMS.PROFILER_CONFIG_A )
      I_Contact( "DB16000_OPC_UA_TRIGGER_ALARM".CLIENT.U01_STA3_MEAS.ALARMS.ANALYZER_CONFIG_A )
      I_Contact( "DB16000_OPC_UA_TRIGGER_ALARM".CLIENT.U01_STA3_MEAS.ALARMS.DMC_STRUCTURE_A )
      I_Contact( "DB16000_OPC_UA_TRIGGER_ALARM".CLIENT.U01_STA3_MEAS.ALARMS.ACQUISITION_A )
      I_Contact( "DB16000_OPC_UA_TRIGGER_ALARM".CLIENT.U01_STA3_MEAS.ALARMS.PROFILER_INIT_A )
      I_Contact( "DB16000_OPC_UA_TRIGGER_ALARM".CLIENT.U01_STA3_MEAS.ALARMS.DISTANCE_CALCULATION_A )
      I_Contact( "DB16000_OPC_UA_TRIGGER_ALARM".CLIENT.U01_STA3_MEAS.ALARMS.LAYER_GROWTH_A )
      I_Contact( "DB16000_OPC_UA_TRIGGER_ALARM".CLIENT.U01_STA3_MEAS.ALARMS.STORAGE_A )
      I_Contact( "DB16000_OPC_UA_TRIGGER_ALARM".CLIENT.U01_STA3_MEAS.ALARMS.DATABASE_CONNECTION_A )
      I_Contact( "DB16000_OPC_UA_TRIGGER_ALARM".CLIENT.U01_STA3_MEAS.ALARMS.CALIBRATION_MISSING_FIX_1_A )
      I_Contact( "DB16000_OPC_UA_TRIGGER_ALARM".CLIENT.U01_STA3_MEAS.ALARMS.CALIBRATION_MISSING_FIX_2_A )
      I_Contact( "DB16000_OPC_UA_TRIGGER_ALARM".CLIENT.U01_STA3_MEAS.ALARMS.CALIBRATION_MISSING_FIX_3_A )
      I_Contact( "DB16000_OPC_UA_TRIGGER_ALARM".CLIENT.U01_STA3_MEAS.ALARMS.CALIBRATION_MISSING_FIX_4_A )
      I_Contact( "DB16000_OPC_UA_TRIGGER_ALARM".CLIENT.U01_STA3_MEAS.ALARMS.CALIBRATION_PROC_A )
      Not()
      Coil( #ALARM_AUX )
   END_RUNG
   RUNG wire#w1
      I_Contact( #ALARM_AUX )
      I_Contact( "DB16000_OPC_UA_TRIGGER_ALARM".CLIENT.U01_STA3_MEAS.ALARMS.CALIBRATION_OUT_RANGE_FIX_1_A )
      I_Contact( "DB16000_OPC_UA_TRIGGER_ALARM".CLIENT.U01_STA3_MEAS.ALARMS.CALIBRATION_OUT_RANGE_FIX_2_A )
      I_Contact( "DB16000_OPC_UA_TRIGGER_ALARM".CLIENT.U01_STA3_MEAS.ALARMS.CALIBRATION_OUT_RANGE_FIX_3_A )
      I_Contact( "DB16000_OPC_UA_TRIGGER_ALARM".CLIENT.U01_STA3_MEAS.ALARMS.CALIBRATION_OUT_RANGE_FIX_4_A )
      Not()
      Move(in := 16011, out1 => "DB440_MACHINE_ALARM_DECODING".GLOBAL_ALARMS_MACHINE.ALARM_DECODING)
      S_Coil( "DB440_MACHINE_ALARM_DECODING".ALARMS_UNIT_01.ST3_CLADDING.IS_SEOC_ALARMS )
   END_RUNG
   // the same network as SCL:
   #ALARM_AUX := NOT ("M_ONE" AND NOT "DB16000_OPC_UA_TRIGGER_ALARM".CLIENT.U01_STA3_MEAS.ALARMS.MEAS_NOOZLE_CONNECTION_A AND NOT "DB16000_OPC_UA_TRIGGER_ALARM".CLIENT.U01_STA3_MEAS.ALARMS.MEAS_NOOZLE_METHOD_WORKING_BLOCKED_A AND NOT "DB16000_OPC_UA_TRIGGER_ALARM".CLIENT.U01_STA3_MEAS.ALARMS.MEAS_START_LAYER_CONNECTION_A AND NOT "DB16000_OPC_UA_TRIGGER_ALARM".CLIENT.U01_STA3_MEAS.ALARMS.MEAS_START_LAYER_METHOD_WORKING_BLOCKED_A AND NOT "DB16000_OPC_UA_TRIGGER_ALARM".CLIENT.U01_STA3_MEAS.ALARMS.MEAS_STOP_LAYER_CONNECTION_A AND NOT "DB16000_OPC_UA_TRIGGER_ALARM".CLIENT.U01_STA3_MEAS.ALARMS.MEAS_STOP_LAYER_METHOD_WORKING_BLOCKED_A AND NOT "DB16000_OPC_UA_TRIGGER_ALARM".CLIENT.U01_STA3_MEAS.ALARMS.CALIBRATE_CONNECTION_A AND NOT "DB16000_OPC_UA_TRIGGER_ALARM".CLIENT.U01_STA3_MEAS.ALARMS.CALIBRATE_METHOD_WORKING_BLOCKED_A AND NOT "DB16000_OPC_UA_TRIGGER_ALARM".CLIENT.U01_STA3_MEAS.ALARMS.RESET_CONNECTION_A AND NOT "DB16000_OPC_UA_TRIGGER_ALARM".CLIENT.U01_STA3_MEAS.ALARMS.RESET_METHOD_WORKING_BLOCKED_A AND NOT "DB16000_OPC_UA_TRIGGER_ALARM".CLIENT.U01_STA3_MEAS.ALARMS.READ_VAR_CONNECTION_A AND NOT "DB16000_OPC_UA_TRIGGER_ALARM".CLIENT.U01_STA3_MEAS.ALARMS.READ_VAR_METHOD_WORKING_BLOCKED_A);
   #ALARM_AUX := NOT ("M_ONE" AND NOT #ALARM_AUX AND NOT "DB16000_OPC_UA_TRIGGER_ALARM".CLIENT.U01_STA3_MEAS.ALARMS.PROFILER_CONFIG_A AND NOT "DB16000_OPC_UA_TRIGGER_ALARM".CLIENT.U01_STA3_MEAS.ALARMS.ANALYZER_CONFIG_A AND NOT "DB16000_OPC_UA_TRIGGER_ALARM".CLIENT.U01_STA3_MEAS.ALARMS.DMC_STRUCTURE_A AND NOT "DB16000_OPC_UA_TRIGGER_ALARM".CLIENT.U01_STA3_MEAS.ALARMS.ACQUISITION_A AND NOT "DB16000_OPC_UA_TRIGGER_ALARM".CLIENT.U01_STA3_MEAS.ALARMS.PROFILER_INIT_A AND NOT "DB16000_OPC_UA_TRIGGER_ALARM".CLIENT.U01_STA3_MEAS.ALARMS.DISTANCE_CALCULATION_A AND NOT "DB16000_OPC_UA_TRIGGER_ALARM".CLIENT.U01_STA3_MEAS.ALARMS.LAYER_GROWTH_A AND NOT "DB16000_OPC_UA_TRIGGER_ALARM".CLIENT.U01_STA3_MEAS.ALARMS.STORAGE_A AND NOT "DB16000_OPC_UA_TRIGGER_ALARM".CLIENT.U01_STA3_MEAS.ALARMS.DATABASE_CONNECTION_A AND NOT "DB16000_OPC_UA_TRIGGER_ALARM".CLIENT.U01_STA3_MEAS.ALARMS.CALIBRATION_MISSING_FIX_1_A AND NOT "DB16000_OPC_UA_TRIGGER_ALARM".CLIENT.U01_STA3_MEAS.ALARMS.CALIBRATION_MISSING_FIX_2_A AND NOT "DB16000_OPC_UA_TRIGGER_ALARM".CLIENT.U01_STA3_MEAS.ALARMS.CALIBRATION_MISSING_FIX_3_A AND NOT "DB16000_OPC_UA_TRIGGER_ALARM".CLIENT.U01_STA3_MEAS.ALARMS.CALIBRATION_MISSING_FIX_4_A AND NOT "DB16000_OPC_UA_TRIGGER_ALARM".CLIENT.U01_STA3_MEAS.ALARMS.CALIBRATION_PROC_A);
   IF NOT ("M_ONE" AND NOT #ALARM_AUX AND NOT "DB16000_OPC_UA_TRIGGER_ALARM".CLIENT.U01_STA3_MEAS.ALARMS.CALIBRATION_OUT_RANGE_FIX_1_A AND NOT "DB16000_OPC_UA_TRIGGER_ALARM".CLIENT.U01_STA3_MEAS.ALARMS.CALIBRATION_OUT_RANGE_FIX_2_A AND NOT "DB16000_OPC_UA_TRIGGER_ALARM".CLIENT.U01_STA3_MEAS.ALARMS.CALIBRATION_OUT_RANGE_FIX_3_A AND NOT "DB16000_OPC_UA_TRIGGER_ALARM".CLIENT.U01_STA3_MEAS.ALARMS.CALIBRATION_OUT_RANGE_FIX_4_A) THEN
       "DB440_MACHINE_ALARM_DECODING".GLOBAL_ALARMS_MACHINE.ALARM_DECODING := 16011;
       "DB440_MACHINE_ALARM_DECODING".ALARMS_UNIT_01.ST3_CLADDING.IS_SEOC_ALARMS := TRUE;
   END_IF;
END_REGION
END_FUNCTION
